REGION Network 12: UNIT 02 STATION 1 PART A PRESENT
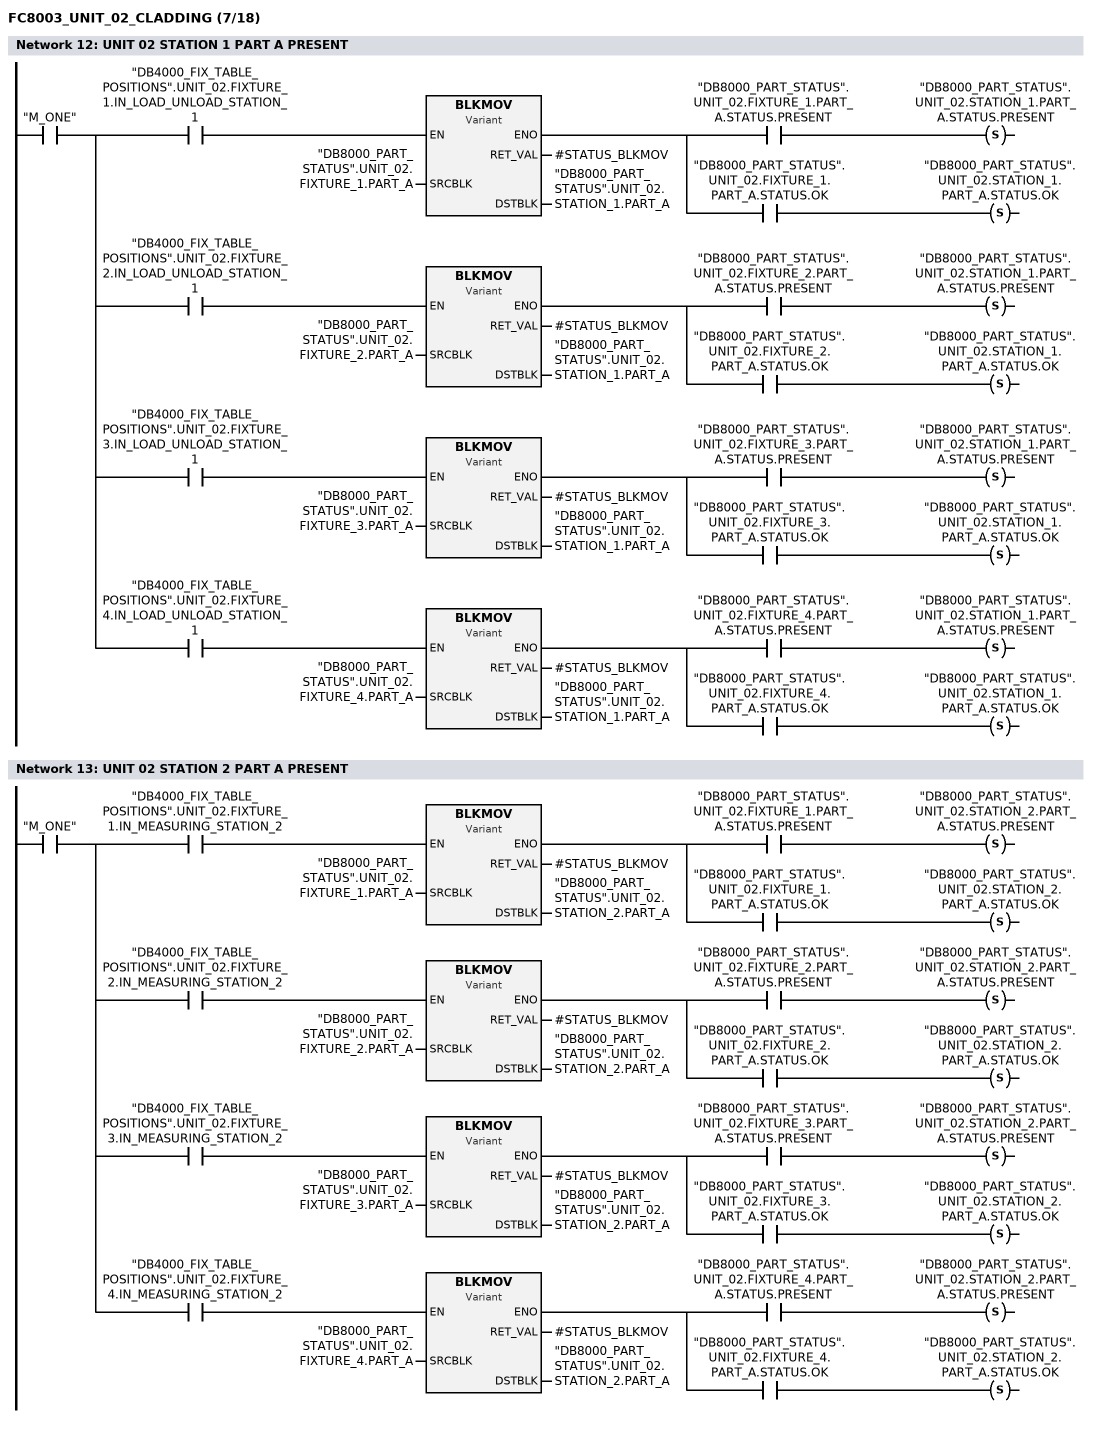
   RUNG wire#powerrail
      Contact( "M_ONE" )
      wire#w1
      Contact( "DB4000_FIX_TABLE_POSITIONS".UNIT_02.FIXTURE_1.IN_LOAD_UNLOAD_STATION_1 )
      { S7_Templates := "blk_type := Variant" } BLKMOV(SRCBLK := "DB8000_PART_STATUS".UNIT_02.FIXTURE_1.PART_A, RET_VAL => #STATUS_BLKMOV, DSTBLK => "DB8000_PART_STATUS".UNIT_02.STATION_1.PART_A)
      wire#w2
      Contact( "DB8000_PART_STATUS".UNIT_02.FIXTURE_1.PART_A.STATUS.PRESENT )
      S_Coil( "DB8000_PART_STATUS".UNIT_02.STATION_1.PART_A.STATUS.PRESENT )
   END_RUNG
   RUNG wire#w2
      Contact( "DB8000_PART_STATUS".UNIT_02.FIXTURE_1.PART_A.STATUS.OK )
      S_Coil( "DB8000_PART_STATUS".UNIT_02.STATION_1.PART_A.STATUS.OK )
   END_RUNG
   RUNG wire#w1
      Contact( "DB4000_FIX_TABLE_POSITIONS".UNIT_02.FIXTURE_2.IN_LOAD_UNLOAD_STATION_1 )
      { S7_Templates := "blk_type := Variant" } BLKMOV(SRCBLK := "DB8000_PART_STATUS".UNIT_02.FIXTURE_2.PART_A, RET_VAL => #STATUS_BLKMOV, DSTBLK => "DB8000_PART_STATUS".UNIT_02.STATION_1.PART_A)
      wire#w3
      Contact( "DB8000_PART_STATUS".UNIT_02.FIXTURE_2.PART_A.STATUS.PRESENT )
      S_Coil( "DB8000_PART_STATUS".UNIT_02.STATION_1.PART_A.STATUS.PRESENT )
   END_RUNG
   RUNG wire#w3
      Contact( "DB8000_PART_STATUS".UNIT_02.FIXTURE_2.PART_A.STATUS.OK )
      S_Coil( "DB8000_PART_STATUS".UNIT_02.STATION_1.PART_A.STATUS.OK )
   END_RUNG
   RUNG wire#w1
      Contact( "DB4000_FIX_TABLE_POSITIONS".UNIT_02.FIXTURE_3.IN_LOAD_UNLOAD_STATION_1 )
      { S7_Templates := "blk_type := Variant" } BLKMOV(SRCBLK := "DB8000_PART_STATUS".UNIT_02.FIXTURE_3.PART_A, RET_VAL => #STATUS_BLKMOV, DSTBLK => "DB8000_PART_STATUS".UNIT_02.STATION_1.PART_A)
      wire#w4
      Contact( "DB8000_PART_STATUS".UNIT_02.FIXTURE_3.PART_A.STATUS.PRESENT )
      S_Coil( "DB8000_PART_STATUS".UNIT_02.STATION_1.PART_A.STATUS.PRESENT )
   END_RUNG
   RUNG wire#w4
      Contact( "DB8000_PART_STATUS".UNIT_02.FIXTURE_3.PART_A.STATUS.OK )
      S_Coil( "DB8000_PART_STATUS".UNIT_02.STATION_1.PART_A.STATUS.OK )
   END_RUNG
   RUNG wire#w1
      Contact( "DB4000_FIX_TABLE_POSITIONS".UNIT_02.FIXTURE_4.IN_LOAD_UNLOAD_STATION_1 )
      { S7_Templates := "blk_type := Variant" } BLKMOV(SRCBLK := "DB8000_PART_STATUS".UNIT_02.FIXTURE_4.PART_A, RET_VAL => #STATUS_BLKMOV, DSTBLK => "DB8000_PART_STATUS".UNIT_02.STATION_1.PART_A)
      wire#w5
      Contact( "DB8000_PART_STATUS".UNIT_02.FIXTURE_4.PART_A.STATUS.PRESENT )
      S_Coil( "DB8000_PART_STATUS".UNIT_02.STATION_1.PART_A.STATUS.PRESENT )
   END_RUNG
   RUNG wire#w5
      Contact( "DB8000_PART_STATUS".UNIT_02.FIXTURE_4.PART_A.STATUS.OK )
      S_Coil( "DB8000_PART_STATUS".UNIT_02.STATION_1.PART_A.STATUS.OK )
   END_RUNG
   // the same network as SCL:
   #_w1 := "M_ONE" AND "DB4000_FIX_TABLE_POSITIONS".UNIT_02.FIXTURE_1.IN_LOAD_UNLOAD_STATION_1;
   #_w3 := "M_ONE";
   #STATUS_BLKMOV := BLKMOV(EN := #_w1,
                           SRCBLK := "DB8000_PART_STATUS".UNIT_02.FIXTURE_1.PART_A,
                           DSTBLK => "DB8000_PART_STATUS".UNIT_02.STATION_1.PART_A,
                           ENO => #_w2);
   IF #_w2 AND "DB8000_PART_STATUS".UNIT_02.FIXTURE_1.PART_A.STATUS.PRESENT THEN
       "DB8000_PART_STATUS".UNIT_02.STATION_1.PART_A.STATUS.PRESENT := TRUE;
   END_IF;
   IF #_w2 AND "DB8000_PART_STATUS".UNIT_02.FIXTURE_1.PART_A.STATUS.OK THEN
       "DB8000_PART_STATUS".UNIT_02.STATION_1.PART_A.STATUS.OK := TRUE;
   END_IF;
   #_w4 := #_w3 AND "DB4000_FIX_TABLE_POSITIONS".UNIT_02.FIXTURE_2.IN_LOAD_UNLOAD_STATION_1;
   #STATUS_BLKMOV := BLKMOV(EN := #_w4,
                           SRCBLK := "DB8000_PART_STATUS".UNIT_02.FIXTURE_2.PART_A,
                           DSTBLK => "DB8000_PART_STATUS".UNIT_02.STATION_1.PART_A,
                           ENO => #_w5);
   IF #_w5 AND "DB8000_PART_STATUS".UNIT_02.FIXTURE_2.PART_A.STATUS.PRESENT THEN
       "DB8000_PART_STATUS".UNIT_02.STATION_1.PART_A.STATUS.PRESENT := TRUE;
   END_IF;
   IF #_w5 AND "DB8000_PART_STATUS".UNIT_02.FIXTURE_2.PART_A.STATUS.OK THEN
       "DB8000_PART_STATUS".UNIT_02.STATION_1.PART_A.STATUS.OK := TRUE;
   END_IF;
   #_w6 := #_w3 AND "DB4000_FIX_TABLE_POSITIONS".UNIT_02.FIXTURE_3.IN_LOAD_UNLOAD_STATION_1;
   #STATUS_BLKMOV := BLKMOV(EN := #_w6,
                           SRCBLK := "DB8000_PART_STATUS".UNIT_02.FIXTURE_3.PART_A,
                           DSTBLK => "DB8000_PART_STATUS".UNIT_02.STATION_1.PART_A,
                           ENO => #_w7);
   IF #_w7 AND "DB8000_PART_STATUS".UNIT_02.FIXTURE_3.PART_A.STATUS.PRESENT THEN
       "DB8000_PART_STATUS".UNIT_02.STATION_1.PART_A.STATUS.PRESENT := TRUE;
   END_IF;
   IF #_w7 AND "DB8000_PART_STATUS".UNIT_02.FIXTURE_3.PART_A.STATUS.OK THEN
       "DB8000_PART_STATUS".UNIT_02.STATION_1.PART_A.STATUS.OK := TRUE;
   END_IF;
   #_w8 := #_w3 AND "DB4000_FIX_TABLE_POSITIONS".UNIT_02.FIXTURE_4.IN_LOAD_UNLOAD_STATION_1;
   #STATUS_BLKMOV := BLKMOV(EN := #_w8,
                           SRCBLK := "DB8000_PART_STATUS".UNIT_02.FIXTURE_4.PART_A,
                           DSTBLK => "DB8000_PART_STATUS".UNIT_02.STATION_1.PART_A,
                           ENO => #_w9);
   IF #_w9 AND "DB8000_PART_STATUS".UNIT_02.FIXTURE_4.PART_A.STATUS.PRESENT THEN
       "DB8000_PART_STATUS".UNIT_02.STATION_1.PART_A.STATUS.PRESENT := TRUE;
   END_IF;
   IF #_w9 AND "DB8000_PART_STATUS".UNIT_02.FIXTURE_4.PART_A.STATUS.OK THEN
       "DB8000_PART_STATUS".UNIT_02.STATION_1.PART_A.STATUS.OK := TRUE;
   END_IF;
END_REGION

REGION Network 13: UNIT 02 STATION 2 PART A PRESENT
   RUNG wire#powerrail
      Contact( "M_ONE" )
      wire#w1
      Contact( "DB4000_FIX_TABLE_POSITIONS".UNIT_02.FIXTURE_1.IN_MEASURING_STATION_2 )
      { S7_Templates := "blk_type := Variant" } BLKMOV(SRCBLK := "DB8000_PART_STATUS".UNIT_02.FIXTURE_1.PART_A, RET_VAL => #STATUS_BLKMOV, DSTBLK => "DB8000_PART_STATUS".UNIT_02.STATION_2.PART_A)
      wire#w2
      Contact( "DB8000_PART_STATUS".UNIT_02.FIXTURE_1.PART_A.STATUS.PRESENT )
      S_Coil( "DB8000_PART_STATUS".UNIT_02.STATION_2.PART_A.STATUS.PRESENT )
   END_RUNG
   RUNG wire#w2
      Contact( "DB8000_PART_STATUS".UNIT_02.FIXTURE_1.PART_A.STATUS.OK )
      S_Coil( "DB8000_PART_STATUS".UNIT_02.STATION_2.PART_A.STATUS.OK )
   END_RUNG
   RUNG wire#w1
      Contact( "DB4000_FIX_TABLE_POSITIONS".UNIT_02.FIXTURE_2.IN_MEASURING_STATION_2 )
      { S7_Templates := "blk_type := Variant" } BLKMOV(SRCBLK := "DB8000_PART_STATUS".UNIT_02.FIXTURE_2.PART_A, RET_VAL => #STATUS_BLKMOV, DSTBLK => "DB8000_PART_STATUS".UNIT_02.STATION_2.PART_A)
      wire#w3
      Contact( "DB8000_PART_STATUS".UNIT_02.FIXTURE_2.PART_A.STATUS.PRESENT )
      S_Coil( "DB8000_PART_STATUS".UNIT_02.STATION_2.PART_A.STATUS.PRESENT )
   END_RUNG
   RUNG wire#w3
      Contact( "DB8000_PART_STATUS".UNIT_02.FIXTURE_2.PART_A.STATUS.OK )
      S_Coil( "DB8000_PART_STATUS".UNIT_02.STATION_2.PART_A.STATUS.OK )
   END_RUNG
   RUNG wire#w1
      Contact( "DB4000_FIX_TABLE_POSITIONS".UNIT_02.FIXTURE_3.IN_MEASURING_STATION_2 )
      { S7_Templates := "blk_type := Variant" } BLKMOV(SRCBLK := "DB8000_PART_STATUS".UNIT_02.FIXTURE_3.PART_A, RET_VAL => #STATUS_BLKMOV, DSTBLK => "DB8000_PART_STATUS".UNIT_02.STATION_2.PART_A)
      wire#w4
      Contact( "DB8000_PART_STATUS".UNIT_02.FIXTURE_3.PART_A.STATUS.PRESENT )
      S_Coil( "DB8000_PART_STATUS".UNIT_02.STATION_2.PART_A.STATUS.PRESENT )
   END_RUNG
   RUNG wire#w4
      Contact( "DB8000_PART_STATUS".UNIT_02.FIXTURE_3.PART_A.STATUS.OK )
      S_Coil( "DB8000_PART_STATUS".UNIT_02.STATION_2.PART_A.STATUS.OK )
   END_RUNG
   RUNG wire#w1
      Contact( "DB4000_FIX_TABLE_POSITIONS".UNIT_02.FIXTURE_4.IN_MEASURING_STATION_2 )
      { S7_Templates := "blk_type := Variant" } BLKMOV(SRCBLK := "DB8000_PART_STATUS".UNIT_02.FIXTURE_4.PART_A, RET_VAL => #STATUS_BLKMOV, DSTBLK => "DB8000_PART_STATUS".UNIT_02.STATION_2.PART_A)
      wire#w5
      Contact( "DB8000_PART_STATUS".UNIT_02.FIXTURE_4.PART_A.STATUS.PRESENT )
      S_Coil( "DB8000_PART_STATUS".UNIT_02.STATION_2.PART_A.STATUS.PRESENT )
   END_RUNG
   RUNG wire#w5
      Contact( "DB8000_PART_STATUS".UNIT_02.FIXTURE_4.PART_A.STATUS.OK )
      S_Coil( "DB8000_PART_STATUS".UNIT_02.STATION_2.PART_A.STATUS.OK )
   END_RUNG
   // the same network as SCL:
   #_w1 := "M_ONE" AND "DB4000_FIX_TABLE_POSITIONS".UNIT_02.FIXTURE_1.IN_MEASURING_STATION_2;
   #_w3 := "M_ONE";
   #STATUS_BLKMOV := BLKMOV(EN := #_w1,
                           SRCBLK := "DB8000_PART_STATUS".UNIT_02.FIXTURE_1.PART_A,
                           DSTBLK => "DB8000_PART_STATUS".UNIT_02.STATION_2.PART_A,
                           ENO => #_w2);
   IF #_w2 AND "DB8000_PART_STATUS".UNIT_02.FIXTURE_1.PART_A.STATUS.PRESENT THEN
       "DB8000_PART_STATUS".UNIT_02.STATION_2.PART_A.STATUS.PRESENT := TRUE;
   END_IF;
   IF #_w2 AND "DB8000_PART_STATUS".UNIT_02.FIXTURE_1.PART_A.STATUS.OK THEN
       "DB8000_PART_STATUS".UNIT_02.STATION_2.PART_A.STATUS.OK := TRUE;
   END_IF;
   #_w4 := #_w3 AND "DB4000_FIX_TABLE_POSITIONS".UNIT_02.FIXTURE_2.IN_MEASURING_STATION_2;
   #STATUS_BLKMOV := BLKMOV(EN := #_w4,
                           SRCBLK := "DB8000_PART_STATUS".UNIT_02.FIXTURE_2.PART_A,
                           DSTBLK => "DB8000_PART_STATUS".UNIT_02.STATION_2.PART_A,
                           ENO => #_w5);
   IF #_w5 AND "DB8000_PART_STATUS".UNIT_02.FIXTURE_2.PART_A.STATUS.PRESENT THEN
       "DB8000_PART_STATUS".UNIT_02.STATION_2.PART_A.STATUS.PRESENT := TRUE;
   END_IF;
   IF #_w5 AND "DB8000_PART_STATUS".UNIT_02.FIXTURE_2.PART_A.STATUS.OK THEN
       "DB8000_PART_STATUS".UNIT_02.STATION_2.PART_A.STATUS.OK := TRUE;
   END_IF;
   #_w6 := #_w3 AND "DB4000_FIX_TABLE_POSITIONS".UNIT_02.FIXTURE_3.IN_MEASURING_STATION_2;
   #STATUS_BLKMOV := BLKMOV(EN := #_w6,
                           SRCBLK := "DB8000_PART_STATUS".UNIT_02.FIXTURE_3.PART_A,
                           DSTBLK => "DB8000_PART_STATUS".UNIT_02.STATION_2.PART_A,
                           ENO => #_w7);
   IF #_w7 AND "DB8000_PART_STATUS".UNIT_02.FIXTURE_3.PART_A.STATUS.PRESENT THEN
       "DB8000_PART_STATUS".UNIT_02.STATION_2.PART_A.STATUS.PRESENT := TRUE;
   END_IF;
   IF #_w7 AND "DB8000_PART_STATUS".UNIT_02.FIXTURE_3.PART_A.STATUS.OK THEN
       "DB8000_PART_STATUS".UNIT_02.STATION_2.PART_A.STATUS.OK := TRUE;
   END_IF;
   #_w8 := #_w3 AND "DB4000_FIX_TABLE_POSITIONS".UNIT_02.FIXTURE_4.IN_MEASURING_STATION_2;
   #STATUS_BLKMOV := BLKMOV(EN := #_w8,
                           SRCBLK := "DB8000_PART_STATUS".UNIT_02.FIXTURE_4.PART_A,
                           DSTBLK => "DB8000_PART_STATUS".UNIT_02.STATION_2.PART_A,
                           ENO => #_w9);
   IF #_w9 AND "DB8000_PART_STATUS".UNIT_02.FIXTURE_4.PART_A.STATUS.PRESENT THEN
       "DB8000_PART_STATUS".UNIT_02.STATION_2.PART_A.STATUS.PRESENT := TRUE;
   END_IF;
   IF #_w9 AND "DB8000_PART_STATUS".UNIT_02.FIXTURE_4.PART_A.STATUS.OK THEN
       "DB8000_PART_STATUS".UNIT_02.STATION_2.PART_A.STATUS.OK := TRUE;
   END_IF;
END_REGION

REGION Network 14: UNIT 02 STATION 3 PART A PRESENT
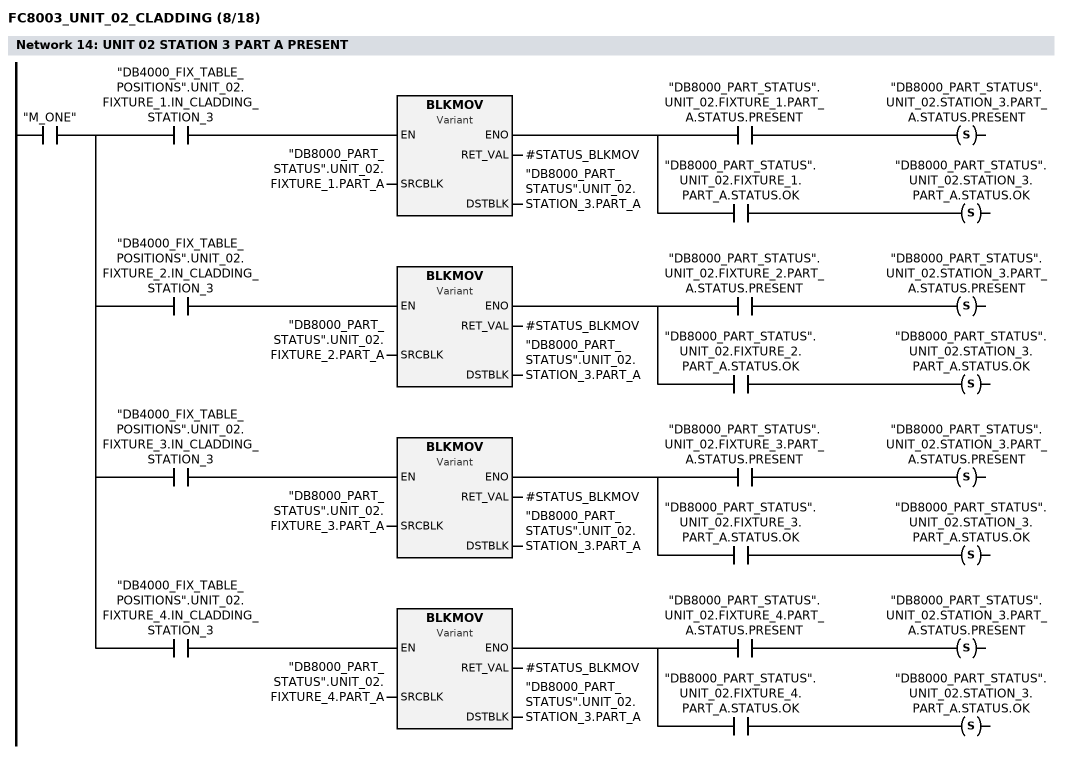
   RUNG wire#powerrail
      Contact( "M_ONE" )
      wire#w1
      Contact( "DB4000_FIX_TABLE_POSITIONS".UNIT_02.FIXTURE_1.IN_CLADDING_STATION_3 )
      { S7_Templates := "blk_type := Variant" } BLKMOV(SRCBLK := "DB8000_PART_STATUS".UNIT_02.FIXTURE_1.PART_A, RET_VAL => #STATUS_BLKMOV, DSTBLK => "DB8000_PART_STATUS".UNIT_02.STATION_3.PART_A)
      wire#w2
      Contact( "DB8000_PART_STATUS".UNIT_02.FIXTURE_1.PART_A.STATUS.PRESENT )
      S_Coil( "DB8000_PART_STATUS".UNIT_02.STATION_3.PART_A.STATUS.PRESENT )
   END_RUNG
   RUNG wire#w2
      Contact( "DB8000_PART_STATUS".UNIT_02.FIXTURE_1.PART_A.STATUS.OK )
      S_Coil( "DB8000_PART_STATUS".UNIT_02.STATION_3.PART_A.STATUS.OK )
   END_RUNG
   RUNG wire#w1
      Contact( "DB4000_FIX_TABLE_POSITIONS".UNIT_02.FIXTURE_2.IN_CLADDING_STATION_3 )
      { S7_Templates := "blk_type := Variant" } BLKMOV(SRCBLK := "DB8000_PART_STATUS".UNIT_02.FIXTURE_2.PART_A, RET_VAL => #STATUS_BLKMOV, DSTBLK => "DB8000_PART_STATUS".UNIT_02.STATION_3.PART_A)
      wire#w3
      Contact( "DB8000_PART_STATUS".UNIT_02.FIXTURE_2.PART_A.STATUS.PRESENT )
      S_Coil( "DB8000_PART_STATUS".UNIT_02.STATION_3.PART_A.STATUS.PRESENT )
   END_RUNG
   RUNG wire#w3
      Contact( "DB8000_PART_STATUS".UNIT_02.FIXTURE_2.PART_A.STATUS.OK )
      S_Coil( "DB8000_PART_STATUS".UNIT_02.STATION_3.PART_A.STATUS.OK )
   END_RUNG
   RUNG wire#w1
      Contact( "DB4000_FIX_TABLE_POSITIONS".UNIT_02.FIXTURE_3.IN_CLADDING_STATION_3 )
      { S7_Templates := "blk_type := Variant" } BLKMOV(SRCBLK := "DB8000_PART_STATUS".UNIT_02.FIXTURE_3.PART_A, RET_VAL => #STATUS_BLKMOV, DSTBLK => "DB8000_PART_STATUS".UNIT_02.STATION_3.PART_A)
      wire#w4
      Contact( "DB8000_PART_STATUS".UNIT_02.FIXTURE_3.PART_A.STATUS.PRESENT )
      S_Coil( "DB8000_PART_STATUS".UNIT_02.STATION_3.PART_A.STATUS.PRESENT )
   END_RUNG
   RUNG wire#w4
      Contact( "DB8000_PART_STATUS".UNIT_02.FIXTURE_3.PART_A.STATUS.OK )
      S_Coil( "DB8000_PART_STATUS".UNIT_02.STATION_3.PART_A.STATUS.OK )
   END_RUNG
   RUNG wire#w1
      Contact( "DB4000_FIX_TABLE_POSITIONS".UNIT_02.FIXTURE_4.IN_CLADDING_STATION_3 )
      { S7_Templates := "blk_type := Variant" } BLKMOV(SRCBLK := "DB8000_PART_STATUS".UNIT_02.FIXTURE_4.PART_A, RET_VAL => #STATUS_BLKMOV, DSTBLK => "DB8000_PART_STATUS".UNIT_02.STATION_3.PART_A)
      wire#w5
      Contact( "DB8000_PART_STATUS".UNIT_02.FIXTURE_4.PART_A.STATUS.PRESENT )
      S_Coil( "DB8000_PART_STATUS".UNIT_02.STATION_3.PART_A.STATUS.PRESENT )
   END_RUNG
   RUNG wire#w5
      Contact( "DB8000_PART_STATUS".UNIT_02.FIXTURE_4.PART_A.STATUS.OK )
      S_Coil( "DB8000_PART_STATUS".UNIT_02.STATION_3.PART_A.STATUS.OK )
   END_RUNG
   // the same network as SCL:
   #_w1 := "M_ONE" AND "DB4000_FIX_TABLE_POSITIONS".UNIT_02.FIXTURE_1.IN_CLADDING_STATION_3;
   #_w3 := "M_ONE";
   #STATUS_BLKMOV := BLKMOV(EN := #_w1,
                           SRCBLK := "DB8000_PART_STATUS".UNIT_02.FIXTURE_1.PART_A,
                           DSTBLK => "DB8000_PART_STATUS".UNIT_02.STATION_3.PART_A,
                           ENO => #_w2);
   IF #_w2 AND "DB8000_PART_STATUS".UNIT_02.FIXTURE_1.PART_A.STATUS.PRESENT THEN
       "DB8000_PART_STATUS".UNIT_02.STATION_3.PART_A.STATUS.PRESENT := TRUE;
   END_IF;
   IF #_w2 AND "DB8000_PART_STATUS".UNIT_02.FIXTURE_1.PART_A.STATUS.OK THEN
       "DB8000_PART_STATUS".UNIT_02.STATION_3.PART_A.STATUS.OK := TRUE;
   END_IF;
   #_w4 := #_w3 AND "DB4000_FIX_TABLE_POSITIONS".UNIT_02.FIXTURE_2.IN_CLADDING_STATION_3;
   #STATUS_BLKMOV := BLKMOV(EN := #_w4,
                           SRCBLK := "DB8000_PART_STATUS".UNIT_02.FIXTURE_2.PART_A,
                           DSTBLK => "DB8000_PART_STATUS".UNIT_02.STATION_3.PART_A,
                           ENO => #_w5);
   IF #_w5 AND "DB8000_PART_STATUS".UNIT_02.FIXTURE_2.PART_A.STATUS.PRESENT THEN
       "DB8000_PART_STATUS".UNIT_02.STATION_3.PART_A.STATUS.PRESENT := TRUE;
   END_IF;
   IF #_w5 AND "DB8000_PART_STATUS".UNIT_02.FIXTURE_2.PART_A.STATUS.OK THEN
       "DB8000_PART_STATUS".UNIT_02.STATION_3.PART_A.STATUS.OK := TRUE;
   END_IF;
   #_w6 := #_w3 AND "DB4000_FIX_TABLE_POSITIONS".UNIT_02.FIXTURE_3.IN_CLADDING_STATION_3;
   #STATUS_BLKMOV := BLKMOV(EN := #_w6,
                           SRCBLK := "DB8000_PART_STATUS".UNIT_02.FIXTURE_3.PART_A,
                           DSTBLK => "DB8000_PART_STATUS".UNIT_02.STATION_3.PART_A,
                           ENO => #_w7);
   IF #_w7 AND "DB8000_PART_STATUS".UNIT_02.FIXTURE_3.PART_A.STATUS.PRESENT THEN
       "DB8000_PART_STATUS".UNIT_02.STATION_3.PART_A.STATUS.PRESENT := TRUE;
   END_IF;
   IF #_w7 AND "DB8000_PART_STATUS".UNIT_02.FIXTURE_3.PART_A.STATUS.OK THEN
       "DB8000_PART_STATUS".UNIT_02.STATION_3.PART_A.STATUS.OK := TRUE;
   END_IF;
   #_w8 := #_w3 AND "DB4000_FIX_TABLE_POSITIONS".UNIT_02.FIXTURE_4.IN_CLADDING_STATION_3;
   #STATUS_BLKMOV := BLKMOV(EN := #_w8,
                           SRCBLK := "DB8000_PART_STATUS".UNIT_02.FIXTURE_4.PART_A,
                           DSTBLK => "DB8000_PART_STATUS".UNIT_02.STATION_3.PART_A,
                           ENO => #_w9);
   IF #_w9 AND "DB8000_PART_STATUS".UNIT_02.FIXTURE_4.PART_A.STATUS.PRESENT THEN
       "DB8000_PART_STATUS".UNIT_02.STATION_3.PART_A.STATUS.PRESENT := TRUE;
   END_IF;
   IF #_w9 AND "DB8000_PART_STATUS".UNIT_02.FIXTURE_4.PART_A.STATUS.OK THEN
       "DB8000_PART_STATUS".UNIT_02.STATION_3.PART_A.STATUS.OK := TRUE;
   END_IF;
END_REGION

REGION Network 15: UNIT 02 STATION 4 PART A PRESENT
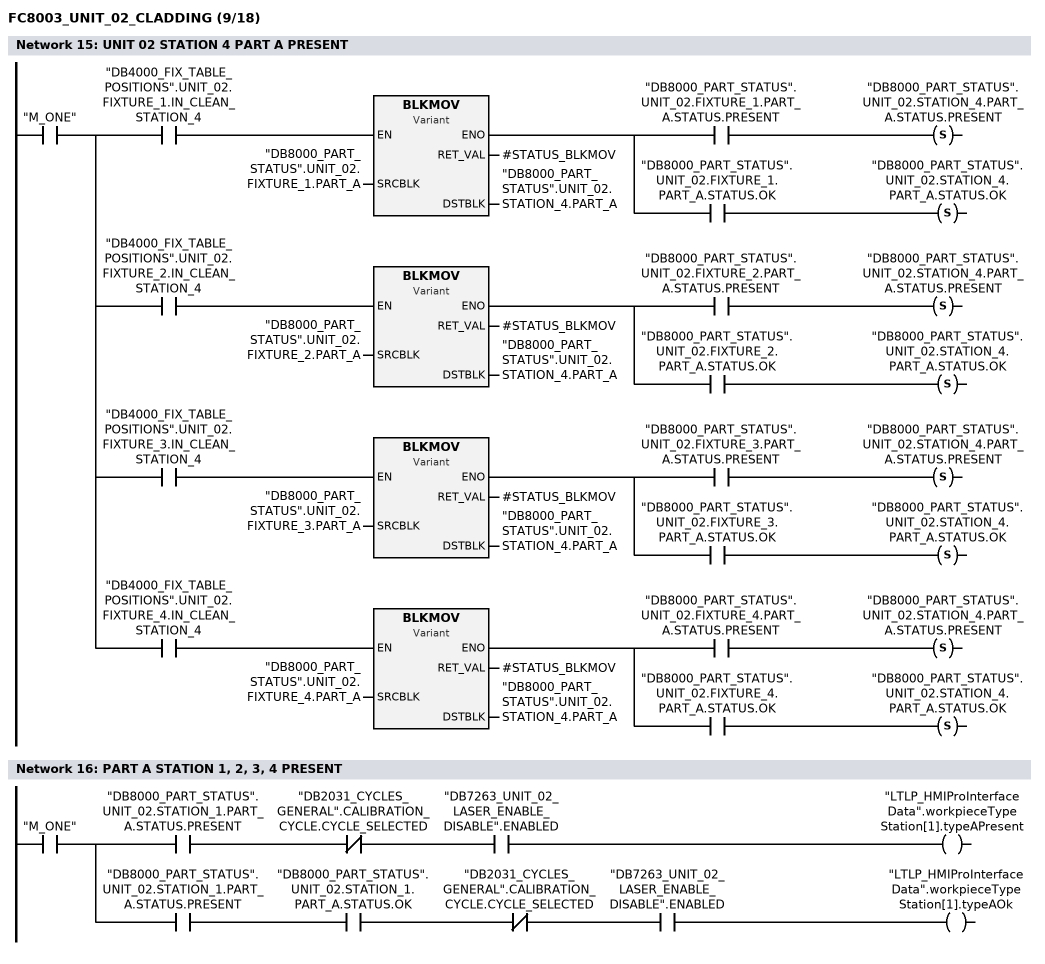
   RUNG wire#powerrail
      Contact( "M_ONE" )
      wire#w1
      Contact( "DB4000_FIX_TABLE_POSITIONS".UNIT_02.FIXTURE_1.IN_CLEAN_STATION_4 )
      { S7_Templates := "blk_type := Variant" } BLKMOV(SRCBLK := "DB8000_PART_STATUS".UNIT_02.FIXTURE_1.PART_A, RET_VAL => #STATUS_BLKMOV, DSTBLK => "DB8000_PART_STATUS".UNIT_02.STATION_4.PART_A)
      wire#w2
      Contact( "DB8000_PART_STATUS".UNIT_02.FIXTURE_1.PART_A.STATUS.PRESENT )
      S_Coil( "DB8000_PART_STATUS".UNIT_02.STATION_4.PART_A.STATUS.PRESENT )
   END_RUNG
   RUNG wire#w2
      Contact( "DB8000_PART_STATUS".UNIT_02.FIXTURE_1.PART_A.STATUS.OK )
      S_Coil( "DB8000_PART_STATUS".UNIT_02.STATION_4.PART_A.STATUS.OK )
   END_RUNG
   RUNG wire#w1
      Contact( "DB4000_FIX_TABLE_POSITIONS".UNIT_02.FIXTURE_2.IN_CLEAN_STATION_4 )
      { S7_Templates := "blk_type := Variant" } BLKMOV(SRCBLK := "DB8000_PART_STATUS".UNIT_02.FIXTURE_2.PART_A, RET_VAL => #STATUS_BLKMOV, DSTBLK => "DB8000_PART_STATUS".UNIT_02.STATION_4.PART_A)
      wire#w3
      Contact( "DB8000_PART_STATUS".UNIT_02.FIXTURE_2.PART_A.STATUS.PRESENT )
      S_Coil( "DB8000_PART_STATUS".UNIT_02.STATION_4.PART_A.STATUS.PRESENT )
   END_RUNG
   RUNG wire#w3
      Contact( "DB8000_PART_STATUS".UNIT_02.FIXTURE_2.PART_A.STATUS.OK )
      S_Coil( "DB8000_PART_STATUS".UNIT_02.STATION_4.PART_A.STATUS.OK )
   END_RUNG
   RUNG wire#w1
      Contact( "DB4000_FIX_TABLE_POSITIONS".UNIT_02.FIXTURE_3.IN_CLEAN_STATION_4 )
      { S7_Templates := "blk_type := Variant" } BLKMOV(SRCBLK := "DB8000_PART_STATUS".UNIT_02.FIXTURE_3.PART_A, RET_VAL => #STATUS_BLKMOV, DSTBLK => "DB8000_PART_STATUS".UNIT_02.STATION_4.PART_A)
      wire#w4
      Contact( "DB8000_PART_STATUS".UNIT_02.FIXTURE_3.PART_A.STATUS.PRESENT )
      S_Coil( "DB8000_PART_STATUS".UNIT_02.STATION_4.PART_A.STATUS.PRESENT )
   END_RUNG
   RUNG wire#w4
      Contact( "DB8000_PART_STATUS".UNIT_02.FIXTURE_3.PART_A.STATUS.OK )
      S_Coil( "DB8000_PART_STATUS".UNIT_02.STATION_4.PART_A.STATUS.OK )
   END_RUNG
   RUNG wire#w1
      Contact( "DB4000_FIX_TABLE_POSITIONS".UNIT_02.FIXTURE_4.IN_CLEAN_STATION_4 )
      { S7_Templates := "blk_type := Variant" } BLKMOV(SRCBLK := "DB8000_PART_STATUS".UNIT_02.FIXTURE_4.PART_A, RET_VAL => #STATUS_BLKMOV, DSTBLK => "DB8000_PART_STATUS".UNIT_02.STATION_4.PART_A)
      wire#w5
      Contact( "DB8000_PART_STATUS".UNIT_02.FIXTURE_4.PART_A.STATUS.PRESENT )
      S_Coil( "DB8000_PART_STATUS".UNIT_02.STATION_4.PART_A.STATUS.PRESENT )
   END_RUNG
   RUNG wire#w5
      Contact( "DB8000_PART_STATUS".UNIT_02.FIXTURE_4.PART_A.STATUS.OK )
      S_Coil( "DB8000_PART_STATUS".UNIT_02.STATION_4.PART_A.STATUS.OK )
   END_RUNG
   // the same network as SCL:
   #_w1 := "M_ONE" AND "DB4000_FIX_TABLE_POSITIONS".UNIT_02.FIXTURE_1.IN_CLEAN_STATION_4;
   #_w3 := "M_ONE";
   #STATUS_BLKMOV := BLKMOV(EN := #_w1,
                           SRCBLK := "DB8000_PART_STATUS".UNIT_02.FIXTURE_1.PART_A,
                           DSTBLK => "DB8000_PART_STATUS".UNIT_02.STATION_4.PART_A,
                           ENO => #_w2);
   IF #_w2 AND "DB8000_PART_STATUS".UNIT_02.FIXTURE_1.PART_A.STATUS.PRESENT THEN
       "DB8000_PART_STATUS".UNIT_02.STATION_4.PART_A.STATUS.PRESENT := TRUE;
   END_IF;
   IF #_w2 AND "DB8000_PART_STATUS".UNIT_02.FIXTURE_1.PART_A.STATUS.OK THEN
       "DB8000_PART_STATUS".UNIT_02.STATION_4.PART_A.STATUS.OK := TRUE;
   END_IF;
   #_w4 := #_w3 AND "DB4000_FIX_TABLE_POSITIONS".UNIT_02.FIXTURE_2.IN_CLEAN_STATION_4;
   #STATUS_BLKMOV := BLKMOV(EN := #_w4,
                           SRCBLK := "DB8000_PART_STATUS".UNIT_02.FIXTURE_2.PART_A,
                           DSTBLK => "DB8000_PART_STATUS".UNIT_02.STATION_4.PART_A,
                           ENO => #_w5);
   IF #_w5 AND "DB8000_PART_STATUS".UNIT_02.FIXTURE_2.PART_A.STATUS.PRESENT THEN
       "DB8000_PART_STATUS".UNIT_02.STATION_4.PART_A.STATUS.PRESENT := TRUE;
   END_IF;
   IF #_w5 AND "DB8000_PART_STATUS".UNIT_02.FIXTURE_2.PART_A.STATUS.OK THEN
       "DB8000_PART_STATUS".UNIT_02.STATION_4.PART_A.STATUS.OK := TRUE;
   END_IF;
   #_w6 := #_w3 AND "DB4000_FIX_TABLE_POSITIONS".UNIT_02.FIXTURE_3.IN_CLEAN_STATION_4;
   #STATUS_BLKMOV := BLKMOV(EN := #_w6,
                           SRCBLK := "DB8000_PART_STATUS".UNIT_02.FIXTURE_3.PART_A,
                           DSTBLK => "DB8000_PART_STATUS".UNIT_02.STATION_4.PART_A,
                           ENO => #_w7);
   IF #_w7 AND "DB8000_PART_STATUS".UNIT_02.FIXTURE_3.PART_A.STATUS.PRESENT THEN
       "DB8000_PART_STATUS".UNIT_02.STATION_4.PART_A.STATUS.PRESENT := TRUE;
   END_IF;
   IF #_w7 AND "DB8000_PART_STATUS".UNIT_02.FIXTURE_3.PART_A.STATUS.OK THEN
       "DB8000_PART_STATUS".UNIT_02.STATION_4.PART_A.STATUS.OK := TRUE;
   END_IF;
   #_w8 := #_w3 AND "DB4000_FIX_TABLE_POSITIONS".UNIT_02.FIXTURE_4.IN_CLEAN_STATION_4;
   #STATUS_BLKMOV := BLKMOV(EN := #_w8,
                           SRCBLK := "DB8000_PART_STATUS".UNIT_02.FIXTURE_4.PART_A,
                           DSTBLK => "DB8000_PART_STATUS".UNIT_02.STATION_4.PART_A,
                           ENO => #_w9);
   IF #_w9 AND "DB8000_PART_STATUS".UNIT_02.FIXTURE_4.PART_A.STATUS.PRESENT THEN
       "DB8000_PART_STATUS".UNIT_02.STATION_4.PART_A.STATUS.PRESENT := TRUE;
   END_IF;
   IF #_w9 AND "DB8000_PART_STATUS".UNIT_02.FIXTURE_4.PART_A.STATUS.OK THEN
       "DB8000_PART_STATUS".UNIT_02.STATION_4.PART_A.STATUS.OK := TRUE;
   END_IF;
END_REGION

REGION Network 16: PART A STATION 1, 2, 3, 4 PRESENT
   RUNG wire#powerrail
      Contact( "M_ONE" )
      wire#w1
      Contact( "DB8000_PART_STATUS".UNIT_02.STATION_1.PART_A.STATUS.PRESENT )
      I_Contact( "DB2031_CYCLES_GENERAL".CALIBRATION_CYCLE.CYCLE_SELECTED )
      Contact( "DB7263_UNIT_02_LASER_ENABLE_DISABLE".ENABLED )
      Coil( "LTLP_HMIProInterfaceData".workpieceTypeStation[1].typeAPresent )
   END_RUNG
   RUNG wire#w1
      Contact( "DB8000_PART_STATUS".UNIT_02.STATION_1.PART_A.STATUS.PRESENT )
      Contact( "DB8000_PART_STATUS".UNIT_02.STATION_1.PART_A.STATUS.OK )
      I_Contact( "DB2031_CYCLES_GENERAL".CALIBRATION_CYCLE.CYCLE_SELECTED )
      Contact( "DB7263_UNIT_02_LASER_ENABLE_DISABLE".ENABLED )
      Coil( "LTLP_HMIProInterfaceData".workpieceTypeStation[1].typeAOk )
   END_RUNG
   // the same network as SCL:
   "LTLP_HMIProInterfaceData".workpieceTypeStation[1].typeAPresent := "M_ONE" AND "DB8000_PART_STATUS".UNIT_02.STATION_1.PART_A.STATUS.PRESENT AND NOT "DB2031_CYCLES_GENERAL".CALIBRATION_CYCLE.CYCLE_SELECTED AND "DB7263_UNIT_02_LASER_ENABLE_DISABLE".ENABLED;
   "LTLP_HMIProInterfaceData".workpieceTypeStation[1].typeAOk := "M_ONE" AND "DB8000_PART_STATUS".UNIT_02.STATION_1.PART_A.STATUS.PRESENT AND "DB8000_PART_STATUS".UNIT_02.STATION_1.PART_A.STATUS.OK AND NOT "DB2031_CYCLES_GENERAL".CALIBRATION_CYCLE.CYCLE_SELECTED AND "DB7263_UNIT_02_LASER_ENABLE_DISABLE".ENABLED;
END_REGION

REGION Network 17: PART A FIXTURE 1, 2, 3, 4 RESET STATUS TO ZERO
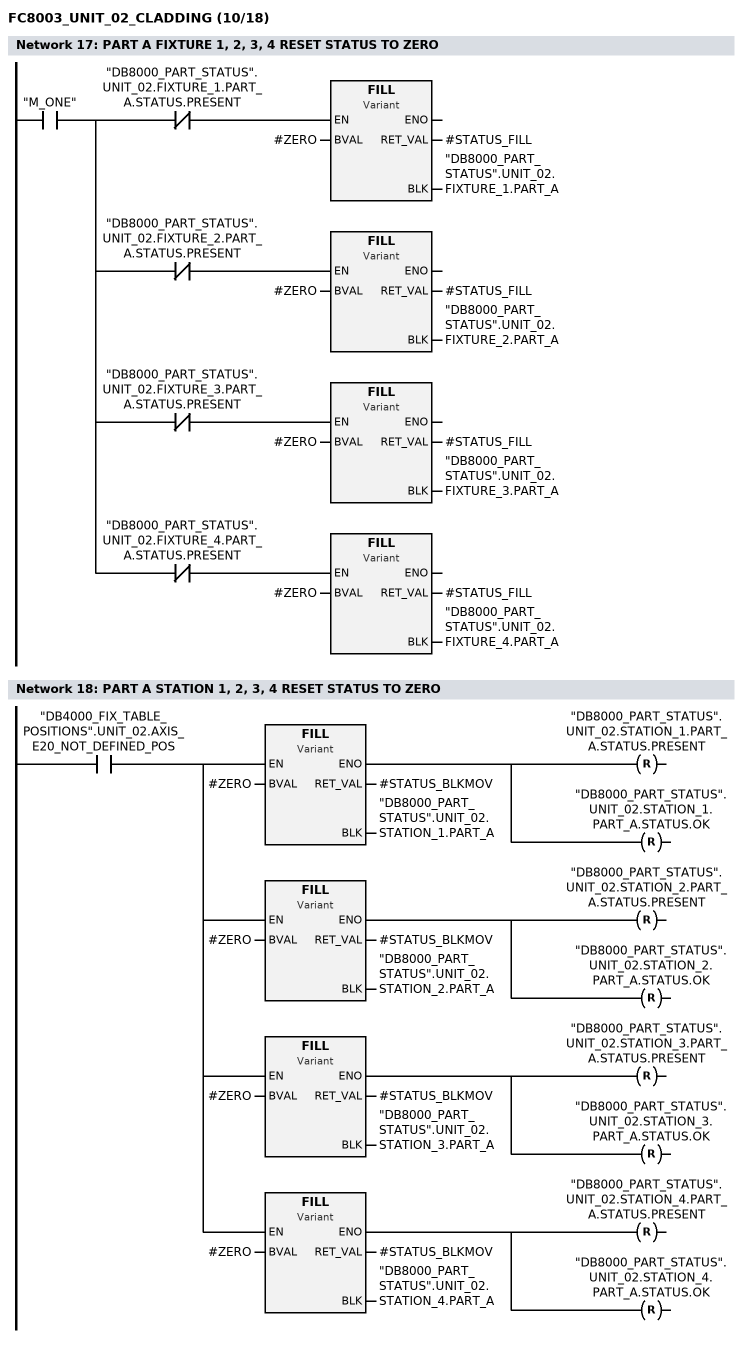
   RUNG wire#powerrail
      Contact( "M_ONE" )
      wire#w1
      I_Contact( "DB8000_PART_STATUS".UNIT_02.FIXTURE_1.PART_A.STATUS.PRESENT )
      { S7_Templates := "ptr_type := Variant" } FILL(BVAL := #ZERO, RET_VAL => #STATUS_FILL, BLK => "DB8000_PART_STATUS".UNIT_02.FIXTURE_1.PART_A)
   END_RUNG
   RUNG wire#w1
      I_Contact( "DB8000_PART_STATUS".UNIT_02.FIXTURE_2.PART_A.STATUS.PRESENT )
      { S7_Templates := "ptr_type := Variant" } FILL(BVAL := #ZERO, RET_VAL => #STATUS_FILL, BLK => "DB8000_PART_STATUS".UNIT_02.FIXTURE_2.PART_A)
   END_RUNG
   RUNG wire#w1
      I_Contact( "DB8000_PART_STATUS".UNIT_02.FIXTURE_3.PART_A.STATUS.PRESENT )
      { S7_Templates := "ptr_type := Variant" } FILL(BVAL := #ZERO, RET_VAL => #STATUS_FILL, BLK => "DB8000_PART_STATUS".UNIT_02.FIXTURE_3.PART_A)
   END_RUNG
   RUNG wire#w1
      I_Contact( "DB8000_PART_STATUS".UNIT_02.FIXTURE_4.PART_A.STATUS.PRESENT )
      { S7_Templates := "ptr_type := Variant" } FILL(BVAL := #ZERO, RET_VAL => #STATUS_FILL, BLK => "DB8000_PART_STATUS".UNIT_02.FIXTURE_4.PART_A)
   END_RUNG
   // the same network as SCL:
   #_w1 := "M_ONE";
   IF "M_ONE" AND NOT "DB8000_PART_STATUS".UNIT_02.FIXTURE_1.PART_A.STATUS.PRESENT THEN
       #STATUS_FILL := FILL(BVAL := #ZERO, BLK => "DB8000_PART_STATUS".UNIT_02.FIXTURE_1.PART_A);
   END_IF;
   IF #_w1 AND NOT "DB8000_PART_STATUS".UNIT_02.FIXTURE_2.PART_A.STATUS.PRESENT THEN
       #STATUS_FILL := FILL(BVAL := #ZERO, BLK => "DB8000_PART_STATUS".UNIT_02.FIXTURE_2.PART_A);
   END_IF;
   IF #_w1 AND NOT "DB8000_PART_STATUS".UNIT_02.FIXTURE_3.PART_A.STATUS.PRESENT THEN
       #STATUS_FILL := FILL(BVAL := #ZERO, BLK => "DB8000_PART_STATUS".UNIT_02.FIXTURE_3.PART_A);
   END_IF;
   IF #_w1 AND NOT "DB8000_PART_STATUS".UNIT_02.FIXTURE_4.PART_A.STATUS.PRESENT THEN
       #STATUS_FILL := FILL(BVAL := #ZERO, BLK => "DB8000_PART_STATUS".UNIT_02.FIXTURE_4.PART_A);
   END_IF;
END_REGION

REGION Network 18: PART A STATION 1, 2, 3, 4 RESET STATUS TO ZERO
   RUNG wire#powerrail
      Contact( "DB4000_FIX_TABLE_POSITIONS".UNIT_02.AXIS_E20_NOT_DEFINED_POS )
      wire#w1
      { S7_Templates := "ptr_type := Variant" } FILL(BVAL := #ZERO, RET_VAL => #STATUS_BLKMOV, BLK => "DB8000_PART_STATUS".UNIT_02.STATION_1.PART_A)
      wire#w2
      R_Coil( "DB8000_PART_STATUS".UNIT_02.STATION_1.PART_A.STATUS.PRESENT )
   END_RUNG
   RUNG wire#w2
      R_Coil( "DB8000_PART_STATUS".UNIT_02.STATION_1.PART_A.STATUS.OK )
   END_RUNG
   RUNG wire#w1
      { S7_Templates := "ptr_type := Variant" } FILL(BVAL := #ZERO, RET_VAL => #STATUS_BLKMOV, BLK => "DB8000_PART_STATUS".UNIT_02.STATION_2.PART_A)
      wire#w3
      R_Coil( "DB8000_PART_STATUS".UNIT_02.STATION_2.PART_A.STATUS.PRESENT )
   END_RUNG
   RUNG wire#w3
      R_Coil( "DB8000_PART_STATUS".UNIT_02.STATION_2.PART_A.STATUS.OK )
   END_RUNG
   RUNG wire#w1
      { S7_Templates := "ptr_type := Variant" } FILL(BVAL := #ZERO, RET_VAL => #STATUS_BLKMOV, BLK => "DB8000_PART_STATUS".UNIT_02.STATION_3.PART_A)
      wire#w4
      R_Coil( "DB8000_PART_STATUS".UNIT_02.STATION_3.PART_A.STATUS.PRESENT )
   END_RUNG
   RUNG wire#w4
      R_Coil( "DB8000_PART_STATUS".UNIT_02.STATION_3.PART_A.STATUS.OK )
   END_RUNG
   RUNG wire#w1
      { S7_Templates := "ptr_type := Variant" } FILL(BVAL := #ZERO, RET_VAL => #STATUS_BLKMOV, BLK => "DB8000_PART_STATUS".UNIT_02.STATION_4.PART_A)
      wire#w5
      R_Coil( "DB8000_PART_STATUS".UNIT_02.STATION_4.PART_A.STATUS.PRESENT )
   END_RUNG
   RUNG wire#w5
      R_Coil( "DB8000_PART_STATUS".UNIT_02.STATION_4.PART_A.STATUS.OK )
   END_RUNG
   // the same network as SCL:
   #_w2 := "DB4000_FIX_TABLE_POSITIONS".UNIT_02.AXIS_E20_NOT_DEFINED_POS;
   #STATUS_BLKMOV := FILL(EN := "DB4000_FIX_TABLE_POSITIONS".UNIT_02.AXIS_E20_NOT_DEFINED_POS,
                          BVAL := #ZERO,
                          BLK => "DB8000_PART_STATUS".UNIT_02.STATION_1.PART_A,
                          ENO => #_w1);
   IF #_w1 THEN
       "DB8000_PART_STATUS".UNIT_02.STATION_1.PART_A.STATUS.PRESENT := FALSE;
       "DB8000_PART_STATUS".UNIT_02.STATION_1.PART_A.STATUS.OK := FALSE;
   END_IF;
   #STATUS_BLKMOV := FILL(EN := #_w2,
                          BVAL := #ZERO,
                          BLK => "DB8000_PART_STATUS".UNIT_02.STATION_2.PART_A,
                          ENO => #_w3);
   IF #_w3 THEN
       "DB8000_PART_STATUS".UNIT_02.STATION_2.PART_A.STATUS.PRESENT := FALSE;
       "DB8000_PART_STATUS".UNIT_02.STATION_2.PART_A.STATUS.OK := FALSE;
   END_IF;
   #STATUS_BLKMOV := FILL(EN := #_w2,
                          BVAL := #ZERO,
                          BLK => "DB8000_PART_STATUS".UNIT_02.STATION_3.PART_A,
                          ENO => #_w4);
   IF #_w4 THEN
       "DB8000_PART_STATUS".UNIT_02.STATION_3.PART_A.STATUS.PRESENT := FALSE;
       "DB8000_PART_STATUS".UNIT_02.STATION_3.PART_A.STATUS.OK := FALSE;
   END_IF;
   #STATUS_BLKMOV := FILL(EN := #_w2,
                          BVAL := #ZERO,
                          BLK => "DB8000_PART_STATUS".UNIT_02.STATION_4.PART_A,
                          ENO => #_w5);
   IF #_w5 THEN
       "DB8000_PART_STATUS".UNIT_02.STATION_4.PART_A.STATUS.PRESENT := FALSE;
       "DB8000_PART_STATUS".UNIT_02.STATION_4.PART_A.STATUS.OK := FALSE;
   END_IF;
END_REGION

REGION Network 19: PART A FIXTURE 1 COLOR STATUS
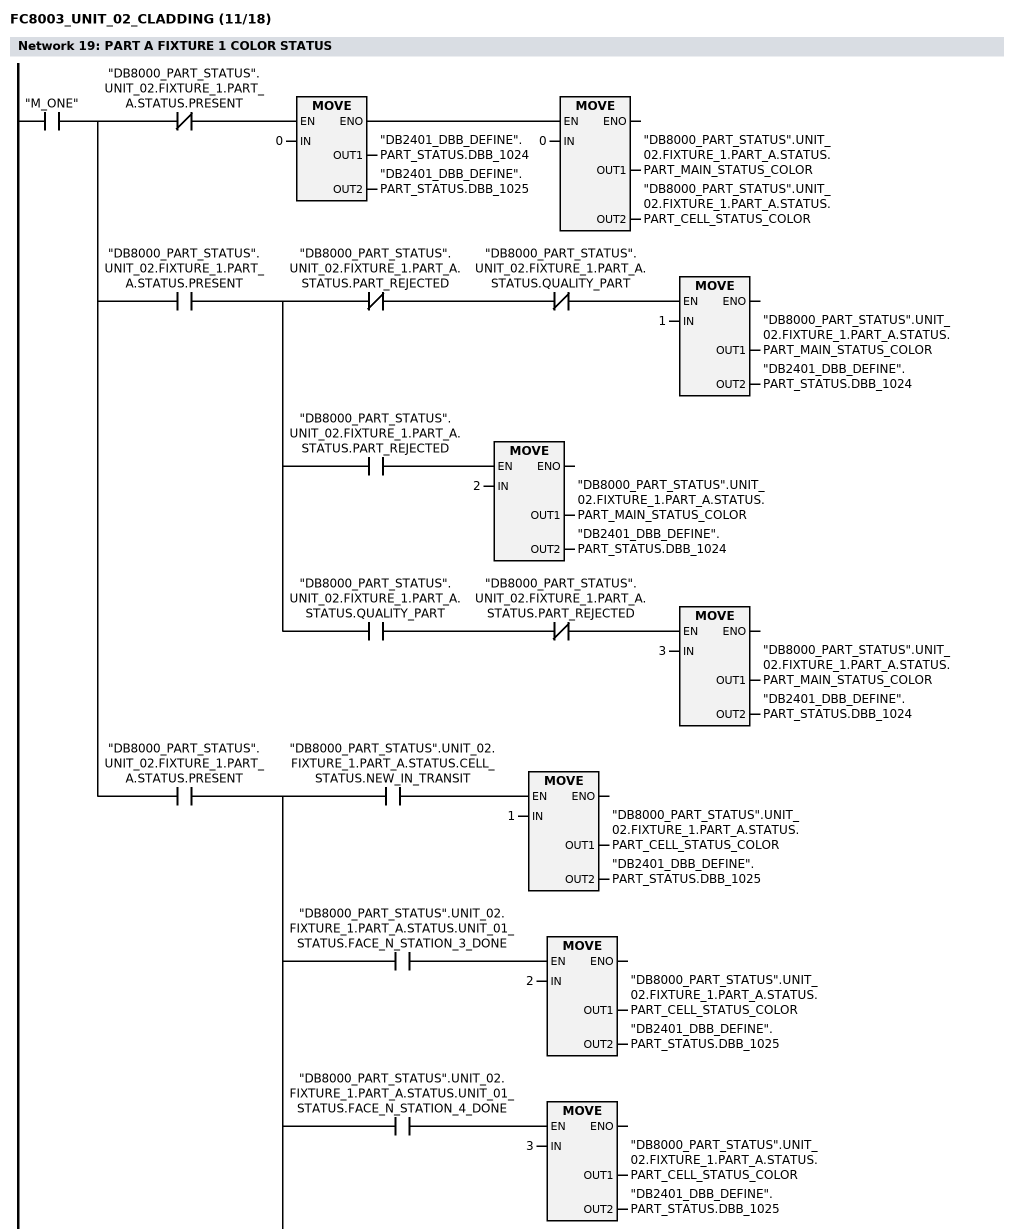
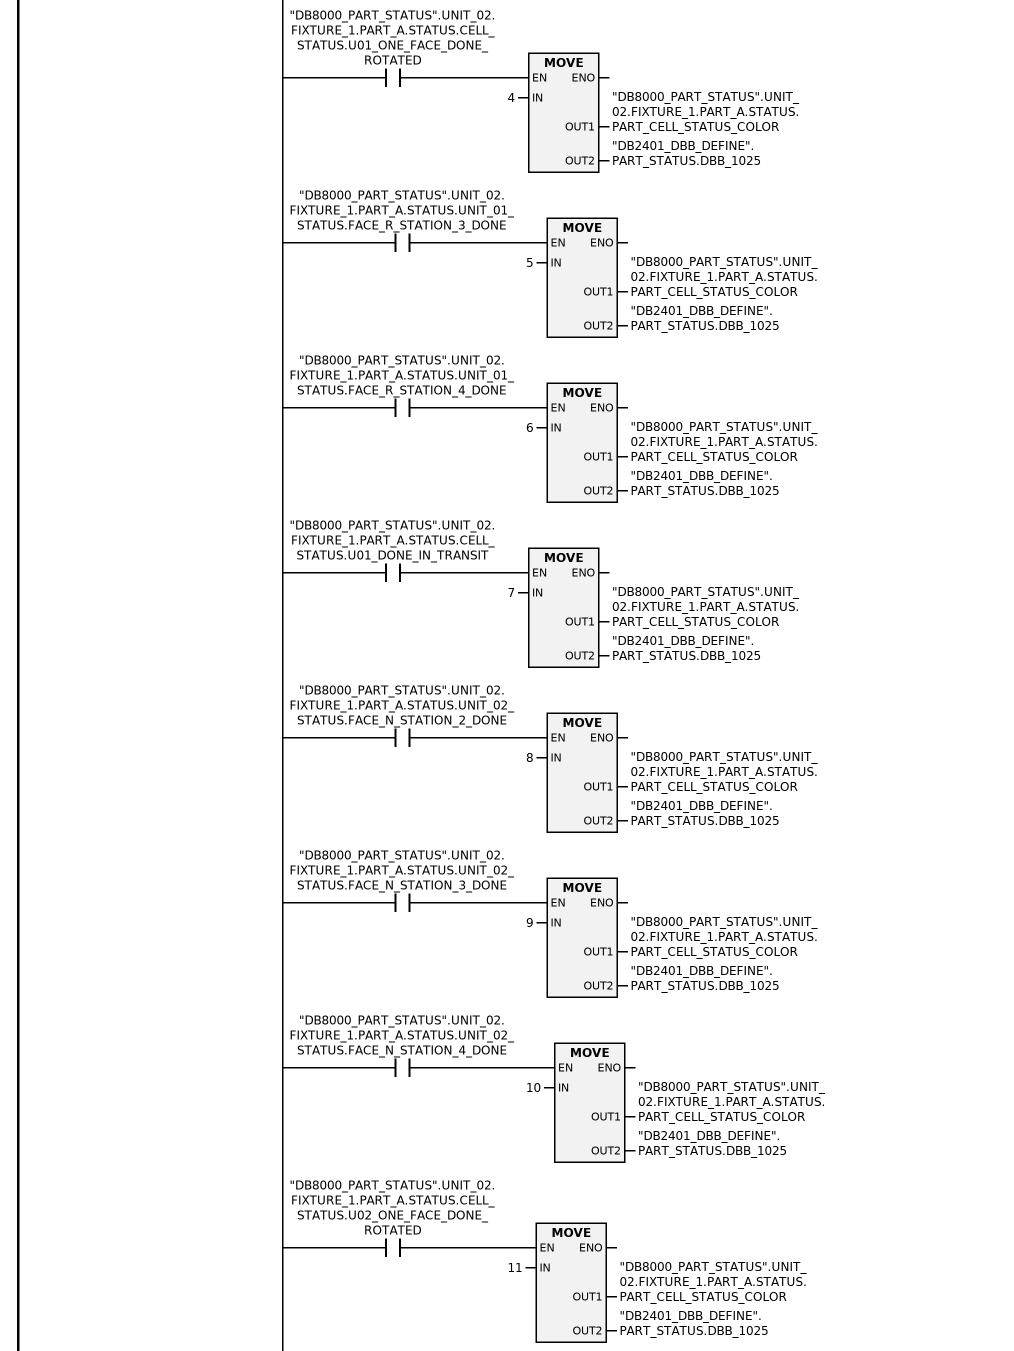
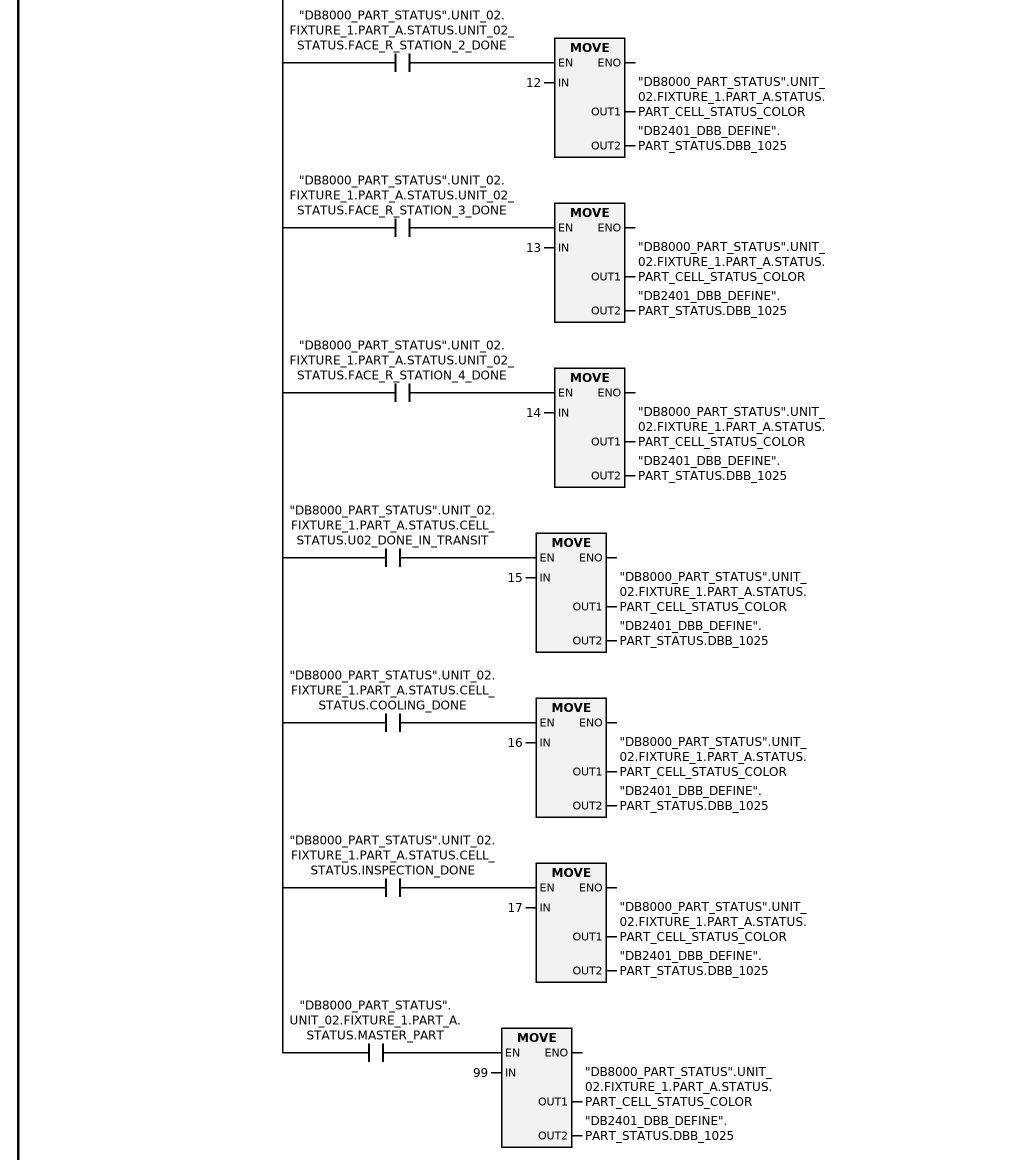
   RUNG wire#powerrail
      Contact( "M_ONE" )
      wire#w1
      I_Contact( "DB8000_PART_STATUS".UNIT_02.FIXTURE_1.PART_A.STATUS.PRESENT )
      { S7_GenerateENO := "TRUE" } Move(in := 0, out1 => "DB2401_DBB_DEFINE".PART_STATUS.DBB_1024, out2 => "DB2401_DBB_DEFINE".PART_STATUS.DBB_1025)
      { S7_GenerateENO := "TRUE" } Move(in := 0, out1 => "DB8000_PART_STATUS".UNIT_02.FIXTURE_1.PART_A.STATUS.PART_MAIN_STATUS_COLOR, out2 => "DB8000_PART_STATUS".UNIT_02.FIXTURE_1.PART_A.STATUS.PART_CELL_STATUS_COLOR)
   END_RUNG
   RUNG wire#w1
      Contact( "DB8000_PART_STATUS".UNIT_02.FIXTURE_1.PART_A.STATUS.PRESENT )
      wire#w2
      I_Contact( "DB8000_PART_STATUS".UNIT_02.FIXTURE_1.PART_A.STATUS.PART_REJECTED )
      I_Contact( "DB8000_PART_STATUS".UNIT_02.FIXTURE_1.PART_A.STATUS.QUALITY_PART )
      { S7_GenerateENO := "TRUE" } Move(in := 1, out1 => "DB8000_PART_STATUS".UNIT_02.FIXTURE_1.PART_A.STATUS.PART_MAIN_STATUS_COLOR, out2 => "DB2401_DBB_DEFINE".PART_STATUS.DBB_1024)
   END_RUNG
   RUNG wire#w2
      Contact( "DB8000_PART_STATUS".UNIT_02.FIXTURE_1.PART_A.STATUS.PART_REJECTED )
      { S7_GenerateENO := "TRUE" } Move(in := 2, out1 => "DB8000_PART_STATUS".UNIT_02.FIXTURE_1.PART_A.STATUS.PART_MAIN_STATUS_COLOR, out2 => "DB2401_DBB_DEFINE".PART_STATUS.DBB_1024)
   END_RUNG
   RUNG wire#w2
      Contact( "DB8000_PART_STATUS".UNIT_02.FIXTURE_1.PART_A.STATUS.QUALITY_PART )
      I_Contact( "DB8000_PART_STATUS".UNIT_02.FIXTURE_1.PART_A.STATUS.PART_REJECTED )
      { S7_GenerateENO := "TRUE" } Move(in := 3, out1 => "DB8000_PART_STATUS".UNIT_02.FIXTURE_1.PART_A.STATUS.PART_MAIN_STATUS_COLOR, out2 => "DB2401_DBB_DEFINE".PART_STATUS.DBB_1024)
   END_RUNG
   RUNG wire#w1
      Contact( "DB8000_PART_STATUS".UNIT_02.FIXTURE_1.PART_A.STATUS.PRESENT )
      wire#w3
      Contact( "DB8000_PART_STATUS".UNIT_02.FIXTURE_1.PART_A.STATUS.CELL_STATUS.NEW_IN_TRANSIT )
      { S7_GenerateENO := "TRUE" } Move(in := 1, out1 => "DB8000_PART_STATUS".UNIT_02.FIXTURE_1.PART_A.STATUS.PART_CELL_STATUS_COLOR, out2 => "DB2401_DBB_DEFINE".PART_STATUS.DBB_1025)
   END_RUNG
   RUNG wire#w3
      Contact( "DB8000_PART_STATUS".UNIT_02.FIXTURE_1.PART_A.STATUS.UNIT_01_STATUS.FACE_N_STATION_3_DONE )
      { S7_GenerateENO := "TRUE" } Move(in := 2, out1 => "DB8000_PART_STATUS".UNIT_02.FIXTURE_1.PART_A.STATUS.PART_CELL_STATUS_COLOR, out2 => "DB2401_DBB_DEFINE".PART_STATUS.DBB_1025)
   END_RUNG
   RUNG wire#w3
      Contact( "DB8000_PART_STATUS".UNIT_02.FIXTURE_1.PART_A.STATUS.UNIT_01_STATUS.FACE_N_STATION_4_DONE )
      { S7_GenerateENO := "TRUE" } Move(in := 3, out1 => "DB8000_PART_STATUS".UNIT_02.FIXTURE_1.PART_A.STATUS.PART_CELL_STATUS_COLOR, out2 => "DB2401_DBB_DEFINE".PART_STATUS.DBB_1025)
   END_RUNG
   RUNG wire#w3
      Contact( "DB8000_PART_STATUS".UNIT_02.FIXTURE_1.PART_A.STATUS.CELL_STATUS.U01_ONE_FACE_DONE_ROTATED )
      { S7_GenerateENO := "TRUE" } Move(in := 4, out1 => "DB8000_PART_STATUS".UNIT_02.FIXTURE_1.PART_A.STATUS.PART_CELL_STATUS_COLOR, out2 => "DB2401_DBB_DEFINE".PART_STATUS.DBB_1025)
   END_RUNG
   RUNG wire#w3
      Contact( "DB8000_PART_STATUS".UNIT_02.FIXTURE_1.PART_A.STATUS.UNIT_01_STATUS.FACE_R_STATION_3_DONE )
      { S7_GenerateENO := "TRUE" } Move(in := 5, out1 => "DB8000_PART_STATUS".UNIT_02.FIXTURE_1.PART_A.STATUS.PART_CELL_STATUS_COLOR, out2 => "DB2401_DBB_DEFINE".PART_STATUS.DBB_1025)
   END_RUNG
   RUNG wire#w3
      Contact( "DB8000_PART_STATUS".UNIT_02.FIXTURE_1.PART_A.STATUS.UNIT_01_STATUS.FACE_R_STATION_4_DONE )
      { S7_GenerateENO := "TRUE" } Move(in := 6, out1 => "DB8000_PART_STATUS".UNIT_02.FIXTURE_1.PART_A.STATUS.PART_CELL_STATUS_COLOR, out2 => "DB2401_DBB_DEFINE".PART_STATUS.DBB_1025)
   END_RUNG
   RUNG wire#w3
      Contact( "DB8000_PART_STATUS".UNIT_02.FIXTURE_1.PART_A.STATUS.CELL_STATUS.U01_DONE_IN_TRANSIT )
      { S7_GenerateENO := "TRUE" } Move(in := 7, out1 => "DB8000_PART_STATUS".UNIT_02.FIXTURE_1.PART_A.STATUS.PART_CELL_STATUS_COLOR, out2 => "DB2401_DBB_DEFINE".PART_STATUS.DBB_1025)
   END_RUNG
   RUNG wire#w3
      Contact( "DB8000_PART_STATUS".UNIT_02.FIXTURE_1.PART_A.STATUS.UNIT_02_STATUS.FACE_N_STATION_2_DONE )
      { S7_GenerateENO := "TRUE" } Move(in := 8, out1 => "DB8000_PART_STATUS".UNIT_02.FIXTURE_1.PART_A.STATUS.PART_CELL_STATUS_COLOR, out2 => "DB2401_DBB_DEFINE".PART_STATUS.DBB_1025)
   END_RUNG
   RUNG wire#w3
      Contact( "DB8000_PART_STATUS".UNIT_02.FIXTURE_1.PART_A.STATUS.UNIT_02_STATUS.FACE_N_STATION_3_DONE )
      Move(in := 9, out1 => "DB8000_PART_STATUS".UNIT_02.FIXTURE_1.PART_A.STATUS.PART_CELL_STATUS_COLOR, out2 => "DB2401_DBB_DEFINE".PART_STATUS.DBB_1025)
   END_RUNG
   RUNG wire#w3
      Contact( "DB8000_PART_STATUS".UNIT_02.FIXTURE_1.PART_A.STATUS.UNIT_02_STATUS.FACE_N_STATION_4_DONE )
      Move(in := 10, out1 => "DB8000_PART_STATUS".UNIT_02.FIXTURE_1.PART_A.STATUS.PART_CELL_STATUS_COLOR, out2 => "DB2401_DBB_DEFINE".PART_STATUS.DBB_1025)
   END_RUNG
   RUNG wire#w3
      Contact( "DB8000_PART_STATUS".UNIT_02.FIXTURE_1.PART_A.STATUS.CELL_STATUS.U02_ONE_FACE_DONE_ROTATED )
      Move(in := 11, out1 => "DB8000_PART_STATUS".UNIT_02.FIXTURE_1.PART_A.STATUS.PART_CELL_STATUS_COLOR, out2 => "DB2401_DBB_DEFINE".PART_STATUS.DBB_1025)
   END_RUNG
   RUNG wire#w3
      Contact( "DB8000_PART_STATUS".UNIT_02.FIXTURE_1.PART_A.STATUS.UNIT_02_STATUS.FACE_R_STATION_2_DONE )
      Move(in := 12, out1 => "DB8000_PART_STATUS".UNIT_02.FIXTURE_1.PART_A.STATUS.PART_CELL_STATUS_COLOR, out2 => "DB2401_DBB_DEFINE".PART_STATUS.DBB_1025)
   END_RUNG
   RUNG wire#w3
      Contact( "DB8000_PART_STATUS".UNIT_02.FIXTURE_1.PART_A.STATUS.UNIT_02_STATUS.FACE_R_STATION_3_DONE )
      Move(in := 13, out1 => "DB8000_PART_STATUS".UNIT_02.FIXTURE_1.PART_A.STATUS.PART_CELL_STATUS_COLOR, out2 => "DB2401_DBB_DEFINE".PART_STATUS.DBB_1025)
   END_RUNG
   RUNG wire#w3
      Contact( "DB8000_PART_STATUS".UNIT_02.FIXTURE_1.PART_A.STATUS.UNIT_02_STATUS.FACE_R_STATION_4_DONE )
      Move(in := 14, out1 => "DB8000_PART_STATUS".UNIT_02.FIXTURE_1.PART_A.STATUS.PART_CELL_STATUS_COLOR, out2 => "DB2401_DBB_DEFINE".PART_STATUS.DBB_1025)
   END_RUNG
   RUNG wire#w3
      Contact( "DB8000_PART_STATUS".UNIT_02.FIXTURE_1.PART_A.STATUS.CELL_STATUS.U02_DONE_IN_TRANSIT )
      Move(in := 15, out1 => "DB8000_PART_STATUS".UNIT_02.FIXTURE_1.PART_A.STATUS.PART_CELL_STATUS_COLOR, out2 => "DB2401_DBB_DEFINE".PART_STATUS.DBB_1025)
   END_RUNG
   RUNG wire#w3
      Contact( "DB8000_PART_STATUS".UNIT_02.FIXTURE_1.PART_A.STATUS.CELL_STATUS.COOLING_DONE )
      Move(in := 16, out1 => "DB8000_PART_STATUS".UNIT_02.FIXTURE_1.PART_A.STATUS.PART_CELL_STATUS_COLOR, out2 => "DB2401_DBB_DEFINE".PART_STATUS.DBB_1025)
   END_RUNG
   RUNG wire#w3
      Contact( "DB8000_PART_STATUS".UNIT_02.FIXTURE_1.PART_A.STATUS.CELL_STATUS.INSPECTION_DONE )
      Move(in := 17, out1 => "DB8000_PART_STATUS".UNIT_02.FIXTURE_1.PART_A.STATUS.PART_CELL_STATUS_COLOR, out2 => "DB2401_DBB_DEFINE".PART_STATUS.DBB_1025)
   END_RUNG
   RUNG wire#w3
      Contact( "DB8000_PART_STATUS".UNIT_02.FIXTURE_1.PART_A.STATUS.MASTER_PART )
      Move(in := 99, out1 => "DB8000_PART_STATUS".UNIT_02.FIXTURE_1.PART_A.STATUS.PART_CELL_STATUS_COLOR, out2 => "DB2401_DBB_DEFINE".PART_STATUS.DBB_1025)
   END_RUNG
   // the same network as SCL:
   // ENO of a box is taken as its EN; it also drops when the box reports an error
   IF "M_ONE" AND NOT "DB8000_PART_STATUS".UNIT_02.FIXTURE_1.PART_A.STATUS.PRESENT THEN
       "DB2401_DBB_DEFINE".PART_STATUS.DBB_1024 := 0;
       "DB2401_DBB_DEFINE".PART_STATUS.DBB_1025 := 0;
       "DB8000_PART_STATUS".UNIT_02.FIXTURE_1.PART_A.STATUS.PART_MAIN_STATUS_COLOR := 0;
       "DB8000_PART_STATUS".UNIT_02.FIXTURE_1.PART_A.STATUS.PART_CELL_STATUS_COLOR := 0;
   END_IF;
   #_w1 := "M_ONE" AND "DB8000_PART_STATUS".UNIT_02.FIXTURE_1.PART_A.STATUS.PRESENT;
   IF #_w1 AND NOT "DB8000_PART_STATUS".UNIT_02.FIXTURE_1.PART_A.STATUS.PART_REJECTED AND NOT "DB8000_PART_STATUS".UNIT_02.FIXTURE_1.PART_A.STATUS.QUALITY_PART THEN
       "DB8000_PART_STATUS".UNIT_02.FIXTURE_1.PART_A.STATUS.PART_MAIN_STATUS_COLOR := 1;
       "DB2401_DBB_DEFINE".PART_STATUS.DBB_1024 := 1;
   END_IF;
   IF #_w1 AND "DB8000_PART_STATUS".UNIT_02.FIXTURE_1.PART_A.STATUS.PART_REJECTED THEN
       "DB8000_PART_STATUS".UNIT_02.FIXTURE_1.PART_A.STATUS.PART_MAIN_STATUS_COLOR := 2;
       "DB2401_DBB_DEFINE".PART_STATUS.DBB_1024 := 2;
   END_IF;
   IF #_w1 AND "DB8000_PART_STATUS".UNIT_02.FIXTURE_1.PART_A.STATUS.QUALITY_PART AND NOT "DB8000_PART_STATUS".UNIT_02.FIXTURE_1.PART_A.STATUS.PART_REJECTED THEN
       "DB8000_PART_STATUS".UNIT_02.FIXTURE_1.PART_A.STATUS.PART_MAIN_STATUS_COLOR := 3;
       "DB2401_DBB_DEFINE".PART_STATUS.DBB_1024 := 3;
   END_IF;
   #_w2 := "M_ONE" AND "DB8000_PART_STATUS".UNIT_02.FIXTURE_1.PART_A.STATUS.PRESENT;
   IF #_w2 AND "DB8000_PART_STATUS".UNIT_02.FIXTURE_1.PART_A.STATUS.CELL_STATUS.NEW_IN_TRANSIT THEN
       "DB8000_PART_STATUS".UNIT_02.FIXTURE_1.PART_A.STATUS.PART_CELL_STATUS_COLOR := 1;
       "DB2401_DBB_DEFINE".PART_STATUS.DBB_1025 := 1;
   END_IF;
   IF #_w2 AND "DB8000_PART_STATUS".UNIT_02.FIXTURE_1.PART_A.STATUS.UNIT_01_STATUS.FACE_N_STATION_3_DONE THEN
       "DB8000_PART_STATUS".UNIT_02.FIXTURE_1.PART_A.STATUS.PART_CELL_STATUS_COLOR := 2;
       "DB2401_DBB_DEFINE".PART_STATUS.DBB_1025 := 2;
   END_IF;
   IF #_w2 AND "DB8000_PART_STATUS".UNIT_02.FIXTURE_1.PART_A.STATUS.UNIT_01_STATUS.FACE_N_STATION_4_DONE THEN
       "DB8000_PART_STATUS".UNIT_02.FIXTURE_1.PART_A.STATUS.PART_CELL_STATUS_COLOR := 3;
       "DB2401_DBB_DEFINE".PART_STATUS.DBB_1025 := 3;
   END_IF;
   IF #_w2 AND "DB8000_PART_STATUS".UNIT_02.FIXTURE_1.PART_A.STATUS.CELL_STATUS.U01_ONE_FACE_DONE_ROTATED THEN
       "DB8000_PART_STATUS".UNIT_02.FIXTURE_1.PART_A.STATUS.PART_CELL_STATUS_COLOR := 4;
       "DB2401_DBB_DEFINE".PART_STATUS.DBB_1025 := 4;
   END_IF;
   IF #_w2 AND "DB8000_PART_STATUS".UNIT_02.FIXTURE_1.PART_A.STATUS.UNIT_01_STATUS.FACE_R_STATION_3_DONE THEN
       "DB8000_PART_STATUS".UNIT_02.FIXTURE_1.PART_A.STATUS.PART_CELL_STATUS_COLOR := 5;
       "DB2401_DBB_DEFINE".PART_STATUS.DBB_1025 := 5;
   END_IF;
   IF #_w2 AND "DB8000_PART_STATUS".UNIT_02.FIXTURE_1.PART_A.STATUS.UNIT_01_STATUS.FACE_R_STATION_4_DONE THEN
       "DB8000_PART_STATUS".UNIT_02.FIXTURE_1.PART_A.STATUS.PART_CELL_STATUS_COLOR := 6;
       "DB2401_DBB_DEFINE".PART_STATUS.DBB_1025 := 6;
   END_IF;
   IF #_w2 AND "DB8000_PART_STATUS".UNIT_02.FIXTURE_1.PART_A.STATUS.CELL_STATUS.U01_DONE_IN_TRANSIT THEN
       "DB8000_PART_STATUS".UNIT_02.FIXTURE_1.PART_A.STATUS.PART_CELL_STATUS_COLOR := 7;
       "DB2401_DBB_DEFINE".PART_STATUS.DBB_1025 := 7;
   END_IF;
   IF #_w2 AND "DB8000_PART_STATUS".UNIT_02.FIXTURE_1.PART_A.STATUS.UNIT_02_STATUS.FACE_N_STATION_2_DONE THEN
       "DB8000_PART_STATUS".UNIT_02.FIXTURE_1.PART_A.STATUS.PART_CELL_STATUS_COLOR := 8;
       "DB2401_DBB_DEFINE".PART_STATUS.DBB_1025 := 8;
   END_IF;
   IF #_w2 AND "DB8000_PART_STATUS".UNIT_02.FIXTURE_1.PART_A.STATUS.UNIT_02_STATUS.FACE_N_STATION_3_DONE THEN
       "DB8000_PART_STATUS".UNIT_02.FIXTURE_1.PART_A.STATUS.PART_CELL_STATUS_COLOR := 9;
       "DB2401_DBB_DEFINE".PART_STATUS.DBB_1025 := 9;
   END_IF;
   IF #_w2 AND "DB8000_PART_STATUS".UNIT_02.FIXTURE_1.PART_A.STATUS.UNIT_02_STATUS.FACE_N_STATION_4_DONE THEN
       "DB8000_PART_STATUS".UNIT_02.FIXTURE_1.PART_A.STATUS.PART_CELL_STATUS_COLOR := 10;
       "DB2401_DBB_DEFINE".PART_STATUS.DBB_1025 := 10;
   END_IF;
   IF #_w2 AND "DB8000_PART_STATUS".UNIT_02.FIXTURE_1.PART_A.STATUS.CELL_STATUS.U02_ONE_FACE_DONE_ROTATED THEN
       "DB8000_PART_STATUS".UNIT_02.FIXTURE_1.PART_A.STATUS.PART_CELL_STATUS_COLOR := 11;
       "DB2401_DBB_DEFINE".PART_STATUS.DBB_1025 := 11;
   END_IF;
   IF #_w2 AND "DB8000_PART_STATUS".UNIT_02.FIXTURE_1.PART_A.STATUS.UNIT_02_STATUS.FACE_R_STATION_2_DONE THEN
       "DB8000_PART_STATUS".UNIT_02.FIXTURE_1.PART_A.STATUS.PART_CELL_STATUS_COLOR := 12;
       "DB2401_DBB_DEFINE".PART_STATUS.DBB_1025 := 12;
   END_IF;
   IF #_w2 AND "DB8000_PART_STATUS".UNIT_02.FIXTURE_1.PART_A.STATUS.UNIT_02_STATUS.FACE_R_STATION_3_DONE THEN
       "DB8000_PART_STATUS".UNIT_02.FIXTURE_1.PART_A.STATUS.PART_CELL_STATUS_COLOR := 13;
       "DB2401_DBB_DEFINE".PART_STATUS.DBB_1025 := 13;
   END_IF;
   IF #_w2 AND "DB8000_PART_STATUS".UNIT_02.FIXTURE_1.PART_A.STATUS.UNIT_02_STATUS.FACE_R_STATION_4_DONE THEN
       "DB8000_PART_STATUS".UNIT_02.FIXTURE_1.PART_A.STATUS.PART_CELL_STATUS_COLOR := 14;
       "DB2401_DBB_DEFINE".PART_STATUS.DBB_1025 := 14;
   END_IF;
   IF #_w2 AND "DB8000_PART_STATUS".UNIT_02.FIXTURE_1.PART_A.STATUS.CELL_STATUS.U02_DONE_IN_TRANSIT THEN
       "DB8000_PART_STATUS".UNIT_02.FIXTURE_1.PART_A.STATUS.PART_CELL_STATUS_COLOR := 15;
       "DB2401_DBB_DEFINE".PART_STATUS.DBB_1025 := 15;
   END_IF;
   IF #_w2 AND "DB8000_PART_STATUS".UNIT_02.FIXTURE_1.PART_A.STATUS.CELL_STATUS.COOLING_DONE THEN
       "DB8000_PART_STATUS".UNIT_02.FIXTURE_1.PART_A.STATUS.PART_CELL_STATUS_COLOR := 16;
       "DB2401_DBB_DEFINE".PART_STATUS.DBB_1025 := 16;
   END_IF;
   IF #_w2 AND "DB8000_PART_STATUS".UNIT_02.FIXTURE_1.PART_A.STATUS.CELL_STATUS.INSPECTION_DONE THEN
       "DB8000_PART_STATUS".UNIT_02.FIXTURE_1.PART_A.STATUS.PART_CELL_STATUS_COLOR := 17;
       "DB2401_DBB_DEFINE".PART_STATUS.DBB_1025 := 17;
   END_IF;
   IF #_w2 AND "DB8000_PART_STATUS".UNIT_02.FIXTURE_1.PART_A.STATUS.MASTER_PART THEN
       "DB8000_PART_STATUS".UNIT_02.FIXTURE_1.PART_A.STATUS.PART_CELL_STATUS_COLOR := 99;
       "DB2401_DBB_DEFINE".PART_STATUS.DBB_1025 := 99;
   END_IF;
END_REGION

REGION Network 20: PART A FIXTURE 2 COLOR STATUS
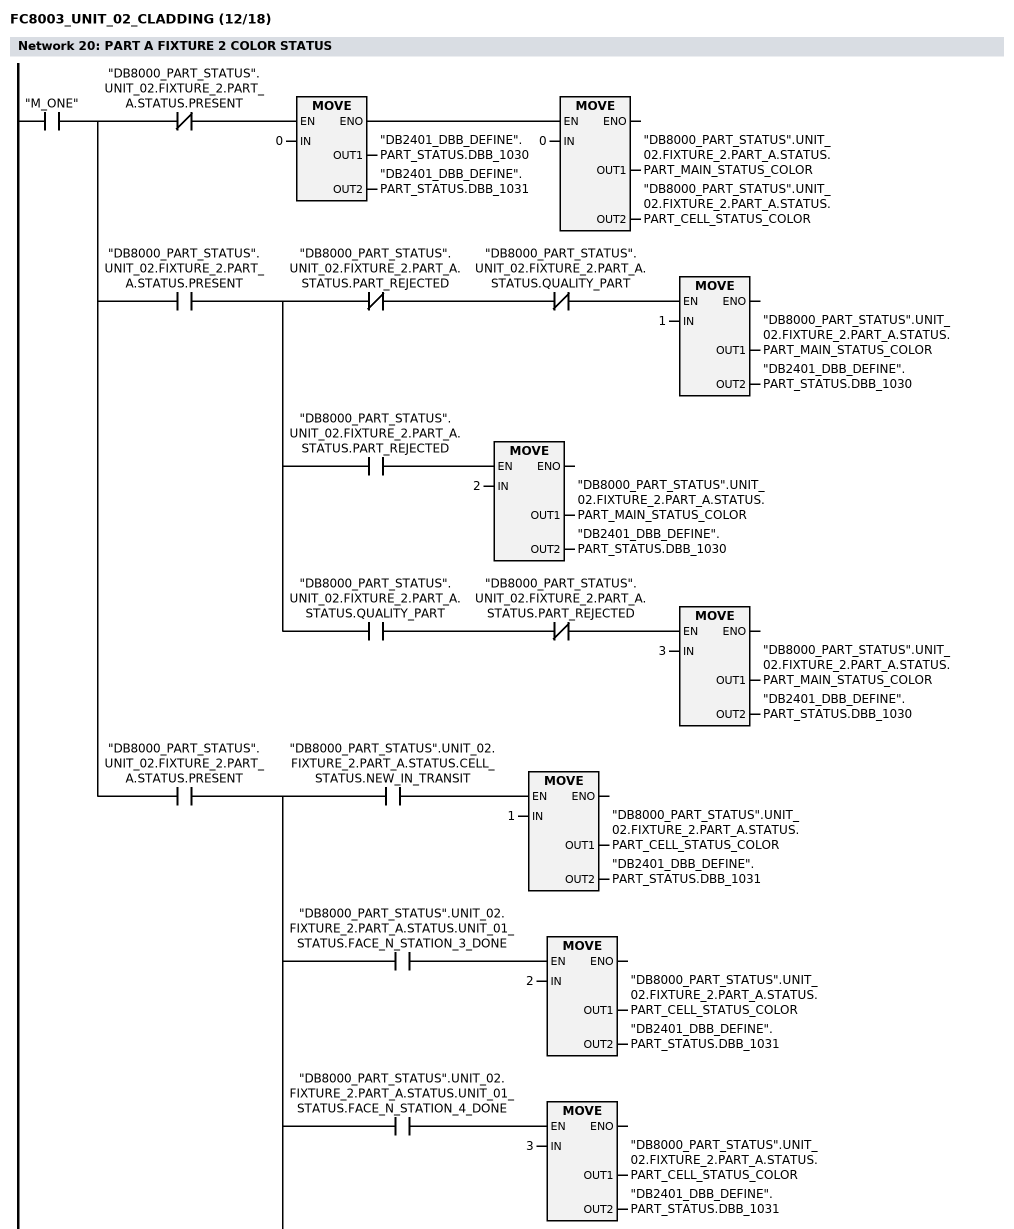
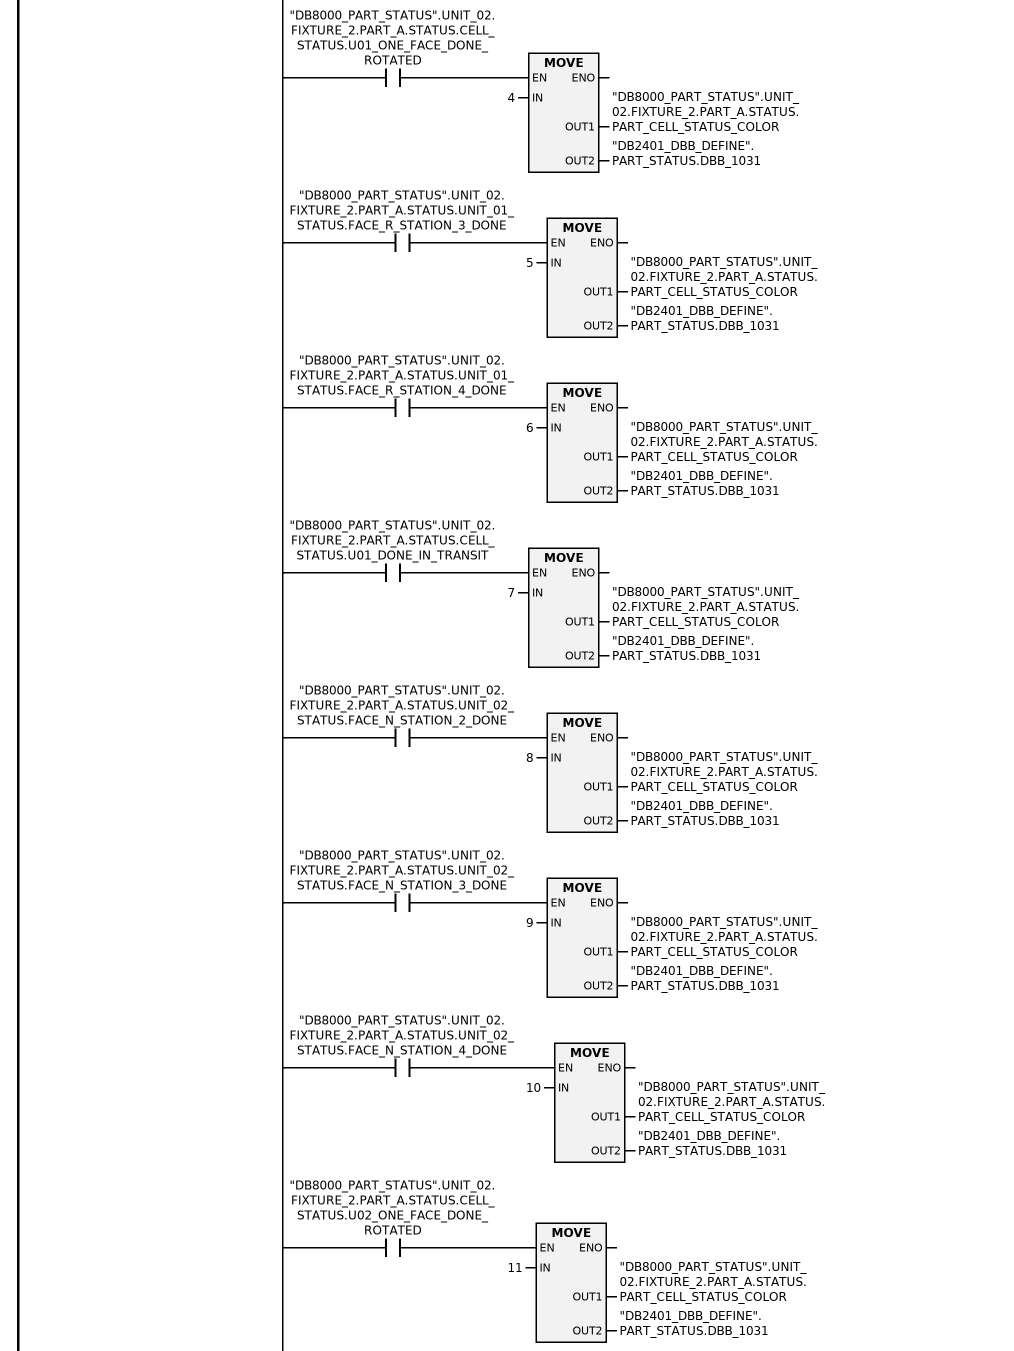
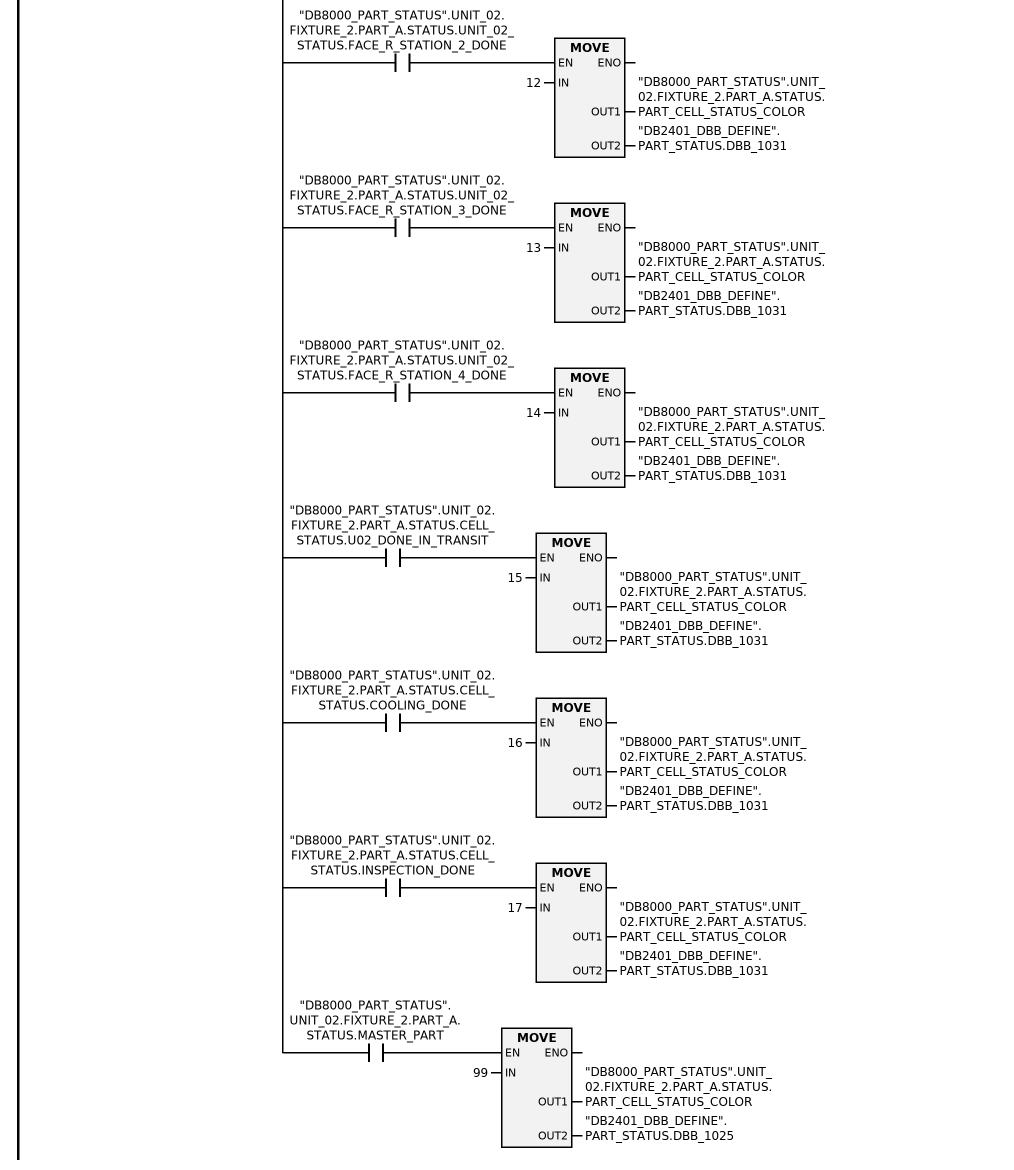
   RUNG wire#powerrail
      Contact( "M_ONE" )
      wire#w1
      I_Contact( "DB8000_PART_STATUS".UNIT_02.FIXTURE_2.PART_A.STATUS.PRESENT )
      { S7_GenerateENO := "TRUE" } Move(in := 0, out1 => "DB2401_DBB_DEFINE".PART_STATUS.DBB_1030, out2 => "DB2401_DBB_DEFINE".PART_STATUS.DBB_1031)
      { S7_GenerateENO := "TRUE" } Move(in := 0, out1 => "DB8000_PART_STATUS".UNIT_02.FIXTURE_2.PART_A.STATUS.PART_MAIN_STATUS_COLOR, out2 => "DB8000_PART_STATUS".UNIT_02.FIXTURE_2.PART_A.STATUS.PART_CELL_STATUS_COLOR)
   END_RUNG
   RUNG wire#w1
      Contact( "DB8000_PART_STATUS".UNIT_02.FIXTURE_2.PART_A.STATUS.PRESENT )
      wire#w2
      I_Contact( "DB8000_PART_STATUS".UNIT_02.FIXTURE_2.PART_A.STATUS.PART_REJECTED )
      I_Contact( "DB8000_PART_STATUS".UNIT_02.FIXTURE_2.PART_A.STATUS.QUALITY_PART )
      { S7_GenerateENO := "TRUE" } Move(in := 1, out1 => "DB8000_PART_STATUS".UNIT_02.FIXTURE_2.PART_A.STATUS.PART_MAIN_STATUS_COLOR, out2 => "DB2401_DBB_DEFINE".PART_STATUS.DBB_1030)
   END_RUNG
   RUNG wire#w2
      Contact( "DB8000_PART_STATUS".UNIT_02.FIXTURE_2.PART_A.STATUS.PART_REJECTED )
      { S7_GenerateENO := "TRUE" } Move(in := 2, out1 => "DB8000_PART_STATUS".UNIT_02.FIXTURE_2.PART_A.STATUS.PART_MAIN_STATUS_COLOR, out2 => "DB2401_DBB_DEFINE".PART_STATUS.DBB_1030)
   END_RUNG
   RUNG wire#w2
      Contact( "DB8000_PART_STATUS".UNIT_02.FIXTURE_2.PART_A.STATUS.QUALITY_PART )
      I_Contact( "DB8000_PART_STATUS".UNIT_02.FIXTURE_2.PART_A.STATUS.PART_REJECTED )
      { S7_GenerateENO := "TRUE" } Move(in := 3, out1 => "DB8000_PART_STATUS".UNIT_02.FIXTURE_2.PART_A.STATUS.PART_MAIN_STATUS_COLOR, out2 => "DB2401_DBB_DEFINE".PART_STATUS.DBB_1030)
   END_RUNG
   RUNG wire#w1
      Contact( "DB8000_PART_STATUS".UNIT_02.FIXTURE_2.PART_A.STATUS.PRESENT )
      wire#w3
      Contact( "DB8000_PART_STATUS".UNIT_02.FIXTURE_2.PART_A.STATUS.CELL_STATUS.NEW_IN_TRANSIT )
      { S7_GenerateENO := "TRUE" } Move(in := 1, out1 => "DB8000_PART_STATUS".UNIT_02.FIXTURE_2.PART_A.STATUS.PART_CELL_STATUS_COLOR, out2 => "DB2401_DBB_DEFINE".PART_STATUS.DBB_1031)
   END_RUNG
   RUNG wire#w3
      Contact( "DB8000_PART_STATUS".UNIT_02.FIXTURE_2.PART_A.STATUS.UNIT_01_STATUS.FACE_N_STATION_3_DONE )
      { S7_GenerateENO := "TRUE" } Move(in := 2, out1 => "DB8000_PART_STATUS".UNIT_02.FIXTURE_2.PART_A.STATUS.PART_CELL_STATUS_COLOR, out2 => "DB2401_DBB_DEFINE".PART_STATUS.DBB_1031)
   END_RUNG
   RUNG wire#w3
      Contact( "DB8000_PART_STATUS".UNIT_02.FIXTURE_2.PART_A.STATUS.UNIT_01_STATUS.FACE_N_STATION_4_DONE )
      { S7_GenerateENO := "TRUE" } Move(in := 3, out1 => "DB8000_PART_STATUS".UNIT_02.FIXTURE_2.PART_A.STATUS.PART_CELL_STATUS_COLOR, out2 => "DB2401_DBB_DEFINE".PART_STATUS.DBB_1031)
   END_RUNG
   RUNG wire#w3
      Contact( "DB8000_PART_STATUS".UNIT_02.FIXTURE_2.PART_A.STATUS.CELL_STATUS.U01_ONE_FACE_DONE_ROTATED )
      { S7_GenerateENO := "TRUE" } Move(in := 4, out1 => "DB8000_PART_STATUS".UNIT_02.FIXTURE_2.PART_A.STATUS.PART_CELL_STATUS_COLOR, out2 => "DB2401_DBB_DEFINE".PART_STATUS.DBB_1031)
   END_RUNG
   RUNG wire#w3
      Contact( "DB8000_PART_STATUS".UNIT_02.FIXTURE_2.PART_A.STATUS.UNIT_01_STATUS.FACE_R_STATION_3_DONE )
      { S7_GenerateENO := "TRUE" } Move(in := 5, out1 => "DB8000_PART_STATUS".UNIT_02.FIXTURE_2.PART_A.STATUS.PART_CELL_STATUS_COLOR, out2 => "DB2401_DBB_DEFINE".PART_STATUS.DBB_1031)
   END_RUNG
   RUNG wire#w3
      Contact( "DB8000_PART_STATUS".UNIT_02.FIXTURE_2.PART_A.STATUS.UNIT_01_STATUS.FACE_R_STATION_4_DONE )
      { S7_GenerateENO := "TRUE" } Move(in := 6, out1 => "DB8000_PART_STATUS".UNIT_02.FIXTURE_2.PART_A.STATUS.PART_CELL_STATUS_COLOR, out2 => "DB2401_DBB_DEFINE".PART_STATUS.DBB_1031)
   END_RUNG
   RUNG wire#w3
      Contact( "DB8000_PART_STATUS".UNIT_02.FIXTURE_2.PART_A.STATUS.CELL_STATUS.U01_DONE_IN_TRANSIT )
      { S7_GenerateENO := "TRUE" } Move(in := 7, out1 => "DB8000_PART_STATUS".UNIT_02.FIXTURE_2.PART_A.STATUS.PART_CELL_STATUS_COLOR, out2 => "DB2401_DBB_DEFINE".PART_STATUS.DBB_1031)
   END_RUNG
   RUNG wire#w3
      Contact( "DB8000_PART_STATUS".UNIT_02.FIXTURE_2.PART_A.STATUS.UNIT_02_STATUS.FACE_N_STATION_2_DONE )
      { S7_GenerateENO := "TRUE" } Move(in := 8, out1 => "DB8000_PART_STATUS".UNIT_02.FIXTURE_2.PART_A.STATUS.PART_CELL_STATUS_COLOR, out2 => "DB2401_DBB_DEFINE".PART_STATUS.DBB_1031)
   END_RUNG
   RUNG wire#w3
      Contact( "DB8000_PART_STATUS".UNIT_02.FIXTURE_2.PART_A.STATUS.UNIT_02_STATUS.FACE_N_STATION_3_DONE )
      Move(in := 9, out1 => "DB8000_PART_STATUS".UNIT_02.FIXTURE_2.PART_A.STATUS.PART_CELL_STATUS_COLOR, out2 => "DB2401_DBB_DEFINE".PART_STATUS.DBB_1031)
   END_RUNG
   RUNG wire#w3
      Contact( "DB8000_PART_STATUS".UNIT_02.FIXTURE_2.PART_A.STATUS.UNIT_02_STATUS.FACE_N_STATION_4_DONE )
      Move(in := 10, out1 => "DB8000_PART_STATUS".UNIT_02.FIXTURE_2.PART_A.STATUS.PART_CELL_STATUS_COLOR, out2 => "DB2401_DBB_DEFINE".PART_STATUS.DBB_1031)
   END_RUNG
   RUNG wire#w3
      Contact( "DB8000_PART_STATUS".UNIT_02.FIXTURE_2.PART_A.STATUS.CELL_STATUS.U02_ONE_FACE_DONE_ROTATED )
      Move(in := 11, out1 => "DB8000_PART_STATUS".UNIT_02.FIXTURE_2.PART_A.STATUS.PART_CELL_STATUS_COLOR, out2 => "DB2401_DBB_DEFINE".PART_STATUS.DBB_1031)
   END_RUNG
   RUNG wire#w3
      Contact( "DB8000_PART_STATUS".UNIT_02.FIXTURE_2.PART_A.STATUS.UNIT_02_STATUS.FACE_R_STATION_2_DONE )
      Move(in := 12, out1 => "DB8000_PART_STATUS".UNIT_02.FIXTURE_2.PART_A.STATUS.PART_CELL_STATUS_COLOR, out2 => "DB2401_DBB_DEFINE".PART_STATUS.DBB_1031)
   END_RUNG
   RUNG wire#w3
      Contact( "DB8000_PART_STATUS".UNIT_02.FIXTURE_2.PART_A.STATUS.UNIT_02_STATUS.FACE_R_STATION_3_DONE )
      Move(in := 13, out1 => "DB8000_PART_STATUS".UNIT_02.FIXTURE_2.PART_A.STATUS.PART_CELL_STATUS_COLOR, out2 => "DB2401_DBB_DEFINE".PART_STATUS.DBB_1031)
   END_RUNG
   RUNG wire#w3
      Contact( "DB8000_PART_STATUS".UNIT_02.FIXTURE_2.PART_A.STATUS.UNIT_02_STATUS.FACE_R_STATION_4_DONE )
      Move(in := 14, out1 => "DB8000_PART_STATUS".UNIT_02.FIXTURE_2.PART_A.STATUS.PART_CELL_STATUS_COLOR, out2 => "DB2401_DBB_DEFINE".PART_STATUS.DBB_1031)
   END_RUNG
   RUNG wire#w3
      Contact( "DB8000_PART_STATUS".UNIT_02.FIXTURE_2.PART_A.STATUS.CELL_STATUS.U02_DONE_IN_TRANSIT )
      Move(in := 15, out1 => "DB8000_PART_STATUS".UNIT_02.FIXTURE_2.PART_A.STATUS.PART_CELL_STATUS_COLOR, out2 => "DB2401_DBB_DEFINE".PART_STATUS.DBB_1031)
   END_RUNG
   RUNG wire#w3
      Contact( "DB8000_PART_STATUS".UNIT_02.FIXTURE_2.PART_A.STATUS.CELL_STATUS.COOLING_DONE )
      Move(in := 16, out1 => "DB8000_PART_STATUS".UNIT_02.FIXTURE_2.PART_A.STATUS.PART_CELL_STATUS_COLOR, out2 => "DB2401_DBB_DEFINE".PART_STATUS.DBB_1031)
   END_RUNG
   RUNG wire#w3
      Contact( "DB8000_PART_STATUS".UNIT_02.FIXTURE_2.PART_A.STATUS.CELL_STATUS.INSPECTION_DONE )
      Move(in := 17, out1 => "DB8000_PART_STATUS".UNIT_02.FIXTURE_2.PART_A.STATUS.PART_CELL_STATUS_COLOR, out2 => "DB2401_DBB_DEFINE".PART_STATUS.DBB_1031)
   END_RUNG
   RUNG wire#w3
      Contact( "DB8000_PART_STATUS".UNIT_02.FIXTURE_2.PART_A.STATUS.MASTER_PART )
      Move(in := 99, out1 => "DB8000_PART_STATUS".UNIT_02.FIXTURE_2.PART_A.STATUS.PART_CELL_STATUS_COLOR, out2 => "DB2401_DBB_DEFINE".PART_STATUS.DBB_1025)
   END_RUNG
   // the same network as SCL:
   // ENO of a box is taken as its EN; it also drops when the box reports an error
   IF "M_ONE" AND NOT "DB8000_PART_STATUS".UNIT_02.FIXTURE_2.PART_A.STATUS.PRESENT THEN
       "DB2401_DBB_DEFINE".PART_STATUS.DBB_1030 := 0;
       "DB2401_DBB_DEFINE".PART_STATUS.DBB_1031 := 0;
       "DB8000_PART_STATUS".UNIT_02.FIXTURE_2.PART_A.STATUS.PART_MAIN_STATUS_COLOR := 0;
       "DB8000_PART_STATUS".UNIT_02.FIXTURE_2.PART_A.STATUS.PART_CELL_STATUS_COLOR := 0;
   END_IF;
   #_w1 := "M_ONE" AND "DB8000_PART_STATUS".UNIT_02.FIXTURE_2.PART_A.STATUS.PRESENT;
   IF #_w1 AND NOT "DB8000_PART_STATUS".UNIT_02.FIXTURE_2.PART_A.STATUS.PART_REJECTED AND NOT "DB8000_PART_STATUS".UNIT_02.FIXTURE_2.PART_A.STATUS.QUALITY_PART THEN
       "DB8000_PART_STATUS".UNIT_02.FIXTURE_2.PART_A.STATUS.PART_MAIN_STATUS_COLOR := 1;
       "DB2401_DBB_DEFINE".PART_STATUS.DBB_1030 := 1;
   END_IF;
   IF #_w1 AND "DB8000_PART_STATUS".UNIT_02.FIXTURE_2.PART_A.STATUS.PART_REJECTED THEN
       "DB8000_PART_STATUS".UNIT_02.FIXTURE_2.PART_A.STATUS.PART_MAIN_STATUS_COLOR := 2;
       "DB2401_DBB_DEFINE".PART_STATUS.DBB_1030 := 2;
   END_IF;
   IF #_w1 AND "DB8000_PART_STATUS".UNIT_02.FIXTURE_2.PART_A.STATUS.QUALITY_PART AND NOT "DB8000_PART_STATUS".UNIT_02.FIXTURE_2.PART_A.STATUS.PART_REJECTED THEN
       "DB8000_PART_STATUS".UNIT_02.FIXTURE_2.PART_A.STATUS.PART_MAIN_STATUS_COLOR := 3;
       "DB2401_DBB_DEFINE".PART_STATUS.DBB_1030 := 3;
   END_IF;
   #_w2 := "M_ONE" AND "DB8000_PART_STATUS".UNIT_02.FIXTURE_2.PART_A.STATUS.PRESENT;
   IF #_w2 AND "DB8000_PART_STATUS".UNIT_02.FIXTURE_2.PART_A.STATUS.CELL_STATUS.NEW_IN_TRANSIT THEN
       "DB8000_PART_STATUS".UNIT_02.FIXTURE_2.PART_A.STATUS.PART_CELL_STATUS_COLOR := 1;
       "DB2401_DBB_DEFINE".PART_STATUS.DBB_1031 := 1;
   END_IF;
   IF #_w2 AND "DB8000_PART_STATUS".UNIT_02.FIXTURE_2.PART_A.STATUS.UNIT_01_STATUS.FACE_N_STATION_3_DONE THEN
       "DB8000_PART_STATUS".UNIT_02.FIXTURE_2.PART_A.STATUS.PART_CELL_STATUS_COLOR := 2;
       "DB2401_DBB_DEFINE".PART_STATUS.DBB_1031 := 2;
   END_IF;
   IF #_w2 AND "DB8000_PART_STATUS".UNIT_02.FIXTURE_2.PART_A.STATUS.UNIT_01_STATUS.FACE_N_STATION_4_DONE THEN
       "DB8000_PART_STATUS".UNIT_02.FIXTURE_2.PART_A.STATUS.PART_CELL_STATUS_COLOR := 3;
       "DB2401_DBB_DEFINE".PART_STATUS.DBB_1031 := 3;
   END_IF;
   IF #_w2 AND "DB8000_PART_STATUS".UNIT_02.FIXTURE_2.PART_A.STATUS.CELL_STATUS.U01_ONE_FACE_DONE_ROTATED THEN
       "DB8000_PART_STATUS".UNIT_02.FIXTURE_2.PART_A.STATUS.PART_CELL_STATUS_COLOR := 4;
       "DB2401_DBB_DEFINE".PART_STATUS.DBB_1031 := 4;
   END_IF;
   IF #_w2 AND "DB8000_PART_STATUS".UNIT_02.FIXTURE_2.PART_A.STATUS.UNIT_01_STATUS.FACE_R_STATION_3_DONE THEN
       "DB8000_PART_STATUS".UNIT_02.FIXTURE_2.PART_A.STATUS.PART_CELL_STATUS_COLOR := 5;
       "DB2401_DBB_DEFINE".PART_STATUS.DBB_1031 := 5;
   END_IF;
   IF #_w2 AND "DB8000_PART_STATUS".UNIT_02.FIXTURE_2.PART_A.STATUS.UNIT_01_STATUS.FACE_R_STATION_4_DONE THEN
       "DB8000_PART_STATUS".UNIT_02.FIXTURE_2.PART_A.STATUS.PART_CELL_STATUS_COLOR := 6;
       "DB2401_DBB_DEFINE".PART_STATUS.DBB_1031 := 6;
   END_IF;
   IF #_w2 AND "DB8000_PART_STATUS".UNIT_02.FIXTURE_2.PART_A.STATUS.CELL_STATUS.U01_DONE_IN_TRANSIT THEN
       "DB8000_PART_STATUS".UNIT_02.FIXTURE_2.PART_A.STATUS.PART_CELL_STATUS_COLOR := 7;
       "DB2401_DBB_DEFINE".PART_STATUS.DBB_1031 := 7;
   END_IF;
   IF #_w2 AND "DB8000_PART_STATUS".UNIT_02.FIXTURE_2.PART_A.STATUS.UNIT_02_STATUS.FACE_N_STATION_2_DONE THEN
       "DB8000_PART_STATUS".UNIT_02.FIXTURE_2.PART_A.STATUS.PART_CELL_STATUS_COLOR := 8;
       "DB2401_DBB_DEFINE".PART_STATUS.DBB_1031 := 8;
   END_IF;
   IF #_w2 AND "DB8000_PART_STATUS".UNIT_02.FIXTURE_2.PART_A.STATUS.UNIT_02_STATUS.FACE_N_STATION_3_DONE THEN
       "DB8000_PART_STATUS".UNIT_02.FIXTURE_2.PART_A.STATUS.PART_CELL_STATUS_COLOR := 9;
       "DB2401_DBB_DEFINE".PART_STATUS.DBB_1031 := 9;
   END_IF;
   IF #_w2 AND "DB8000_PART_STATUS".UNIT_02.FIXTURE_2.PART_A.STATUS.UNIT_02_STATUS.FACE_N_STATION_4_DONE THEN
       "DB8000_PART_STATUS".UNIT_02.FIXTURE_2.PART_A.STATUS.PART_CELL_STATUS_COLOR := 10;
       "DB2401_DBB_DEFINE".PART_STATUS.DBB_1031 := 10;
   END_IF;
   IF #_w2 AND "DB8000_PART_STATUS".UNIT_02.FIXTURE_2.PART_A.STATUS.CELL_STATUS.U02_ONE_FACE_DONE_ROTATED THEN
       "DB8000_PART_STATUS".UNIT_02.FIXTURE_2.PART_A.STATUS.PART_CELL_STATUS_COLOR := 11;
       "DB2401_DBB_DEFINE".PART_STATUS.DBB_1031 := 11;
   END_IF;
   IF #_w2 AND "DB8000_PART_STATUS".UNIT_02.FIXTURE_2.PART_A.STATUS.UNIT_02_STATUS.FACE_R_STATION_2_DONE THEN
       "DB8000_PART_STATUS".UNIT_02.FIXTURE_2.PART_A.STATUS.PART_CELL_STATUS_COLOR := 12;
       "DB2401_DBB_DEFINE".PART_STATUS.DBB_1031 := 12;
   END_IF;
   IF #_w2 AND "DB8000_PART_STATUS".UNIT_02.FIXTURE_2.PART_A.STATUS.UNIT_02_STATUS.FACE_R_STATION_3_DONE THEN
       "DB8000_PART_STATUS".UNIT_02.FIXTURE_2.PART_A.STATUS.PART_CELL_STATUS_COLOR := 13;
       "DB2401_DBB_DEFINE".PART_STATUS.DBB_1031 := 13;
   END_IF;
   IF #_w2 AND "DB8000_PART_STATUS".UNIT_02.FIXTURE_2.PART_A.STATUS.UNIT_02_STATUS.FACE_R_STATION_4_DONE THEN
       "DB8000_PART_STATUS".UNIT_02.FIXTURE_2.PART_A.STATUS.PART_CELL_STATUS_COLOR := 14;
       "DB2401_DBB_DEFINE".PART_STATUS.DBB_1031 := 14;
   END_IF;
   IF #_w2 AND "DB8000_PART_STATUS".UNIT_02.FIXTURE_2.PART_A.STATUS.CELL_STATUS.U02_DONE_IN_TRANSIT THEN
       "DB8000_PART_STATUS".UNIT_02.FIXTURE_2.PART_A.STATUS.PART_CELL_STATUS_COLOR := 15;
       "DB2401_DBB_DEFINE".PART_STATUS.DBB_1031 := 15;
   END_IF;
   IF #_w2 AND "DB8000_PART_STATUS".UNIT_02.FIXTURE_2.PART_A.STATUS.CELL_STATUS.COOLING_DONE THEN
       "DB8000_PART_STATUS".UNIT_02.FIXTURE_2.PART_A.STATUS.PART_CELL_STATUS_COLOR := 16;
       "DB2401_DBB_DEFINE".PART_STATUS.DBB_1031 := 16;
   END_IF;
   IF #_w2 AND "DB8000_PART_STATUS".UNIT_02.FIXTURE_2.PART_A.STATUS.CELL_STATUS.INSPECTION_DONE THEN
       "DB8000_PART_STATUS".UNIT_02.FIXTURE_2.PART_A.STATUS.PART_CELL_STATUS_COLOR := 17;
       "DB2401_DBB_DEFINE".PART_STATUS.DBB_1031 := 17;
   END_IF;
   IF #_w2 AND "DB8000_PART_STATUS".UNIT_02.FIXTURE_2.PART_A.STATUS.MASTER_PART THEN
       "DB8000_PART_STATUS".UNIT_02.FIXTURE_2.PART_A.STATUS.PART_CELL_STATUS_COLOR := 99;
       "DB2401_DBB_DEFINE".PART_STATUS.DBB_1025 := 99;
   END_IF;
END_REGION

REGION Network 21: PART A FIXTURE 3 COLOR STATUS
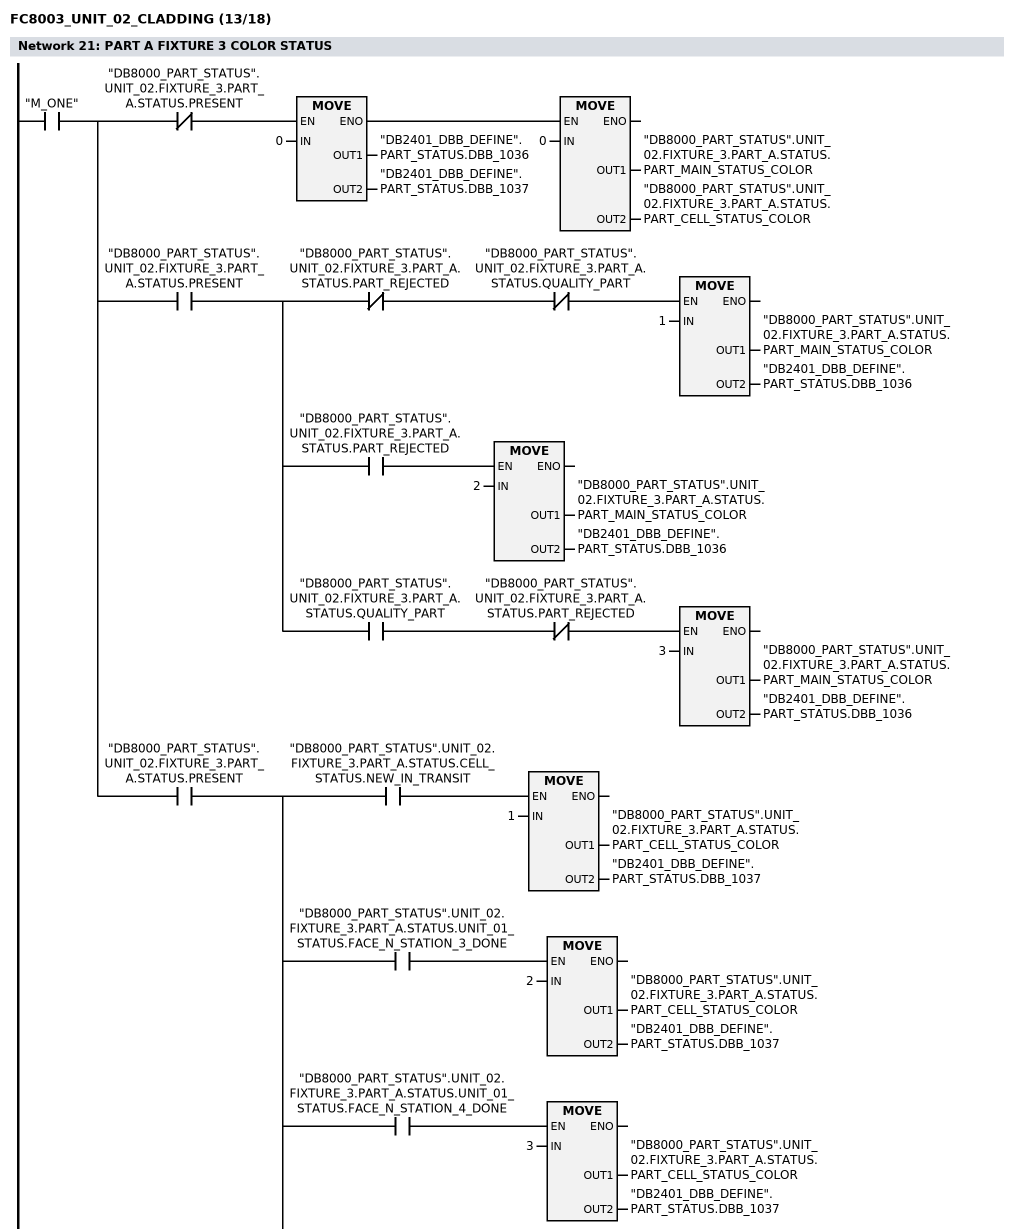
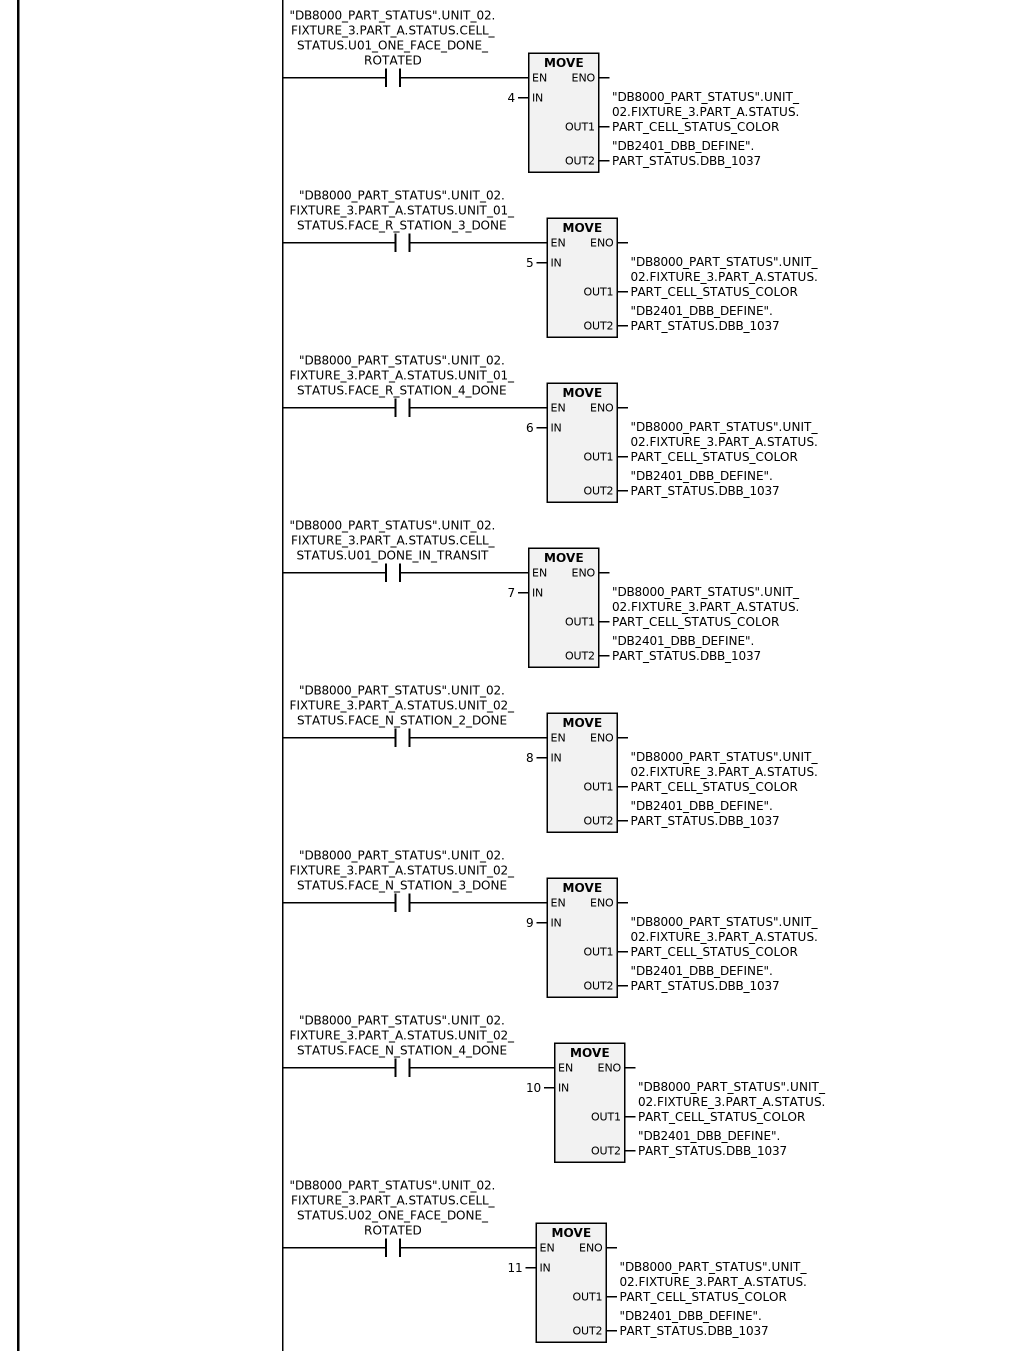
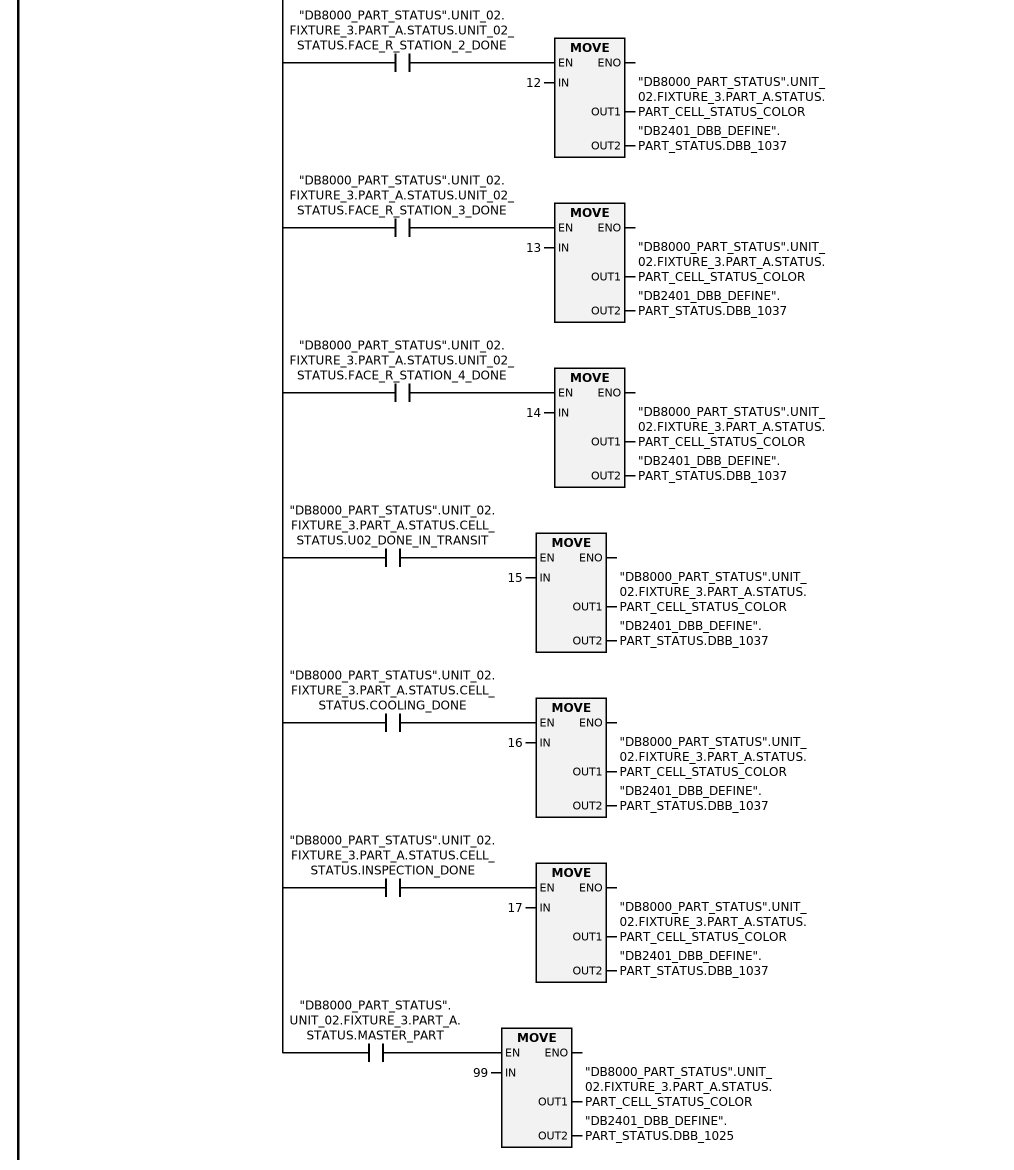
   RUNG wire#powerrail
      Contact( "M_ONE" )
      wire#w1
      I_Contact( "DB8000_PART_STATUS".UNIT_02.FIXTURE_3.PART_A.STATUS.PRESENT )
      { S7_GenerateENO := "TRUE" } Move(in := 0, out1 => "DB2401_DBB_DEFINE".PART_STATUS.DBB_1036, out2 => "DB2401_DBB_DEFINE".PART_STATUS.DBB_1037)
      { S7_GenerateENO := "TRUE" } Move(in := 0, out1 => "DB8000_PART_STATUS".UNIT_02.FIXTURE_3.PART_A.STATUS.PART_MAIN_STATUS_COLOR, out2 => "DB8000_PART_STATUS".UNIT_02.FIXTURE_3.PART_A.STATUS.PART_CELL_STATUS_COLOR)
   END_RUNG
   RUNG wire#w1
      Contact( "DB8000_PART_STATUS".UNIT_02.FIXTURE_3.PART_A.STATUS.PRESENT )
      wire#w2
      I_Contact( "DB8000_PART_STATUS".UNIT_02.FIXTURE_3.PART_A.STATUS.PART_REJECTED )
      I_Contact( "DB8000_PART_STATUS".UNIT_02.FIXTURE_3.PART_A.STATUS.QUALITY_PART )
      { S7_GenerateENO := "TRUE" } Move(in := 1, out1 => "DB8000_PART_STATUS".UNIT_02.FIXTURE_3.PART_A.STATUS.PART_MAIN_STATUS_COLOR, out2 => "DB2401_DBB_DEFINE".PART_STATUS.DBB_1036)
   END_RUNG
   RUNG wire#w2
      Contact( "DB8000_PART_STATUS".UNIT_02.FIXTURE_3.PART_A.STATUS.PART_REJECTED )
      { S7_GenerateENO := "TRUE" } Move(in := 2, out1 => "DB8000_PART_STATUS".UNIT_02.FIXTURE_3.PART_A.STATUS.PART_MAIN_STATUS_COLOR, out2 => "DB2401_DBB_DEFINE".PART_STATUS.DBB_1036)
   END_RUNG
   RUNG wire#w2
      Contact( "DB8000_PART_STATUS".UNIT_02.FIXTURE_3.PART_A.STATUS.QUALITY_PART )
      I_Contact( "DB8000_PART_STATUS".UNIT_02.FIXTURE_3.PART_A.STATUS.PART_REJECTED )
      { S7_GenerateENO := "TRUE" } Move(in := 3, out1 => "DB8000_PART_STATUS".UNIT_02.FIXTURE_3.PART_A.STATUS.PART_MAIN_STATUS_COLOR, out2 => "DB2401_DBB_DEFINE".PART_STATUS.DBB_1036)
   END_RUNG
   RUNG wire#w1
      Contact( "DB8000_PART_STATUS".UNIT_02.FIXTURE_3.PART_A.STATUS.PRESENT )
      wire#w3
      Contact( "DB8000_PART_STATUS".UNIT_02.FIXTURE_3.PART_A.STATUS.CELL_STATUS.NEW_IN_TRANSIT )
      { S7_GenerateENO := "TRUE" } Move(in := 1, out1 => "DB8000_PART_STATUS".UNIT_02.FIXTURE_3.PART_A.STATUS.PART_CELL_STATUS_COLOR, out2 => "DB2401_DBB_DEFINE".PART_STATUS.DBB_1037)
   END_RUNG
   RUNG wire#w3
      Contact( "DB8000_PART_STATUS".UNIT_02.FIXTURE_3.PART_A.STATUS.UNIT_01_STATUS.FACE_N_STATION_3_DONE )
      { S7_GenerateENO := "TRUE" } Move(in := 2, out1 => "DB8000_PART_STATUS".UNIT_02.FIXTURE_3.PART_A.STATUS.PART_CELL_STATUS_COLOR, out2 => "DB2401_DBB_DEFINE".PART_STATUS.DBB_1037)
   END_RUNG
   RUNG wire#w3
      Contact( "DB8000_PART_STATUS".UNIT_02.FIXTURE_3.PART_A.STATUS.UNIT_01_STATUS.FACE_N_STATION_4_DONE )
      { S7_GenerateENO := "TRUE" } Move(in := 3, out1 => "DB8000_PART_STATUS".UNIT_02.FIXTURE_3.PART_A.STATUS.PART_CELL_STATUS_COLOR, out2 => "DB2401_DBB_DEFINE".PART_STATUS.DBB_1037)
   END_RUNG
   RUNG wire#w3
      Contact( "DB8000_PART_STATUS".UNIT_02.FIXTURE_3.PART_A.STATUS.CELL_STATUS.U01_ONE_FACE_DONE_ROTATED )
      { S7_GenerateENO := "TRUE" } Move(in := 4, out1 => "DB8000_PART_STATUS".UNIT_02.FIXTURE_3.PART_A.STATUS.PART_CELL_STATUS_COLOR, out2 => "DB2401_DBB_DEFINE".PART_STATUS.DBB_1037)
   END_RUNG
   RUNG wire#w3
      Contact( "DB8000_PART_STATUS".UNIT_02.FIXTURE_3.PART_A.STATUS.UNIT_01_STATUS.FACE_R_STATION_3_DONE )
      { S7_GenerateENO := "TRUE" } Move(in := 5, out1 => "DB8000_PART_STATUS".UNIT_02.FIXTURE_3.PART_A.STATUS.PART_CELL_STATUS_COLOR, out2 => "DB2401_DBB_DEFINE".PART_STATUS.DBB_1037)
   END_RUNG
   RUNG wire#w3
      Contact( "DB8000_PART_STATUS".UNIT_02.FIXTURE_3.PART_A.STATUS.UNIT_01_STATUS.FACE_R_STATION_4_DONE )
      { S7_GenerateENO := "TRUE" } Move(in := 6, out1 => "DB8000_PART_STATUS".UNIT_02.FIXTURE_3.PART_A.STATUS.PART_CELL_STATUS_COLOR, out2 => "DB2401_DBB_DEFINE".PART_STATUS.DBB_1037)
   END_RUNG
   RUNG wire#w3
      Contact( "DB8000_PART_STATUS".UNIT_02.FIXTURE_3.PART_A.STATUS.CELL_STATUS.U01_DONE_IN_TRANSIT )
      { S7_GenerateENO := "TRUE" } Move(in := 7, out1 => "DB8000_PART_STATUS".UNIT_02.FIXTURE_3.PART_A.STATUS.PART_CELL_STATUS_COLOR, out2 => "DB2401_DBB_DEFINE".PART_STATUS.DBB_1037)
   END_RUNG
   RUNG wire#w3
      Contact( "DB8000_PART_STATUS".UNIT_02.FIXTURE_3.PART_A.STATUS.UNIT_02_STATUS.FACE_N_STATION_2_DONE )
      { S7_GenerateENO := "TRUE" } Move(in := 8, out1 => "DB8000_PART_STATUS".UNIT_02.FIXTURE_3.PART_A.STATUS.PART_CELL_STATUS_COLOR, out2 => "DB2401_DBB_DEFINE".PART_STATUS.DBB_1037)
   END_RUNG
   RUNG wire#w3
      Contact( "DB8000_PART_STATUS".UNIT_02.FIXTURE_3.PART_A.STATUS.UNIT_02_STATUS.FACE_N_STATION_3_DONE )
      Move(in := 9, out1 => "DB8000_PART_STATUS".UNIT_02.FIXTURE_3.PART_A.STATUS.PART_CELL_STATUS_COLOR, out2 => "DB2401_DBB_DEFINE".PART_STATUS.DBB_1037)
   END_RUNG
   RUNG wire#w3
      Contact( "DB8000_PART_STATUS".UNIT_02.FIXTURE_3.PART_A.STATUS.UNIT_02_STATUS.FACE_N_STATION_4_DONE )
      Move(in := 10, out1 => "DB8000_PART_STATUS".UNIT_02.FIXTURE_3.PART_A.STATUS.PART_CELL_STATUS_COLOR, out2 => "DB2401_DBB_DEFINE".PART_STATUS.DBB_1037)
   END_RUNG
   RUNG wire#w3
      Contact( "DB8000_PART_STATUS".UNIT_02.FIXTURE_3.PART_A.STATUS.CELL_STATUS.U02_ONE_FACE_DONE_ROTATED )
      Move(in := 11, out1 => "DB8000_PART_STATUS".UNIT_02.FIXTURE_3.PART_A.STATUS.PART_CELL_STATUS_COLOR, out2 => "DB2401_DBB_DEFINE".PART_STATUS.DBB_1037)
   END_RUNG
   RUNG wire#w3
      Contact( "DB8000_PART_STATUS".UNIT_02.FIXTURE_3.PART_A.STATUS.UNIT_02_STATUS.FACE_R_STATION_2_DONE )
      Move(in := 12, out1 => "DB8000_PART_STATUS".UNIT_02.FIXTURE_3.PART_A.STATUS.PART_CELL_STATUS_COLOR, out2 => "DB2401_DBB_DEFINE".PART_STATUS.DBB_1037)
   END_RUNG
   RUNG wire#w3
      Contact( "DB8000_PART_STATUS".UNIT_02.FIXTURE_3.PART_A.STATUS.UNIT_02_STATUS.FACE_R_STATION_3_DONE )
      Move(in := 13, out1 => "DB8000_PART_STATUS".UNIT_02.FIXTURE_3.PART_A.STATUS.PART_CELL_STATUS_COLOR, out2 => "DB2401_DBB_DEFINE".PART_STATUS.DBB_1037)
   END_RUNG
   RUNG wire#w3
      Contact( "DB8000_PART_STATUS".UNIT_02.FIXTURE_3.PART_A.STATUS.UNIT_02_STATUS.FACE_R_STATION_4_DONE )
      Move(in := 14, out1 => "DB8000_PART_STATUS".UNIT_02.FIXTURE_3.PART_A.STATUS.PART_CELL_STATUS_COLOR, out2 => "DB2401_DBB_DEFINE".PART_STATUS.DBB_1037)
   END_RUNG
   RUNG wire#w3
      Contact( "DB8000_PART_STATUS".UNIT_02.FIXTURE_3.PART_A.STATUS.CELL_STATUS.U02_DONE_IN_TRANSIT )
      Move(in := 15, out1 => "DB8000_PART_STATUS".UNIT_02.FIXTURE_3.PART_A.STATUS.PART_CELL_STATUS_COLOR, out2 => "DB2401_DBB_DEFINE".PART_STATUS.DBB_1037)
   END_RUNG
   RUNG wire#w3
      Contact( "DB8000_PART_STATUS".UNIT_02.FIXTURE_3.PART_A.STATUS.CELL_STATUS.COOLING_DONE )
      Move(in := 16, out1 => "DB8000_PART_STATUS".UNIT_02.FIXTURE_3.PART_A.STATUS.PART_CELL_STATUS_COLOR, out2 => "DB2401_DBB_DEFINE".PART_STATUS.DBB_1037)
   END_RUNG
   RUNG wire#w3
      Contact( "DB8000_PART_STATUS".UNIT_02.FIXTURE_3.PART_A.STATUS.CELL_STATUS.INSPECTION_DONE )
      Move(in := 17, out1 => "DB8000_PART_STATUS".UNIT_02.FIXTURE_3.PART_A.STATUS.PART_CELL_STATUS_COLOR, out2 => "DB2401_DBB_DEFINE".PART_STATUS.DBB_1037)
   END_RUNG
   RUNG wire#w3
      Contact( "DB8000_PART_STATUS".UNIT_02.FIXTURE_3.PART_A.STATUS.MASTER_PART )
      Move(in := 99, out1 => "DB8000_PART_STATUS".UNIT_02.FIXTURE_3.PART_A.STATUS.PART_CELL_STATUS_COLOR, out2 => "DB2401_DBB_DEFINE".PART_STATUS.DBB_1025)
   END_RUNG
   // the same network as SCL:
   // ENO of a box is taken as its EN; it also drops when the box reports an error
   IF "M_ONE" AND NOT "DB8000_PART_STATUS".UNIT_02.FIXTURE_3.PART_A.STATUS.PRESENT THEN
       "DB2401_DBB_DEFINE".PART_STATUS.DBB_1036 := 0;
       "DB2401_DBB_DEFINE".PART_STATUS.DBB_1037 := 0;
       "DB8000_PART_STATUS".UNIT_02.FIXTURE_3.PART_A.STATUS.PART_MAIN_STATUS_COLOR := 0;
       "DB8000_PART_STATUS".UNIT_02.FIXTURE_3.PART_A.STATUS.PART_CELL_STATUS_COLOR := 0;
   END_IF;
   #_w1 := "M_ONE" AND "DB8000_PART_STATUS".UNIT_02.FIXTURE_3.PART_A.STATUS.PRESENT;
   IF #_w1 AND NOT "DB8000_PART_STATUS".UNIT_02.FIXTURE_3.PART_A.STATUS.PART_REJECTED AND NOT "DB8000_PART_STATUS".UNIT_02.FIXTURE_3.PART_A.STATUS.QUALITY_PART THEN
       "DB8000_PART_STATUS".UNIT_02.FIXTURE_3.PART_A.STATUS.PART_MAIN_STATUS_COLOR := 1;
       "DB2401_DBB_DEFINE".PART_STATUS.DBB_1036 := 1;
   END_IF;
   IF #_w1 AND "DB8000_PART_STATUS".UNIT_02.FIXTURE_3.PART_A.STATUS.PART_REJECTED THEN
       "DB8000_PART_STATUS".UNIT_02.FIXTURE_3.PART_A.STATUS.PART_MAIN_STATUS_COLOR := 2;
       "DB2401_DBB_DEFINE".PART_STATUS.DBB_1036 := 2;
   END_IF;
   IF #_w1 AND "DB8000_PART_STATUS".UNIT_02.FIXTURE_3.PART_A.STATUS.QUALITY_PART AND NOT "DB8000_PART_STATUS".UNIT_02.FIXTURE_3.PART_A.STATUS.PART_REJECTED THEN
       "DB8000_PART_STATUS".UNIT_02.FIXTURE_3.PART_A.STATUS.PART_MAIN_STATUS_COLOR := 3;
       "DB2401_DBB_DEFINE".PART_STATUS.DBB_1036 := 3;
   END_IF;
   #_w2 := "M_ONE" AND "DB8000_PART_STATUS".UNIT_02.FIXTURE_3.PART_A.STATUS.PRESENT;
   IF #_w2 AND "DB8000_PART_STATUS".UNIT_02.FIXTURE_3.PART_A.STATUS.CELL_STATUS.NEW_IN_TRANSIT THEN
       "DB8000_PART_STATUS".UNIT_02.FIXTURE_3.PART_A.STATUS.PART_CELL_STATUS_COLOR := 1;
       "DB2401_DBB_DEFINE".PART_STATUS.DBB_1037 := 1;
   END_IF;
   IF #_w2 AND "DB8000_PART_STATUS".UNIT_02.FIXTURE_3.PART_A.STATUS.UNIT_01_STATUS.FACE_N_STATION_3_DONE THEN
       "DB8000_PART_STATUS".UNIT_02.FIXTURE_3.PART_A.STATUS.PART_CELL_STATUS_COLOR := 2;
       "DB2401_DBB_DEFINE".PART_STATUS.DBB_1037 := 2;
   END_IF;
   IF #_w2 AND "DB8000_PART_STATUS".UNIT_02.FIXTURE_3.PART_A.STATUS.UNIT_01_STATUS.FACE_N_STATION_4_DONE THEN
       "DB8000_PART_STATUS".UNIT_02.FIXTURE_3.PART_A.STATUS.PART_CELL_STATUS_COLOR := 3;
       "DB2401_DBB_DEFINE".PART_STATUS.DBB_1037 := 3;
   END_IF;
   IF #_w2 AND "DB8000_PART_STATUS".UNIT_02.FIXTURE_3.PART_A.STATUS.CELL_STATUS.U01_ONE_FACE_DONE_ROTATED THEN
       "DB8000_PART_STATUS".UNIT_02.FIXTURE_3.PART_A.STATUS.PART_CELL_STATUS_COLOR := 4;
       "DB2401_DBB_DEFINE".PART_STATUS.DBB_1037 := 4;
   END_IF;
   IF #_w2 AND "DB8000_PART_STATUS".UNIT_02.FIXTURE_3.PART_A.STATUS.UNIT_01_STATUS.FACE_R_STATION_3_DONE THEN
       "DB8000_PART_STATUS".UNIT_02.FIXTURE_3.PART_A.STATUS.PART_CELL_STATUS_COLOR := 5;
       "DB2401_DBB_DEFINE".PART_STATUS.DBB_1037 := 5;
   END_IF;
   IF #_w2 AND "DB8000_PART_STATUS".UNIT_02.FIXTURE_3.PART_A.STATUS.UNIT_01_STATUS.FACE_R_STATION_4_DONE THEN
       "DB8000_PART_STATUS".UNIT_02.FIXTURE_3.PART_A.STATUS.PART_CELL_STATUS_COLOR := 6;
       "DB2401_DBB_DEFINE".PART_STATUS.DBB_1037 := 6;
   END_IF;
   IF #_w2 AND "DB8000_PART_STATUS".UNIT_02.FIXTURE_3.PART_A.STATUS.CELL_STATUS.U01_DONE_IN_TRANSIT THEN
       "DB8000_PART_STATUS".UNIT_02.FIXTURE_3.PART_A.STATUS.PART_CELL_STATUS_COLOR := 7;
       "DB2401_DBB_DEFINE".PART_STATUS.DBB_1037 := 7;
   END_IF;
   IF #_w2 AND "DB8000_PART_STATUS".UNIT_02.FIXTURE_3.PART_A.STATUS.UNIT_02_STATUS.FACE_N_STATION_2_DONE THEN
       "DB8000_PART_STATUS".UNIT_02.FIXTURE_3.PART_A.STATUS.PART_CELL_STATUS_COLOR := 8;
       "DB2401_DBB_DEFINE".PART_STATUS.DBB_1037 := 8;
   END_IF;
   IF #_w2 AND "DB8000_PART_STATUS".UNIT_02.FIXTURE_3.PART_A.STATUS.UNIT_02_STATUS.FACE_N_STATION_3_DONE THEN
       "DB8000_PART_STATUS".UNIT_02.FIXTURE_3.PART_A.STATUS.PART_CELL_STATUS_COLOR := 9;
       "DB2401_DBB_DEFINE".PART_STATUS.DBB_1037 := 9;
   END_IF;
   IF #_w2 AND "DB8000_PART_STATUS".UNIT_02.FIXTURE_3.PART_A.STATUS.UNIT_02_STATUS.FACE_N_STATION_4_DONE THEN
       "DB8000_PART_STATUS".UNIT_02.FIXTURE_3.PART_A.STATUS.PART_CELL_STATUS_COLOR := 10;
       "DB2401_DBB_DEFINE".PART_STATUS.DBB_1037 := 10;
   END_IF;
   IF #_w2 AND "DB8000_PART_STATUS".UNIT_02.FIXTURE_3.PART_A.STATUS.CELL_STATUS.U02_ONE_FACE_DONE_ROTATED THEN
       "DB8000_PART_STATUS".UNIT_02.FIXTURE_3.PART_A.STATUS.PART_CELL_STATUS_COLOR := 11;
       "DB2401_DBB_DEFINE".PART_STATUS.DBB_1037 := 11;
   END_IF;
   IF #_w2 AND "DB8000_PART_STATUS".UNIT_02.FIXTURE_3.PART_A.STATUS.UNIT_02_STATUS.FACE_R_STATION_2_DONE THEN
       "DB8000_PART_STATUS".UNIT_02.FIXTURE_3.PART_A.STATUS.PART_CELL_STATUS_COLOR := 12;
       "DB2401_DBB_DEFINE".PART_STATUS.DBB_1037 := 12;
   END_IF;
   IF #_w2 AND "DB8000_PART_STATUS".UNIT_02.FIXTURE_3.PART_A.STATUS.UNIT_02_STATUS.FACE_R_STATION_3_DONE THEN
       "DB8000_PART_STATUS".UNIT_02.FIXTURE_3.PART_A.STATUS.PART_CELL_STATUS_COLOR := 13;
       "DB2401_DBB_DEFINE".PART_STATUS.DBB_1037 := 13;
   END_IF;
   IF #_w2 AND "DB8000_PART_STATUS".UNIT_02.FIXTURE_3.PART_A.STATUS.UNIT_02_STATUS.FACE_R_STATION_4_DONE THEN
       "DB8000_PART_STATUS".UNIT_02.FIXTURE_3.PART_A.STATUS.PART_CELL_STATUS_COLOR := 14;
       "DB2401_DBB_DEFINE".PART_STATUS.DBB_1037 := 14;
   END_IF;
   IF #_w2 AND "DB8000_PART_STATUS".UNIT_02.FIXTURE_3.PART_A.STATUS.CELL_STATUS.U02_DONE_IN_TRANSIT THEN
       "DB8000_PART_STATUS".UNIT_02.FIXTURE_3.PART_A.STATUS.PART_CELL_STATUS_COLOR := 15;
       "DB2401_DBB_DEFINE".PART_STATUS.DBB_1037 := 15;
   END_IF;
   IF #_w2 AND "DB8000_PART_STATUS".UNIT_02.FIXTURE_3.PART_A.STATUS.CELL_STATUS.COOLING_DONE THEN
       "DB8000_PART_STATUS".UNIT_02.FIXTURE_3.PART_A.STATUS.PART_CELL_STATUS_COLOR := 16;
       "DB2401_DBB_DEFINE".PART_STATUS.DBB_1037 := 16;
   END_IF;
   IF #_w2 AND "DB8000_PART_STATUS".UNIT_02.FIXTURE_3.PART_A.STATUS.CELL_STATUS.INSPECTION_DONE THEN
       "DB8000_PART_STATUS".UNIT_02.FIXTURE_3.PART_A.STATUS.PART_CELL_STATUS_COLOR := 17;
       "DB2401_DBB_DEFINE".PART_STATUS.DBB_1037 := 17;
   END_IF;
   IF #_w2 AND "DB8000_PART_STATUS".UNIT_02.FIXTURE_3.PART_A.STATUS.MASTER_PART THEN
       "DB8000_PART_STATUS".UNIT_02.FIXTURE_3.PART_A.STATUS.PART_CELL_STATUS_COLOR := 99;
       "DB2401_DBB_DEFINE".PART_STATUS.DBB_1025 := 99;
   END_IF;
END_REGION

REGION Network 22: PART A FIXTURE 4 COLOR STATUS
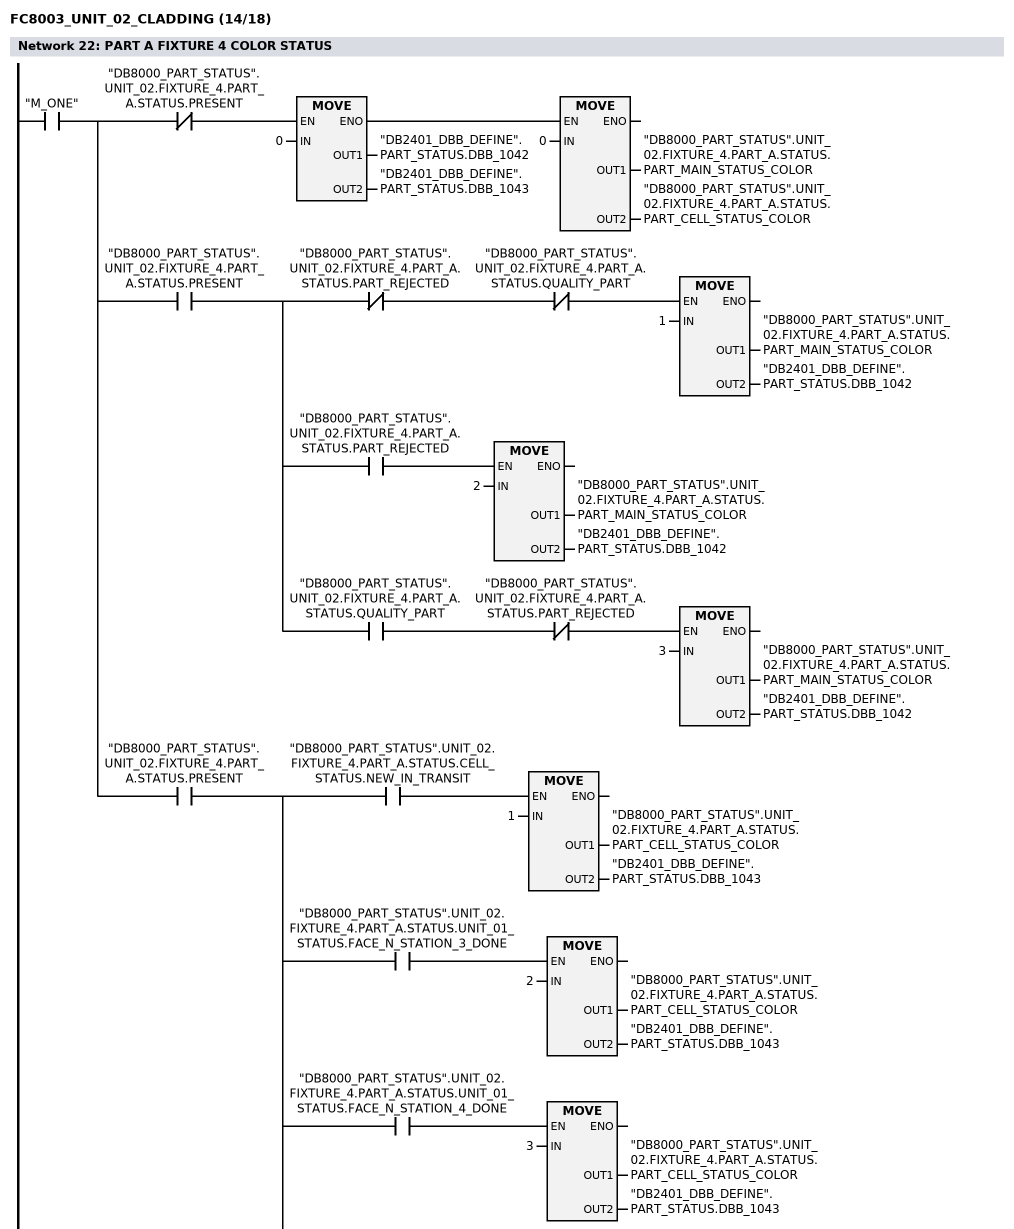
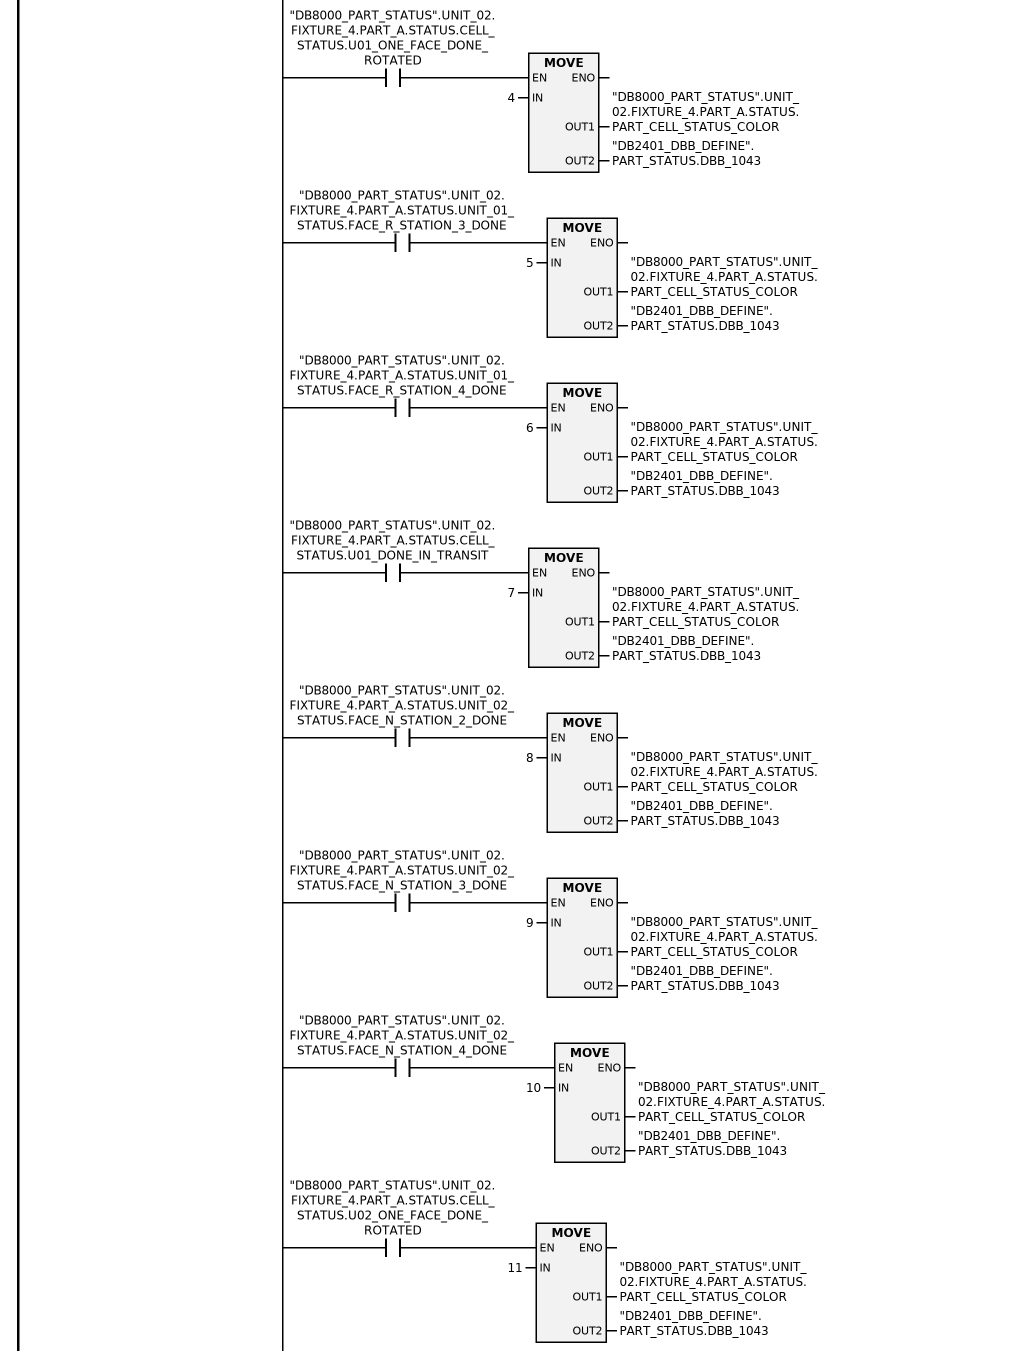
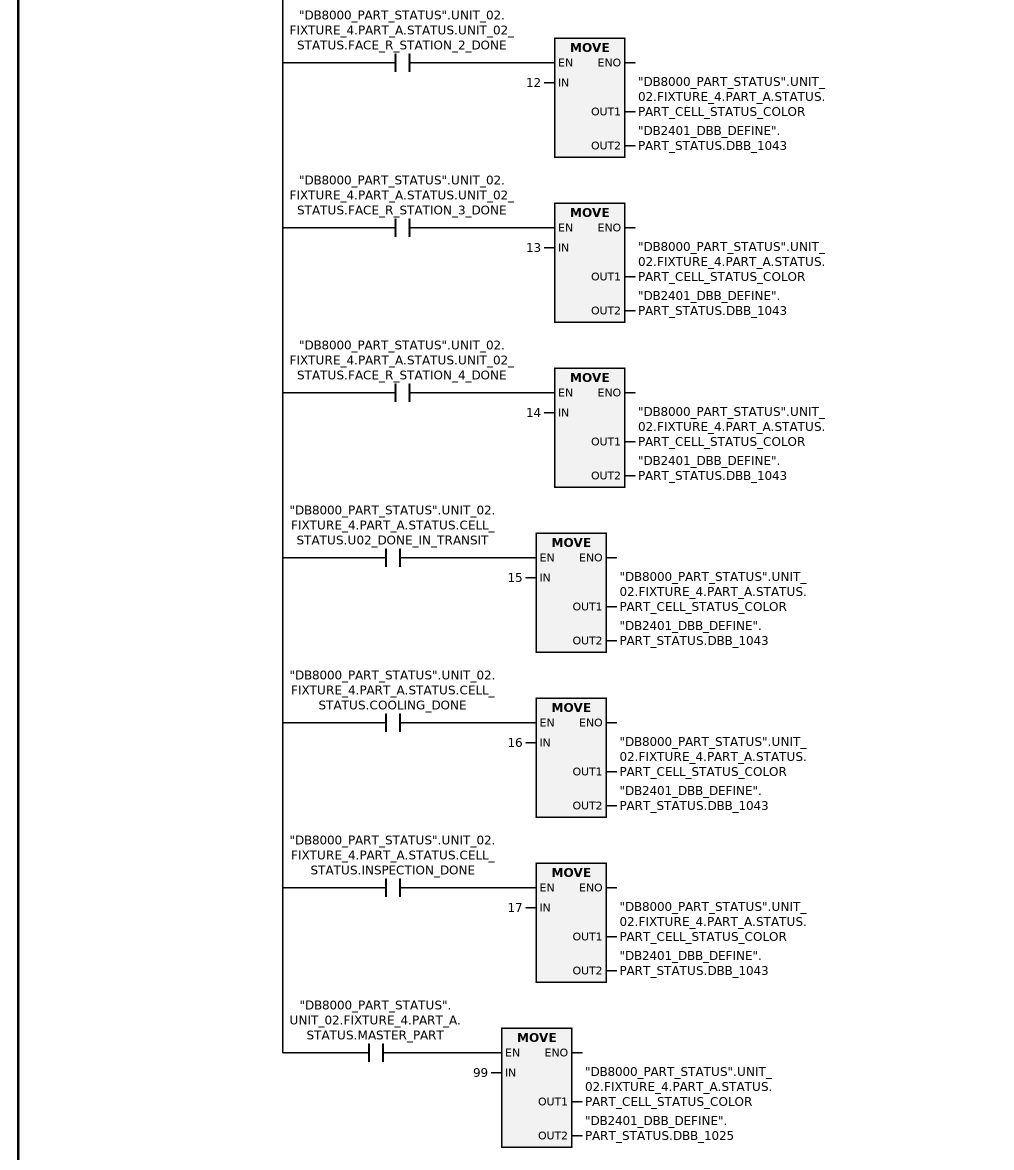
   RUNG wire#powerrail
      Contact( "M_ONE" )
      wire#w1
      I_Contact( "DB8000_PART_STATUS".UNIT_02.FIXTURE_4.PART_A.STATUS.PRESENT )
      { S7_GenerateENO := "TRUE" } Move(in := 0, out1 => "DB2401_DBB_DEFINE".PART_STATUS.DBB_1042, out2 => "DB2401_DBB_DEFINE".PART_STATUS.DBB_1043)
      { S7_GenerateENO := "TRUE" } Move(in := 0, out1 => "DB8000_PART_STATUS".UNIT_02.FIXTURE_4.PART_A.STATUS.PART_MAIN_STATUS_COLOR, out2 => "DB8000_PART_STATUS".UNIT_02.FIXTURE_4.PART_A.STATUS.PART_CELL_STATUS_COLOR)
   END_RUNG
   RUNG wire#w1
      Contact( "DB8000_PART_STATUS".UNIT_02.FIXTURE_4.PART_A.STATUS.PRESENT )
      wire#w2
      I_Contact( "DB8000_PART_STATUS".UNIT_02.FIXTURE_4.PART_A.STATUS.PART_REJECTED )
      I_Contact( "DB8000_PART_STATUS".UNIT_02.FIXTURE_4.PART_A.STATUS.QUALITY_PART )
      { S7_GenerateENO := "TRUE" } Move(in := 1, out1 => "DB8000_PART_STATUS".UNIT_02.FIXTURE_4.PART_A.STATUS.PART_MAIN_STATUS_COLOR, out2 => "DB2401_DBB_DEFINE".PART_STATUS.DBB_1042)
   END_RUNG
   RUNG wire#w2
      Contact( "DB8000_PART_STATUS".UNIT_02.FIXTURE_4.PART_A.STATUS.PART_REJECTED )
      { S7_GenerateENO := "TRUE" } Move(in := 2, out1 => "DB8000_PART_STATUS".UNIT_02.FIXTURE_4.PART_A.STATUS.PART_MAIN_STATUS_COLOR, out2 => "DB2401_DBB_DEFINE".PART_STATUS.DBB_1042)
   END_RUNG
   RUNG wire#w2
      Contact( "DB8000_PART_STATUS".UNIT_02.FIXTURE_4.PART_A.STATUS.QUALITY_PART )
      I_Contact( "DB8000_PART_STATUS".UNIT_02.FIXTURE_4.PART_A.STATUS.PART_REJECTED )
      { S7_GenerateENO := "TRUE" } Move(in := 3, out1 => "DB8000_PART_STATUS".UNIT_02.FIXTURE_4.PART_A.STATUS.PART_MAIN_STATUS_COLOR, out2 => "DB2401_DBB_DEFINE".PART_STATUS.DBB_1042)
   END_RUNG
   RUNG wire#w1
      Contact( "DB8000_PART_STATUS".UNIT_02.FIXTURE_4.PART_A.STATUS.PRESENT )
      wire#w3
      Contact( "DB8000_PART_STATUS".UNIT_02.FIXTURE_4.PART_A.STATUS.CELL_STATUS.NEW_IN_TRANSIT )
      { S7_GenerateENO := "TRUE" } Move(in := 1, out1 => "DB8000_PART_STATUS".UNIT_02.FIXTURE_4.PART_A.STATUS.PART_CELL_STATUS_COLOR, out2 => "DB2401_DBB_DEFINE".PART_STATUS.DBB_1043)
   END_RUNG
   RUNG wire#w3
      Contact( "DB8000_PART_STATUS".UNIT_02.FIXTURE_4.PART_A.STATUS.UNIT_01_STATUS.FACE_N_STATION_3_DONE )
      { S7_GenerateENO := "TRUE" } Move(in := 2, out1 => "DB8000_PART_STATUS".UNIT_02.FIXTURE_4.PART_A.STATUS.PART_CELL_STATUS_COLOR, out2 => "DB2401_DBB_DEFINE".PART_STATUS.DBB_1043)
   END_RUNG
   RUNG wire#w3
      Contact( "DB8000_PART_STATUS".UNIT_02.FIXTURE_4.PART_A.STATUS.UNIT_01_STATUS.FACE_N_STATION_4_DONE )
      { S7_GenerateENO := "TRUE" } Move(in := 3, out1 => "DB8000_PART_STATUS".UNIT_02.FIXTURE_4.PART_A.STATUS.PART_CELL_STATUS_COLOR, out2 => "DB2401_DBB_DEFINE".PART_STATUS.DBB_1043)
   END_RUNG
   RUNG wire#w3
      Contact( "DB8000_PART_STATUS".UNIT_02.FIXTURE_4.PART_A.STATUS.CELL_STATUS.U01_ONE_FACE_DONE_ROTATED )
      { S7_GenerateENO := "TRUE" } Move(in := 4, out1 => "DB8000_PART_STATUS".UNIT_02.FIXTURE_4.PART_A.STATUS.PART_CELL_STATUS_COLOR, out2 => "DB2401_DBB_DEFINE".PART_STATUS.DBB_1043)
   END_RUNG
   RUNG wire#w3
      Contact( "DB8000_PART_STATUS".UNIT_02.FIXTURE_4.PART_A.STATUS.UNIT_01_STATUS.FACE_R_STATION_3_DONE )
      { S7_GenerateENO := "TRUE" } Move(in := 5, out1 => "DB8000_PART_STATUS".UNIT_02.FIXTURE_4.PART_A.STATUS.PART_CELL_STATUS_COLOR, out2 => "DB2401_DBB_DEFINE".PART_STATUS.DBB_1043)
   END_RUNG
   RUNG wire#w3
      Contact( "DB8000_PART_STATUS".UNIT_02.FIXTURE_4.PART_A.STATUS.UNIT_01_STATUS.FACE_R_STATION_4_DONE )
      { S7_GenerateENO := "TRUE" } Move(in := 6, out1 => "DB8000_PART_STATUS".UNIT_02.FIXTURE_4.PART_A.STATUS.PART_CELL_STATUS_COLOR, out2 => "DB2401_DBB_DEFINE".PART_STATUS.DBB_1043)
   END_RUNG
   RUNG wire#w3
      Contact( "DB8000_PART_STATUS".UNIT_02.FIXTURE_4.PART_A.STATUS.CELL_STATUS.U01_DONE_IN_TRANSIT )
      { S7_GenerateENO := "TRUE" } Move(in := 7, out1 => "DB8000_PART_STATUS".UNIT_02.FIXTURE_4.PART_A.STATUS.PART_CELL_STATUS_COLOR, out2 => "DB2401_DBB_DEFINE".PART_STATUS.DBB_1043)
   END_RUNG
   RUNG wire#w3
      Contact( "DB8000_PART_STATUS".UNIT_02.FIXTURE_4.PART_A.STATUS.UNIT_02_STATUS.FACE_N_STATION_2_DONE )
      { S7_GenerateENO := "TRUE" } Move(in := 8, out1 => "DB8000_PART_STATUS".UNIT_02.FIXTURE_4.PART_A.STATUS.PART_CELL_STATUS_COLOR, out2 => "DB2401_DBB_DEFINE".PART_STATUS.DBB_1043)
   END_RUNG
   RUNG wire#w3
      Contact( "DB8000_PART_STATUS".UNIT_02.FIXTURE_4.PART_A.STATUS.UNIT_02_STATUS.FACE_N_STATION_3_DONE )
      Move(in := 9, out1 => "DB8000_PART_STATUS".UNIT_02.FIXTURE_4.PART_A.STATUS.PART_CELL_STATUS_COLOR, out2 => "DB2401_DBB_DEFINE".PART_STATUS.DBB_1043)
   END_RUNG
   RUNG wire#w3
      Contact( "DB8000_PART_STATUS".UNIT_02.FIXTURE_4.PART_A.STATUS.UNIT_02_STATUS.FACE_N_STATION_4_DONE )
      Move(in := 10, out1 => "DB8000_PART_STATUS".UNIT_02.FIXTURE_4.PART_A.STATUS.PART_CELL_STATUS_COLOR, out2 => "DB2401_DBB_DEFINE".PART_STATUS.DBB_1043)
   END_RUNG
   RUNG wire#w3
      Contact( "DB8000_PART_STATUS".UNIT_02.FIXTURE_4.PART_A.STATUS.CELL_STATUS.U02_ONE_FACE_DONE_ROTATED )
      Move(in := 11, out1 => "DB8000_PART_STATUS".UNIT_02.FIXTURE_4.PART_A.STATUS.PART_CELL_STATUS_COLOR, out2 => "DB2401_DBB_DEFINE".PART_STATUS.DBB_1043)
   END_RUNG
   RUNG wire#w3
      Contact( "DB8000_PART_STATUS".UNIT_02.FIXTURE_4.PART_A.STATUS.UNIT_02_STATUS.FACE_R_STATION_2_DONE )
      Move(in := 12, out1 => "DB8000_PART_STATUS".UNIT_02.FIXTURE_4.PART_A.STATUS.PART_CELL_STATUS_COLOR, out2 => "DB2401_DBB_DEFINE".PART_STATUS.DBB_1043)
   END_RUNG
   RUNG wire#w3
      Contact( "DB8000_PART_STATUS".UNIT_02.FIXTURE_4.PART_A.STATUS.UNIT_02_STATUS.FACE_R_STATION_3_DONE )
      Move(in := 13, out1 => "DB8000_PART_STATUS".UNIT_02.FIXTURE_4.PART_A.STATUS.PART_CELL_STATUS_COLOR, out2 => "DB2401_DBB_DEFINE".PART_STATUS.DBB_1043)
   END_RUNG
   RUNG wire#w3
      Contact( "DB8000_PART_STATUS".UNIT_02.FIXTURE_4.PART_A.STATUS.UNIT_02_STATUS.FACE_R_STATION_4_DONE )
      Move(in := 14, out1 => "DB8000_PART_STATUS".UNIT_02.FIXTURE_4.PART_A.STATUS.PART_CELL_STATUS_COLOR, out2 => "DB2401_DBB_DEFINE".PART_STATUS.DBB_1043)
   END_RUNG
   RUNG wire#w3
      Contact( "DB8000_PART_STATUS".UNIT_02.FIXTURE_4.PART_A.STATUS.CELL_STATUS.U02_DONE_IN_TRANSIT )
      Move(in := 15, out1 => "DB8000_PART_STATUS".UNIT_02.FIXTURE_4.PART_A.STATUS.PART_CELL_STATUS_COLOR, out2 => "DB2401_DBB_DEFINE".PART_STATUS.DBB_1043)
   END_RUNG
   RUNG wire#w3
      Contact( "DB8000_PART_STATUS".UNIT_02.FIXTURE_4.PART_A.STATUS.CELL_STATUS.COOLING_DONE )
      Move(in := 16, out1 => "DB8000_PART_STATUS".UNIT_02.FIXTURE_4.PART_A.STATUS.PART_CELL_STATUS_COLOR, out2 => "DB2401_DBB_DEFINE".PART_STATUS.DBB_1043)
   END_RUNG
   RUNG wire#w3
      Contact( "DB8000_PART_STATUS".UNIT_02.FIXTURE_4.PART_A.STATUS.CELL_STATUS.INSPECTION_DONE )
      Move(in := 17, out1 => "DB8000_PART_STATUS".UNIT_02.FIXTURE_4.PART_A.STATUS.PART_CELL_STATUS_COLOR, out2 => "DB2401_DBB_DEFINE".PART_STATUS.DBB_1043)
   END_RUNG
   RUNG wire#w3
      Contact( "DB8000_PART_STATUS".UNIT_02.FIXTURE_4.PART_A.STATUS.MASTER_PART )
      Move(in := 99, out1 => "DB8000_PART_STATUS".UNIT_02.FIXTURE_4.PART_A.STATUS.PART_CELL_STATUS_COLOR, out2 => "DB2401_DBB_DEFINE".PART_STATUS.DBB_1025)
   END_RUNG
   // the same network as SCL:
   // ENO of a box is taken as its EN; it also drops when the box reports an error
   IF "M_ONE" AND NOT "DB8000_PART_STATUS".UNIT_02.FIXTURE_4.PART_A.STATUS.PRESENT THEN
       "DB2401_DBB_DEFINE".PART_STATUS.DBB_1042 := 0;
       "DB2401_DBB_DEFINE".PART_STATUS.DBB_1043 := 0;
       "DB8000_PART_STATUS".UNIT_02.FIXTURE_4.PART_A.STATUS.PART_MAIN_STATUS_COLOR := 0;
       "DB8000_PART_STATUS".UNIT_02.FIXTURE_4.PART_A.STATUS.PART_CELL_STATUS_COLOR := 0;
   END_IF;
   #_w1 := "M_ONE" AND "DB8000_PART_STATUS".UNIT_02.FIXTURE_4.PART_A.STATUS.PRESENT;
   IF #_w1 AND NOT "DB8000_PART_STATUS".UNIT_02.FIXTURE_4.PART_A.STATUS.PART_REJECTED AND NOT "DB8000_PART_STATUS".UNIT_02.FIXTURE_4.PART_A.STATUS.QUALITY_PART THEN
       "DB8000_PART_STATUS".UNIT_02.FIXTURE_4.PART_A.STATUS.PART_MAIN_STATUS_COLOR := 1;
       "DB2401_DBB_DEFINE".PART_STATUS.DBB_1042 := 1;
   END_IF;
   IF #_w1 AND "DB8000_PART_STATUS".UNIT_02.FIXTURE_4.PART_A.STATUS.PART_REJECTED THEN
       "DB8000_PART_STATUS".UNIT_02.FIXTURE_4.PART_A.STATUS.PART_MAIN_STATUS_COLOR := 2;
       "DB2401_DBB_DEFINE".PART_STATUS.DBB_1042 := 2;
   END_IF;
   IF #_w1 AND "DB8000_PART_STATUS".UNIT_02.FIXTURE_4.PART_A.STATUS.QUALITY_PART AND NOT "DB8000_PART_STATUS".UNIT_02.FIXTURE_4.PART_A.STATUS.PART_REJECTED THEN
       "DB8000_PART_STATUS".UNIT_02.FIXTURE_4.PART_A.STATUS.PART_MAIN_STATUS_COLOR := 3;
       "DB2401_DBB_DEFINE".PART_STATUS.DBB_1042 := 3;
   END_IF;
   #_w2 := "M_ONE" AND "DB8000_PART_STATUS".UNIT_02.FIXTURE_4.PART_A.STATUS.PRESENT;
   IF #_w2 AND "DB8000_PART_STATUS".UNIT_02.FIXTURE_4.PART_A.STATUS.CELL_STATUS.NEW_IN_TRANSIT THEN
       "DB8000_PART_STATUS".UNIT_02.FIXTURE_4.PART_A.STATUS.PART_CELL_STATUS_COLOR := 1;
       "DB2401_DBB_DEFINE".PART_STATUS.DBB_1043 := 1;
   END_IF;
   IF #_w2 AND "DB8000_PART_STATUS".UNIT_02.FIXTURE_4.PART_A.STATUS.UNIT_01_STATUS.FACE_N_STATION_3_DONE THEN
       "DB8000_PART_STATUS".UNIT_02.FIXTURE_4.PART_A.STATUS.PART_CELL_STATUS_COLOR := 2;
       "DB2401_DBB_DEFINE".PART_STATUS.DBB_1043 := 2;
   END_IF;
   IF #_w2 AND "DB8000_PART_STATUS".UNIT_02.FIXTURE_4.PART_A.STATUS.UNIT_01_STATUS.FACE_N_STATION_4_DONE THEN
       "DB8000_PART_STATUS".UNIT_02.FIXTURE_4.PART_A.STATUS.PART_CELL_STATUS_COLOR := 3;
       "DB2401_DBB_DEFINE".PART_STATUS.DBB_1043 := 3;
   END_IF;
   IF #_w2 AND "DB8000_PART_STATUS".UNIT_02.FIXTURE_4.PART_A.STATUS.CELL_STATUS.U01_ONE_FACE_DONE_ROTATED THEN
       "DB8000_PART_STATUS".UNIT_02.FIXTURE_4.PART_A.STATUS.PART_CELL_STATUS_COLOR := 4;
       "DB2401_DBB_DEFINE".PART_STATUS.DBB_1043 := 4;
   END_IF;
   IF #_w2 AND "DB8000_PART_STATUS".UNIT_02.FIXTURE_4.PART_A.STATUS.UNIT_01_STATUS.FACE_R_STATION_3_DONE THEN
       "DB8000_PART_STATUS".UNIT_02.FIXTURE_4.PART_A.STATUS.PART_CELL_STATUS_COLOR := 5;
       "DB2401_DBB_DEFINE".PART_STATUS.DBB_1043 := 5;
   END_IF;
   IF #_w2 AND "DB8000_PART_STATUS".UNIT_02.FIXTURE_4.PART_A.STATUS.UNIT_01_STATUS.FACE_R_STATION_4_DONE THEN
       "DB8000_PART_STATUS".UNIT_02.FIXTURE_4.PART_A.STATUS.PART_CELL_STATUS_COLOR := 6;
       "DB2401_DBB_DEFINE".PART_STATUS.DBB_1043 := 6;
   END_IF;
   IF #_w2 AND "DB8000_PART_STATUS".UNIT_02.FIXTURE_4.PART_A.STATUS.CELL_STATUS.U01_DONE_IN_TRANSIT THEN
       "DB8000_PART_STATUS".UNIT_02.FIXTURE_4.PART_A.STATUS.PART_CELL_STATUS_COLOR := 7;
       "DB2401_DBB_DEFINE".PART_STATUS.DBB_1043 := 7;
   END_IF;
   IF #_w2 AND "DB8000_PART_STATUS".UNIT_02.FIXTURE_4.PART_A.STATUS.UNIT_02_STATUS.FACE_N_STATION_2_DONE THEN
       "DB8000_PART_STATUS".UNIT_02.FIXTURE_4.PART_A.STATUS.PART_CELL_STATUS_COLOR := 8;
       "DB2401_DBB_DEFINE".PART_STATUS.DBB_1043 := 8;
   END_IF;
   IF #_w2 AND "DB8000_PART_STATUS".UNIT_02.FIXTURE_4.PART_A.STATUS.UNIT_02_STATUS.FACE_N_STATION_3_DONE THEN
       "DB8000_PART_STATUS".UNIT_02.FIXTURE_4.PART_A.STATUS.PART_CELL_STATUS_COLOR := 9;
       "DB2401_DBB_DEFINE".PART_STATUS.DBB_1043 := 9;
   END_IF;
   IF #_w2 AND "DB8000_PART_STATUS".UNIT_02.FIXTURE_4.PART_A.STATUS.UNIT_02_STATUS.FACE_N_STATION_4_DONE THEN
       "DB8000_PART_STATUS".UNIT_02.FIXTURE_4.PART_A.STATUS.PART_CELL_STATUS_COLOR := 10;
       "DB2401_DBB_DEFINE".PART_STATUS.DBB_1043 := 10;
   END_IF;
   IF #_w2 AND "DB8000_PART_STATUS".UNIT_02.FIXTURE_4.PART_A.STATUS.CELL_STATUS.U02_ONE_FACE_DONE_ROTATED THEN
       "DB8000_PART_STATUS".UNIT_02.FIXTURE_4.PART_A.STATUS.PART_CELL_STATUS_COLOR := 11;
       "DB2401_DBB_DEFINE".PART_STATUS.DBB_1043 := 11;
   END_IF;
   IF #_w2 AND "DB8000_PART_STATUS".UNIT_02.FIXTURE_4.PART_A.STATUS.UNIT_02_STATUS.FACE_R_STATION_2_DONE THEN
       "DB8000_PART_STATUS".UNIT_02.FIXTURE_4.PART_A.STATUS.PART_CELL_STATUS_COLOR := 12;
       "DB2401_DBB_DEFINE".PART_STATUS.DBB_1043 := 12;
   END_IF;
   IF #_w2 AND "DB8000_PART_STATUS".UNIT_02.FIXTURE_4.PART_A.STATUS.UNIT_02_STATUS.FACE_R_STATION_3_DONE THEN
       "DB8000_PART_STATUS".UNIT_02.FIXTURE_4.PART_A.STATUS.PART_CELL_STATUS_COLOR := 13;
       "DB2401_DBB_DEFINE".PART_STATUS.DBB_1043 := 13;
   END_IF;
   IF #_w2 AND "DB8000_PART_STATUS".UNIT_02.FIXTURE_4.PART_A.STATUS.UNIT_02_STATUS.FACE_R_STATION_4_DONE THEN
       "DB8000_PART_STATUS".UNIT_02.FIXTURE_4.PART_A.STATUS.PART_CELL_STATUS_COLOR := 14;
       "DB2401_DBB_DEFINE".PART_STATUS.DBB_1043 := 14;
   END_IF;
   IF #_w2 AND "DB8000_PART_STATUS".UNIT_02.FIXTURE_4.PART_A.STATUS.CELL_STATUS.U02_DONE_IN_TRANSIT THEN
       "DB8000_PART_STATUS".UNIT_02.FIXTURE_4.PART_A.STATUS.PART_CELL_STATUS_COLOR := 15;
       "DB2401_DBB_DEFINE".PART_STATUS.DBB_1043 := 15;
   END_IF;
   IF #_w2 AND "DB8000_PART_STATUS".UNIT_02.FIXTURE_4.PART_A.STATUS.CELL_STATUS.COOLING_DONE THEN
       "DB8000_PART_STATUS".UNIT_02.FIXTURE_4.PART_A.STATUS.PART_CELL_STATUS_COLOR := 16;
       "DB2401_DBB_DEFINE".PART_STATUS.DBB_1043 := 16;
   END_IF;
   IF #_w2 AND "DB8000_PART_STATUS".UNIT_02.FIXTURE_4.PART_A.STATUS.CELL_STATUS.INSPECTION_DONE THEN
       "DB8000_PART_STATUS".UNIT_02.FIXTURE_4.PART_A.STATUS.PART_CELL_STATUS_COLOR := 17;
       "DB2401_DBB_DEFINE".PART_STATUS.DBB_1043 := 17;
   END_IF;
   IF #_w2 AND "DB8000_PART_STATUS".UNIT_02.FIXTURE_4.PART_A.STATUS.MASTER_PART THEN
       "DB8000_PART_STATUS".UNIT_02.FIXTURE_4.PART_A.STATUS.PART_CELL_STATUS_COLOR := 99;
       "DB2401_DBB_DEFINE".PART_STATUS.DBB_1025 := 99;
   END_IF;
END_REGION

REGION Network 23: PART A STATION 1 COLOR STATUS
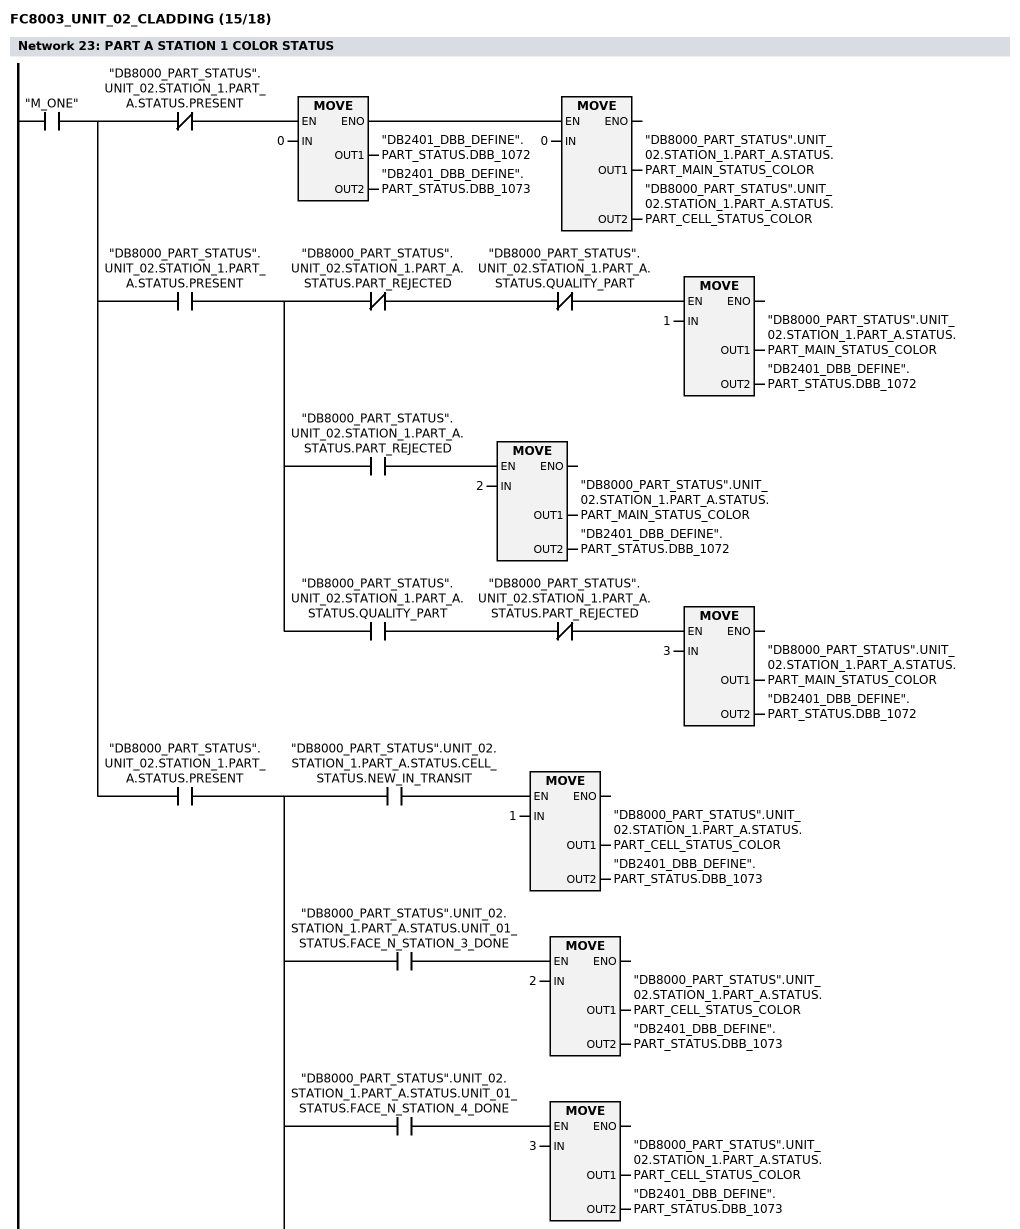
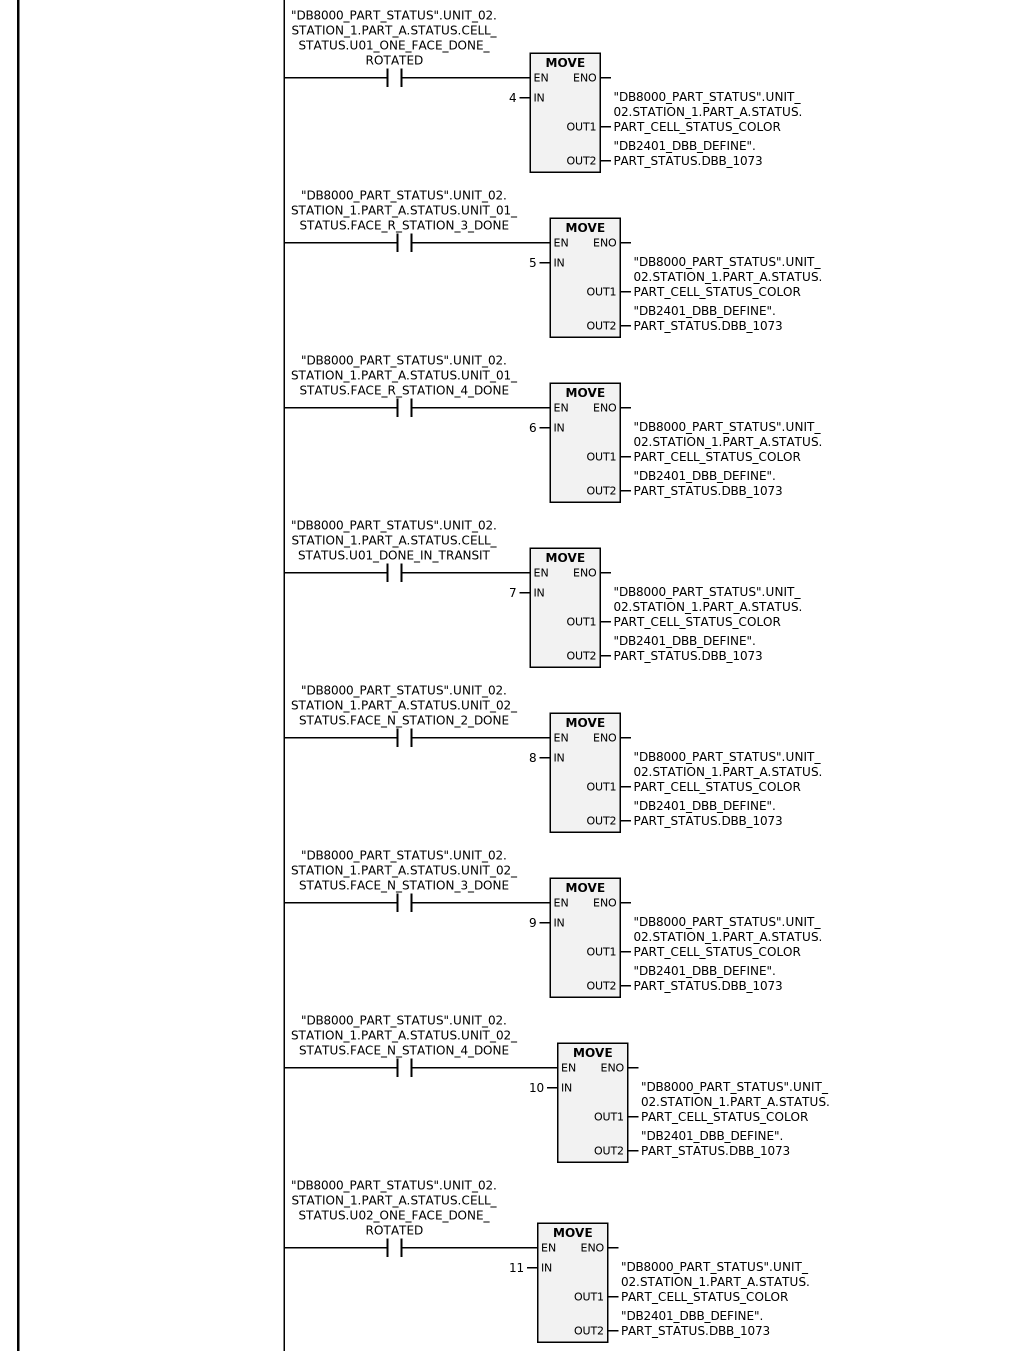
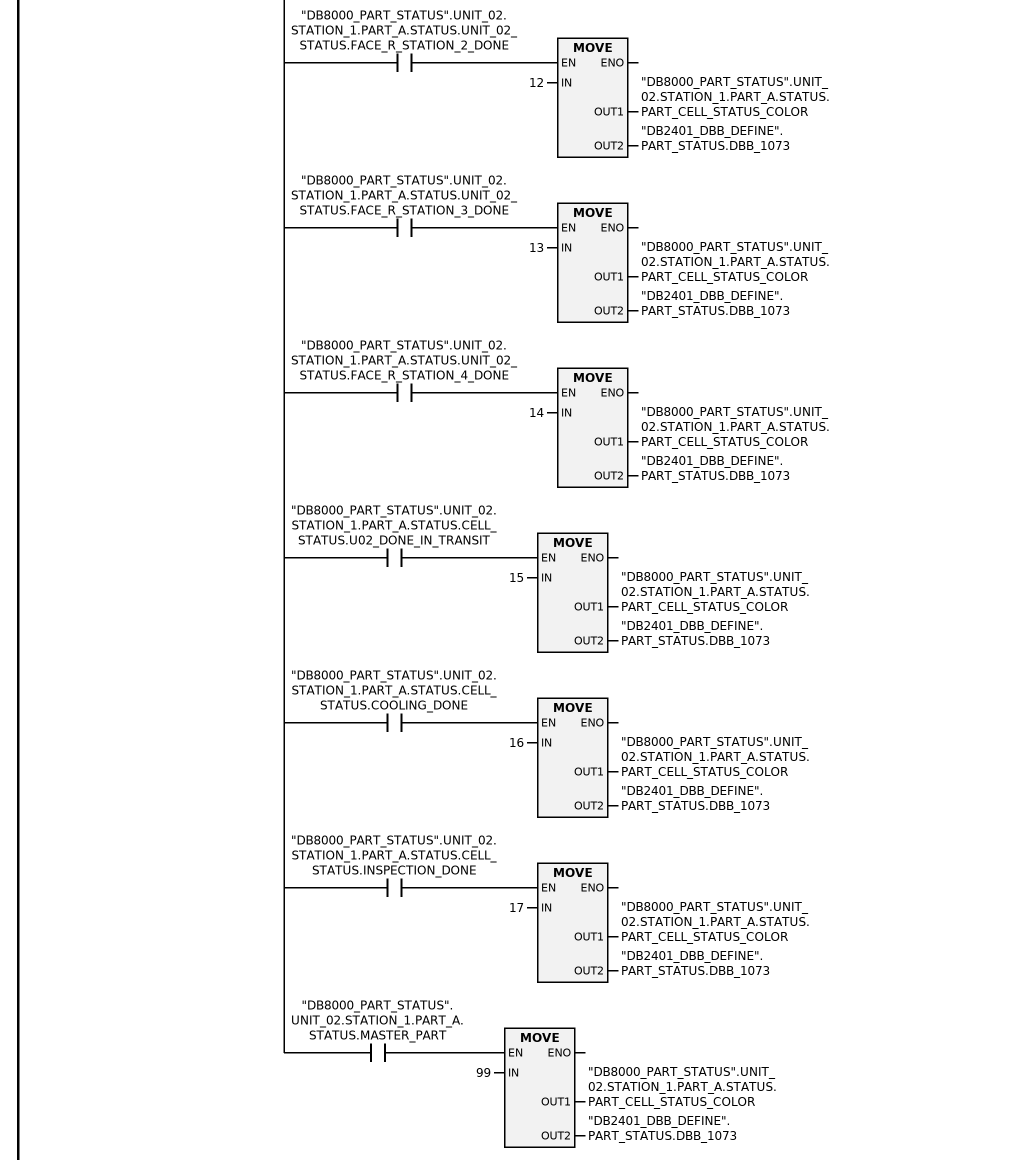
   RUNG wire#powerrail
      Contact( "M_ONE" )
      wire#w1
      I_Contact( "DB8000_PART_STATUS".UNIT_02.STATION_1.PART_A.STATUS.PRESENT )
      { S7_GenerateENO := "TRUE" } Move(in := 0, out1 => "DB2401_DBB_DEFINE".PART_STATUS.DBB_1072, out2 => "DB2401_DBB_DEFINE".PART_STATUS.DBB_1073)
      { S7_GenerateENO := "TRUE" } Move(in := 0, out1 => "DB8000_PART_STATUS".UNIT_02.STATION_1.PART_A.STATUS.PART_MAIN_STATUS_COLOR, out2 => "DB8000_PART_STATUS".UNIT_02.STATION_1.PART_A.STATUS.PART_CELL_STATUS_COLOR)
   END_RUNG
   RUNG wire#w1
      Contact( "DB8000_PART_STATUS".UNIT_02.STATION_1.PART_A.STATUS.PRESENT )
      wire#w2
      I_Contact( "DB8000_PART_STATUS".UNIT_02.STATION_1.PART_A.STATUS.PART_REJECTED )
      I_Contact( "DB8000_PART_STATUS".UNIT_02.STATION_1.PART_A.STATUS.QUALITY_PART )
      { S7_GenerateENO := "TRUE" } Move(in := 1, out1 => "DB8000_PART_STATUS".UNIT_02.STATION_1.PART_A.STATUS.PART_MAIN_STATUS_COLOR, out2 => "DB2401_DBB_DEFINE".PART_STATUS.DBB_1072)
   END_RUNG
   RUNG wire#w2
      Contact( "DB8000_PART_STATUS".UNIT_02.STATION_1.PART_A.STATUS.PART_REJECTED )
      { S7_GenerateENO := "TRUE" } Move(in := 2, out1 => "DB8000_PART_STATUS".UNIT_02.STATION_1.PART_A.STATUS.PART_MAIN_STATUS_COLOR, out2 => "DB2401_DBB_DEFINE".PART_STATUS.DBB_1072)
   END_RUNG
   RUNG wire#w2
      Contact( "DB8000_PART_STATUS".UNIT_02.STATION_1.PART_A.STATUS.QUALITY_PART )
      I_Contact( "DB8000_PART_STATUS".UNIT_02.STATION_1.PART_A.STATUS.PART_REJECTED )
      { S7_GenerateENO := "TRUE" } Move(in := 3, out1 => "DB8000_PART_STATUS".UNIT_02.STATION_1.PART_A.STATUS.PART_MAIN_STATUS_COLOR, out2 => "DB2401_DBB_DEFINE".PART_STATUS.DBB_1072)
   END_RUNG
   RUNG wire#w1
      Contact( "DB8000_PART_STATUS".UNIT_02.STATION_1.PART_A.STATUS.PRESENT )
      wire#w3
      Contact( "DB8000_PART_STATUS".UNIT_02.STATION_1.PART_A.STATUS.CELL_STATUS.NEW_IN_TRANSIT )
      { S7_GenerateENO := "TRUE" } Move(in := 1, out1 => "DB8000_PART_STATUS".UNIT_02.STATION_1.PART_A.STATUS.PART_CELL_STATUS_COLOR, out2 => "DB2401_DBB_DEFINE".PART_STATUS.DBB_1073)
   END_RUNG
   RUNG wire#w3
      Contact( "DB8000_PART_STATUS".UNIT_02.STATION_1.PART_A.STATUS.UNIT_01_STATUS.FACE_N_STATION_3_DONE )
      { S7_GenerateENO := "TRUE" } Move(in := 2, out1 => "DB8000_PART_STATUS".UNIT_02.STATION_1.PART_A.STATUS.PART_CELL_STATUS_COLOR, out2 => "DB2401_DBB_DEFINE".PART_STATUS.DBB_1073)
   END_RUNG
   RUNG wire#w3
      Contact( "DB8000_PART_STATUS".UNIT_02.STATION_1.PART_A.STATUS.UNIT_01_STATUS.FACE_N_STATION_4_DONE )
      { S7_GenerateENO := "TRUE" } Move(in := 3, out1 => "DB8000_PART_STATUS".UNIT_02.STATION_1.PART_A.STATUS.PART_CELL_STATUS_COLOR, out2 => "DB2401_DBB_DEFINE".PART_STATUS.DBB_1073)
   END_RUNG
   RUNG wire#w3
      Contact( "DB8000_PART_STATUS".UNIT_02.STATION_1.PART_A.STATUS.CELL_STATUS.U01_ONE_FACE_DONE_ROTATED )
      { S7_GenerateENO := "TRUE" } Move(in := 4, out1 => "DB8000_PART_STATUS".UNIT_02.STATION_1.PART_A.STATUS.PART_CELL_STATUS_COLOR, out2 => "DB2401_DBB_DEFINE".PART_STATUS.DBB_1073)
   END_RUNG
   RUNG wire#w3
      Contact( "DB8000_PART_STATUS".UNIT_02.STATION_1.PART_A.STATUS.UNIT_01_STATUS.FACE_R_STATION_3_DONE )
      { S7_GenerateENO := "TRUE" } Move(in := 5, out1 => "DB8000_PART_STATUS".UNIT_02.STATION_1.PART_A.STATUS.PART_CELL_STATUS_COLOR, out2 => "DB2401_DBB_DEFINE".PART_STATUS.DBB_1073)
   END_RUNG
   RUNG wire#w3
      Contact( "DB8000_PART_STATUS".UNIT_02.STATION_1.PART_A.STATUS.UNIT_01_STATUS.FACE_R_STATION_4_DONE )
      { S7_GenerateENO := "TRUE" } Move(in := 6, out1 => "DB8000_PART_STATUS".UNIT_02.STATION_1.PART_A.STATUS.PART_CELL_STATUS_COLOR, out2 => "DB2401_DBB_DEFINE".PART_STATUS.DBB_1073)
   END_RUNG
   RUNG wire#w3
      Contact( "DB8000_PART_STATUS".UNIT_02.STATION_1.PART_A.STATUS.CELL_STATUS.U01_DONE_IN_TRANSIT )
      { S7_GenerateENO := "TRUE" } Move(in := 7, out1 => "DB8000_PART_STATUS".UNIT_02.STATION_1.PART_A.STATUS.PART_CELL_STATUS_COLOR, out2 => "DB2401_DBB_DEFINE".PART_STATUS.DBB_1073)
   END_RUNG
   RUNG wire#w3
      Contact( "DB8000_PART_STATUS".UNIT_02.STATION_1.PART_A.STATUS.UNIT_02_STATUS.FACE_N_STATION_2_DONE )
      { S7_GenerateENO := "TRUE" } Move(in := 8, out1 => "DB8000_PART_STATUS".UNIT_02.STATION_1.PART_A.STATUS.PART_CELL_STATUS_COLOR, out2 => "DB2401_DBB_DEFINE".PART_STATUS.DBB_1073)
   END_RUNG
   RUNG wire#w3
      Contact( "DB8000_PART_STATUS".UNIT_02.STATION_1.PART_A.STATUS.UNIT_02_STATUS.FACE_N_STATION_3_DONE )
      Move(in := 9, out1 => "DB8000_PART_STATUS".UNIT_02.STATION_1.PART_A.STATUS.PART_CELL_STATUS_COLOR, out2 => "DB2401_DBB_DEFINE".PART_STATUS.DBB_1073)
   END_RUNG
   RUNG wire#w3
      Contact( "DB8000_PART_STATUS".UNIT_02.STATION_1.PART_A.STATUS.UNIT_02_STATUS.FACE_N_STATION_4_DONE )
      Move(in := 10, out1 => "DB8000_PART_STATUS".UNIT_02.STATION_1.PART_A.STATUS.PART_CELL_STATUS_COLOR, out2 => "DB2401_DBB_DEFINE".PART_STATUS.DBB_1073)
   END_RUNG
   RUNG wire#w3
      Contact( "DB8000_PART_STATUS".UNIT_02.STATION_1.PART_A.STATUS.CELL_STATUS.U02_ONE_FACE_DONE_ROTATED )
      Move(in := 11, out1 => "DB8000_PART_STATUS".UNIT_02.STATION_1.PART_A.STATUS.PART_CELL_STATUS_COLOR, out2 => "DB2401_DBB_DEFINE".PART_STATUS.DBB_1073)
   END_RUNG
   RUNG wire#w3
      Contact( "DB8000_PART_STATUS".UNIT_02.STATION_1.PART_A.STATUS.UNIT_02_STATUS.FACE_R_STATION_2_DONE )
      Move(in := 12, out1 => "DB8000_PART_STATUS".UNIT_02.STATION_1.PART_A.STATUS.PART_CELL_STATUS_COLOR, out2 => "DB2401_DBB_DEFINE".PART_STATUS.DBB_1073)
   END_RUNG
   RUNG wire#w3
      Contact( "DB8000_PART_STATUS".UNIT_02.STATION_1.PART_A.STATUS.UNIT_02_STATUS.FACE_R_STATION_3_DONE )
      Move(in := 13, out1 => "DB8000_PART_STATUS".UNIT_02.STATION_1.PART_A.STATUS.PART_CELL_STATUS_COLOR, out2 => "DB2401_DBB_DEFINE".PART_STATUS.DBB_1073)
   END_RUNG
   RUNG wire#w3
      Contact( "DB8000_PART_STATUS".UNIT_02.STATION_1.PART_A.STATUS.UNIT_02_STATUS.FACE_R_STATION_4_DONE )
      Move(in := 14, out1 => "DB8000_PART_STATUS".UNIT_02.STATION_1.PART_A.STATUS.PART_CELL_STATUS_COLOR, out2 => "DB2401_DBB_DEFINE".PART_STATUS.DBB_1073)
   END_RUNG
   RUNG wire#w3
      Contact( "DB8000_PART_STATUS".UNIT_02.STATION_1.PART_A.STATUS.CELL_STATUS.U02_DONE_IN_TRANSIT )
      Move(in := 15, out1 => "DB8000_PART_STATUS".UNIT_02.STATION_1.PART_A.STATUS.PART_CELL_STATUS_COLOR, out2 => "DB2401_DBB_DEFINE".PART_STATUS.DBB_1073)
   END_RUNG
   RUNG wire#w3
      Contact( "DB8000_PART_STATUS".UNIT_02.STATION_1.PART_A.STATUS.CELL_STATUS.COOLING_DONE )
      Move(in := 16, out1 => "DB8000_PART_STATUS".UNIT_02.STATION_1.PART_A.STATUS.PART_CELL_STATUS_COLOR, out2 => "DB2401_DBB_DEFINE".PART_STATUS.DBB_1073)
   END_RUNG
   RUNG wire#w3
      Contact( "DB8000_PART_STATUS".UNIT_02.STATION_1.PART_A.STATUS.CELL_STATUS.INSPECTION_DONE )
      Move(in := 17, out1 => "DB8000_PART_STATUS".UNIT_02.STATION_1.PART_A.STATUS.PART_CELL_STATUS_COLOR, out2 => "DB2401_DBB_DEFINE".PART_STATUS.DBB_1073)
   END_RUNG
   RUNG wire#w3
      Contact( "DB8000_PART_STATUS".UNIT_02.STATION_1.PART_A.STATUS.MASTER_PART )
      Move(in := 99, out1 => "DB8000_PART_STATUS".UNIT_02.STATION_1.PART_A.STATUS.PART_CELL_STATUS_COLOR, out2 => "DB2401_DBB_DEFINE".PART_STATUS.DBB_1073)
   END_RUNG
   // the same network as SCL:
   // ENO of a box is taken as its EN; it also drops when the box reports an error
   IF "M_ONE" AND NOT "DB8000_PART_STATUS".UNIT_02.STATION_1.PART_A.STATUS.PRESENT THEN
       "DB2401_DBB_DEFINE".PART_STATUS.DBB_1072 := 0;
       "DB2401_DBB_DEFINE".PART_STATUS.DBB_1073 := 0;
       "DB8000_PART_STATUS".UNIT_02.STATION_1.PART_A.STATUS.PART_MAIN_STATUS_COLOR := 0;
       "DB8000_PART_STATUS".UNIT_02.STATION_1.PART_A.STATUS.PART_CELL_STATUS_COLOR := 0;
   END_IF;
   #_w1 := "M_ONE" AND "DB8000_PART_STATUS".UNIT_02.STATION_1.PART_A.STATUS.PRESENT;
   IF #_w1 AND NOT "DB8000_PART_STATUS".UNIT_02.STATION_1.PART_A.STATUS.PART_REJECTED AND NOT "DB8000_PART_STATUS".UNIT_02.STATION_1.PART_A.STATUS.QUALITY_PART THEN
       "DB8000_PART_STATUS".UNIT_02.STATION_1.PART_A.STATUS.PART_MAIN_STATUS_COLOR := 1;
       "DB2401_DBB_DEFINE".PART_STATUS.DBB_1072 := 1;
   END_IF;
   IF #_w1 AND "DB8000_PART_STATUS".UNIT_02.STATION_1.PART_A.STATUS.PART_REJECTED THEN
       "DB8000_PART_STATUS".UNIT_02.STATION_1.PART_A.STATUS.PART_MAIN_STATUS_COLOR := 2;
       "DB2401_DBB_DEFINE".PART_STATUS.DBB_1072 := 2;
   END_IF;
   IF #_w1 AND "DB8000_PART_STATUS".UNIT_02.STATION_1.PART_A.STATUS.QUALITY_PART AND NOT "DB8000_PART_STATUS".UNIT_02.STATION_1.PART_A.STATUS.PART_REJECTED THEN
       "DB8000_PART_STATUS".UNIT_02.STATION_1.PART_A.STATUS.PART_MAIN_STATUS_COLOR := 3;
       "DB2401_DBB_DEFINE".PART_STATUS.DBB_1072 := 3;
   END_IF;
   #_w2 := "M_ONE" AND "DB8000_PART_STATUS".UNIT_02.STATION_1.PART_A.STATUS.PRESENT;
   IF #_w2 AND "DB8000_PART_STATUS".UNIT_02.STATION_1.PART_A.STATUS.CELL_STATUS.NEW_IN_TRANSIT THEN
       "DB8000_PART_STATUS".UNIT_02.STATION_1.PART_A.STATUS.PART_CELL_STATUS_COLOR := 1;
       "DB2401_DBB_DEFINE".PART_STATUS.DBB_1073 := 1;
   END_IF;
   IF #_w2 AND "DB8000_PART_STATUS".UNIT_02.STATION_1.PART_A.STATUS.UNIT_01_STATUS.FACE_N_STATION_3_DONE THEN
       "DB8000_PART_STATUS".UNIT_02.STATION_1.PART_A.STATUS.PART_CELL_STATUS_COLOR := 2;
       "DB2401_DBB_DEFINE".PART_STATUS.DBB_1073 := 2;
   END_IF;
   IF #_w2 AND "DB8000_PART_STATUS".UNIT_02.STATION_1.PART_A.STATUS.UNIT_01_STATUS.FACE_N_STATION_4_DONE THEN
       "DB8000_PART_STATUS".UNIT_02.STATION_1.PART_A.STATUS.PART_CELL_STATUS_COLOR := 3;
       "DB2401_DBB_DEFINE".PART_STATUS.DBB_1073 := 3;
   END_IF;
   IF #_w2 AND "DB8000_PART_STATUS".UNIT_02.STATION_1.PART_A.STATUS.CELL_STATUS.U01_ONE_FACE_DONE_ROTATED THEN
       "DB8000_PART_STATUS".UNIT_02.STATION_1.PART_A.STATUS.PART_CELL_STATUS_COLOR := 4;
       "DB2401_DBB_DEFINE".PART_STATUS.DBB_1073 := 4;
   END_IF;
   IF #_w2 AND "DB8000_PART_STATUS".UNIT_02.STATION_1.PART_A.STATUS.UNIT_01_STATUS.FACE_R_STATION_3_DONE THEN
       "DB8000_PART_STATUS".UNIT_02.STATION_1.PART_A.STATUS.PART_CELL_STATUS_COLOR := 5;
       "DB2401_DBB_DEFINE".PART_STATUS.DBB_1073 := 5;
   END_IF;
   IF #_w2 AND "DB8000_PART_STATUS".UNIT_02.STATION_1.PART_A.STATUS.UNIT_01_STATUS.FACE_R_STATION_4_DONE THEN
       "DB8000_PART_STATUS".UNIT_02.STATION_1.PART_A.STATUS.PART_CELL_STATUS_COLOR := 6;
       "DB2401_DBB_DEFINE".PART_STATUS.DBB_1073 := 6;
   END_IF;
   IF #_w2 AND "DB8000_PART_STATUS".UNIT_02.STATION_1.PART_A.STATUS.CELL_STATUS.U01_DONE_IN_TRANSIT THEN
       "DB8000_PART_STATUS".UNIT_02.STATION_1.PART_A.STATUS.PART_CELL_STATUS_COLOR := 7;
       "DB2401_DBB_DEFINE".PART_STATUS.DBB_1073 := 7;
   END_IF;
   IF #_w2 AND "DB8000_PART_STATUS".UNIT_02.STATION_1.PART_A.STATUS.UNIT_02_STATUS.FACE_N_STATION_2_DONE THEN
       "DB8000_PART_STATUS".UNIT_02.STATION_1.PART_A.STATUS.PART_CELL_STATUS_COLOR := 8;
       "DB2401_DBB_DEFINE".PART_STATUS.DBB_1073 := 8;
   END_IF;
   IF #_w2 AND "DB8000_PART_STATUS".UNIT_02.STATION_1.PART_A.STATUS.UNIT_02_STATUS.FACE_N_STATION_3_DONE THEN
       "DB8000_PART_STATUS".UNIT_02.STATION_1.PART_A.STATUS.PART_CELL_STATUS_COLOR := 9;
       "DB2401_DBB_DEFINE".PART_STATUS.DBB_1073 := 9;
   END_IF;
   IF #_w2 AND "DB8000_PART_STATUS".UNIT_02.STATION_1.PART_A.STATUS.UNIT_02_STATUS.FACE_N_STATION_4_DONE THEN
       "DB8000_PART_STATUS".UNIT_02.STATION_1.PART_A.STATUS.PART_CELL_STATUS_COLOR := 10;
       "DB2401_DBB_DEFINE".PART_STATUS.DBB_1073 := 10;
   END_IF;
   IF #_w2 AND "DB8000_PART_STATUS".UNIT_02.STATION_1.PART_A.STATUS.CELL_STATUS.U02_ONE_FACE_DONE_ROTATED THEN
       "DB8000_PART_STATUS".UNIT_02.STATION_1.PART_A.STATUS.PART_CELL_STATUS_COLOR := 11;
       "DB2401_DBB_DEFINE".PART_STATUS.DBB_1073 := 11;
   END_IF;
   IF #_w2 AND "DB8000_PART_STATUS".UNIT_02.STATION_1.PART_A.STATUS.UNIT_02_STATUS.FACE_R_STATION_2_DONE THEN
       "DB8000_PART_STATUS".UNIT_02.STATION_1.PART_A.STATUS.PART_CELL_STATUS_COLOR := 12;
       "DB2401_DBB_DEFINE".PART_STATUS.DBB_1073 := 12;
   END_IF;
   IF #_w2 AND "DB8000_PART_STATUS".UNIT_02.STATION_1.PART_A.STATUS.UNIT_02_STATUS.FACE_R_STATION_3_DONE THEN
       "DB8000_PART_STATUS".UNIT_02.STATION_1.PART_A.STATUS.PART_CELL_STATUS_COLOR := 13;
       "DB2401_DBB_DEFINE".PART_STATUS.DBB_1073 := 13;
   END_IF;
   IF #_w2 AND "DB8000_PART_STATUS".UNIT_02.STATION_1.PART_A.STATUS.UNIT_02_STATUS.FACE_R_STATION_4_DONE THEN
       "DB8000_PART_STATUS".UNIT_02.STATION_1.PART_A.STATUS.PART_CELL_STATUS_COLOR := 14;
       "DB2401_DBB_DEFINE".PART_STATUS.DBB_1073 := 14;
   END_IF;
   IF #_w2 AND "DB8000_PART_STATUS".UNIT_02.STATION_1.PART_A.STATUS.CELL_STATUS.U02_DONE_IN_TRANSIT THEN
       "DB8000_PART_STATUS".UNIT_02.STATION_1.PART_A.STATUS.PART_CELL_STATUS_COLOR := 15;
       "DB2401_DBB_DEFINE".PART_STATUS.DBB_1073 := 15;
   END_IF;
   IF #_w2 AND "DB8000_PART_STATUS".UNIT_02.STATION_1.PART_A.STATUS.CELL_STATUS.COOLING_DONE THEN
       "DB8000_PART_STATUS".UNIT_02.STATION_1.PART_A.STATUS.PART_CELL_STATUS_COLOR := 16;
       "DB2401_DBB_DEFINE".PART_STATUS.DBB_1073 := 16;
   END_IF;
   IF #_w2 AND "DB8000_PART_STATUS".UNIT_02.STATION_1.PART_A.STATUS.CELL_STATUS.INSPECTION_DONE THEN
       "DB8000_PART_STATUS".UNIT_02.STATION_1.PART_A.STATUS.PART_CELL_STATUS_COLOR := 17;
       "DB2401_DBB_DEFINE".PART_STATUS.DBB_1073 := 17;
   END_IF;
   IF #_w2 AND "DB8000_PART_STATUS".UNIT_02.STATION_1.PART_A.STATUS.MASTER_PART THEN
       "DB8000_PART_STATUS".UNIT_02.STATION_1.PART_A.STATUS.PART_CELL_STATUS_COLOR := 99;
       "DB2401_DBB_DEFINE".PART_STATUS.DBB_1073 := 99;
   END_IF;
END_REGION

